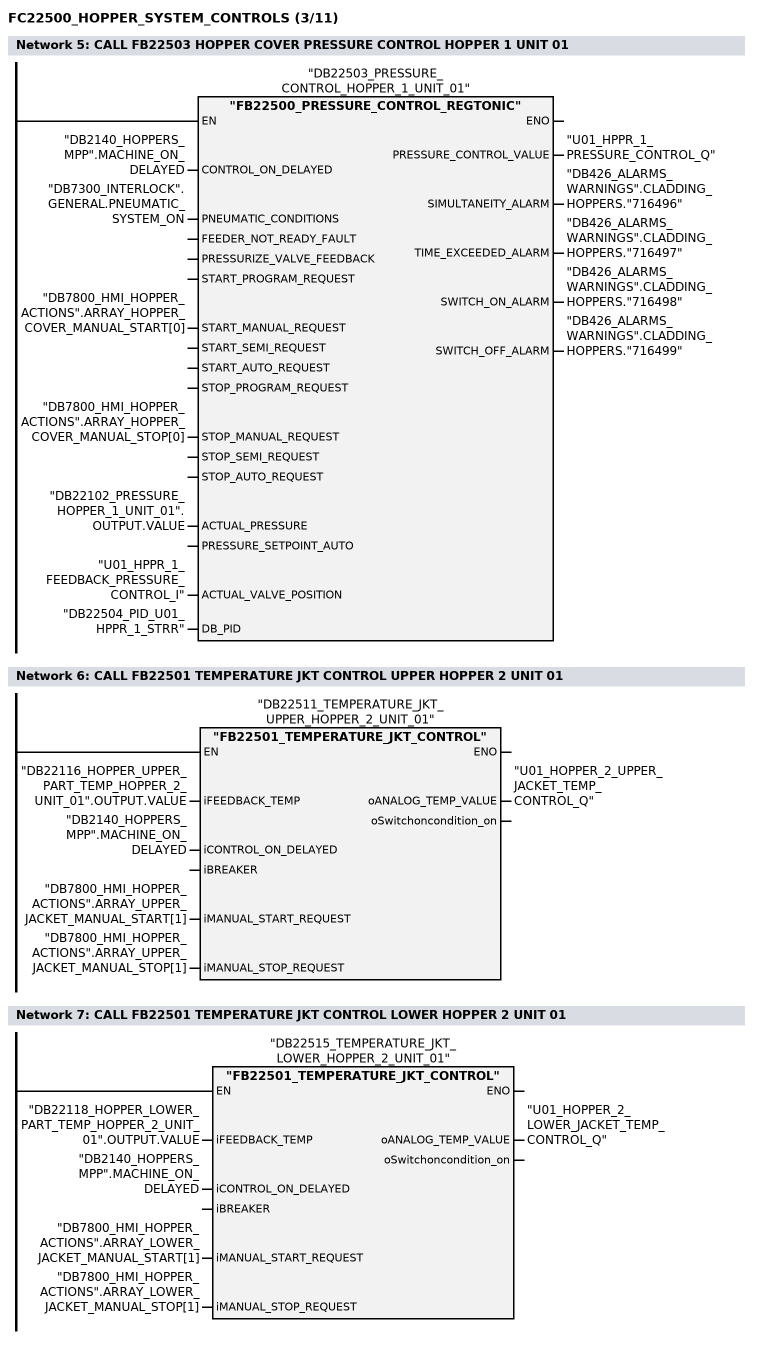
   RUNG wire#powerrail
      "DB22503_PRESSURE_CONTROL_HOPPER_1_UNIT_01"(CONTROL_ON_DELAYED := "DB2140_HOPPERS_MPP".MACHINE_ON_DELAYED, PNEUMATIC_CONDITIONS := "DB7300_INTERLOCK".GENERAL.PNEUMATIC_SYSTEM_ON, FEEDER_NOT_READY_FAULT :=, PRESSURIZE_VALVE_FEEDBACK :=, START_PROGRAM_REQUEST :=, START_MANUAL_REQUEST := "DB7800_HMI_HOPPER_ACTIONS".ARRAY_HOPPER_COVER_MANUAL_START[0], START_SEMI_REQUEST :=, START_AUTO_REQUEST :=, STOP_PROGRAM_REQUEST :=, STOP_MANUAL_REQUEST := "DB7800_HMI_HOPPER_ACTIONS".ARRAY_HOPPER_COVER_MANUAL_STOP[0], STOP_SEMI_REQUEST :=, STOP_AUTO_REQUEST :=, ACTUAL_PRESSURE := "DB22102_PRESSURE_HOPPER_1_UNIT_01".OUTPUT.VALUE, PRESSURE_SETPOINT_AUTO :=, ACTUAL_VALVE_POSITION := "U01_HPPR_1_FEEDBACK_PRESSURE_CONTROL_I", DB_PID := "DB22504_PID_U01_HPPR_1_STRR", PRESSURE_CONTROL_VALUE => "U01_HPPR_1_PRESSURE_CONTROL_Q", SIMULTANEITY_ALARM => "DB426_ALARMS_WARNINGS".CLADDING_HOPPERS."716496", TIME_EXCEEDED_ALARM => "DB426_ALARMS_WARNINGS".CLADDING_HOPPERS."716497", SWITCH_ON_ALARM => "DB426_ALARMS_WARNINGS".CLADDING_HOPPERS."716498", SWITCH_OFF_ALARM => "DB426_ALARMS_WARNINGS".CLADDING_HOPPERS."716499")
   END_RUNG
   // the same network as SCL:
   "DB22503_PRESSURE_CONTROL_HOPPER_1_UNIT_01"(CONTROL_ON_DELAYED := "DB2140_HOPPERS_MPP".MACHINE_ON_DELAYED,   // "FB22500_PRESSURE_CONTROL_REGTONIC"
                           PNEUMATIC_CONDITIONS := "DB7300_INTERLOCK".GENERAL.PNEUMATIC_SYSTEM_ON,
                           START_MANUAL_REQUEST := "DB7800_HMI_HOPPER_ACTIONS".ARRAY_HOPPER_COVER_MANUAL_START[0],
                           STOP_MANUAL_REQUEST := "DB7800_HMI_HOPPER_ACTIONS".ARRAY_HOPPER_COVER_MANUAL_STOP[0],
                           ACTUAL_PRESSURE := "DB22102_PRESSURE_HOPPER_1_UNIT_01".OUTPUT.VALUE,
                           ACTUAL_VALVE_POSITION := "U01_HPPR_1_FEEDBACK_PRESSURE_CONTROL_I",
                           DB_PID := "DB22504_PID_U01_HPPR_1_STRR",
                           PRESSURE_CONTROL_VALUE => "U01_HPPR_1_PRESSURE_CONTROL_Q",
                           SIMULTANEITY_ALARM => "DB426_ALARMS_WARNINGS".CLADDING_HOPPERS."716496",
                           TIME_EXCEEDED_ALARM => "DB426_ALARMS_WARNINGS".CLADDING_HOPPERS."716497",
                           SWITCH_ON_ALARM => "DB426_ALARMS_WARNINGS".CLADDING_HOPPERS."716498",
                           SWITCH_OFF_ALARM => "DB426_ALARMS_WARNINGS".CLADDING_HOPPERS."716499");
END_REGION

REGION Network 6: CALL FB22501 TEMPERATURE JKT CONTROL UPPER HOPPER 2 UNIT 01
   RUNG wire#powerrail
      "DB22511_TEMPERATURE_JKT_UPPER_HOPPER_2_UNIT_01"(iFEEDBACK_TEMP := "DB22116_HOPPER_UPPER_PART_TEMP_HOPPER_2_UNIT_01".OUTPUT.VALUE, iCONTROL_ON_DELAYED := "DB2140_HOPPERS_MPP".MACHINE_ON_DELAYED, iBREAKER :=, iMANUAL_START_REQUEST := "DB7800_HMI_HOPPER_ACTIONS".ARRAY_UPPER_JACKET_MANUAL_START[1], iMANUAL_STOP_REQUEST := "DB7800_HMI_HOPPER_ACTIONS".ARRAY_UPPER_JACKET_MANUAL_STOP[1], oANALOG_TEMP_VALUE => "U01_HOPPER_2_UPPER_JACKET_TEMP_CONTROL_Q", oSwitchoncondition_on =>)
   END_RUNG
   // the same network as SCL:
   "DB22511_TEMPERATURE_JKT_UPPER_HOPPER_2_UNIT_01"(iFEEDBACK_TEMP := "DB22116_HOPPER_UPPER_PART_TEMP_HOPPER_2_UNIT_01".OUTPUT.VALUE,   // "FB22501_TEMPERATURE_JKT_CONTROL"
                           iCONTROL_ON_DELAYED := "DB2140_HOPPERS_MPP".MACHINE_ON_DELAYED,
                           iMANUAL_START_REQUEST := "DB7800_HMI_HOPPER_ACTIONS".ARRAY_UPPER_JACKET_MANUAL_START[1],
                           iMANUAL_STOP_REQUEST := "DB7800_HMI_HOPPER_ACTIONS".ARRAY_UPPER_JACKET_MANUAL_STOP[1],
                           oANALOG_TEMP_VALUE => "U01_HOPPER_2_UPPER_JACKET_TEMP_CONTROL_Q");
END_REGION

REGION Network 7: CALL FB22501 TEMPERATURE JKT CONTROL LOWER HOPPER 2 UNIT 01
   RUNG wire#powerrail
      "DB22515_TEMPERATURE_JKT_LOWER_HOPPER_2_UNIT_01"(iFEEDBACK_TEMP := "DB22118_HOPPER_LOWER_PART_TEMP_HOPPER_2_UNIT_01".OUTPUT.VALUE, iCONTROL_ON_DELAYED := "DB2140_HOPPERS_MPP".MACHINE_ON_DELAYED, iBREAKER :=, iMANUAL_START_REQUEST := "DB7800_HMI_HOPPER_ACTIONS".ARRAY_LOWER_JACKET_MANUAL_START[1], iMANUAL_STOP_REQUEST := "DB7800_HMI_HOPPER_ACTIONS".ARRAY_LOWER_JACKET_MANUAL_STOP[1], oANALOG_TEMP_VALUE => "U01_HOPPER_2_LOWER_JACKET_TEMP_CONTROL_Q", oSwitchoncondition_on =>)
   END_RUNG
   // the same network as SCL:
   "DB22515_TEMPERATURE_JKT_LOWER_HOPPER_2_UNIT_01"(iFEEDBACK_TEMP := "DB22118_HOPPER_LOWER_PART_TEMP_HOPPER_2_UNIT_01".OUTPUT.VALUE,   // "FB22501_TEMPERATURE_JKT_CONTROL"
                           iCONTROL_ON_DELAYED := "DB2140_HOPPERS_MPP".MACHINE_ON_DELAYED,
                           iMANUAL_START_REQUEST := "DB7800_HMI_HOPPER_ACTIONS".ARRAY_LOWER_JACKET_MANUAL_START[1],
                           iMANUAL_STOP_REQUEST := "DB7800_HMI_HOPPER_ACTIONS".ARRAY_LOWER_JACKET_MANUAL_STOP[1],
                           oANALOG_TEMP_VALUE => "U01_HOPPER_2_LOWER_JACKET_TEMP_CONTROL_Q");
END_REGION

REGION Network 8: CALL FB22502 MOTOR STIRRER CONTROL HOPPER 2 UNIT 01
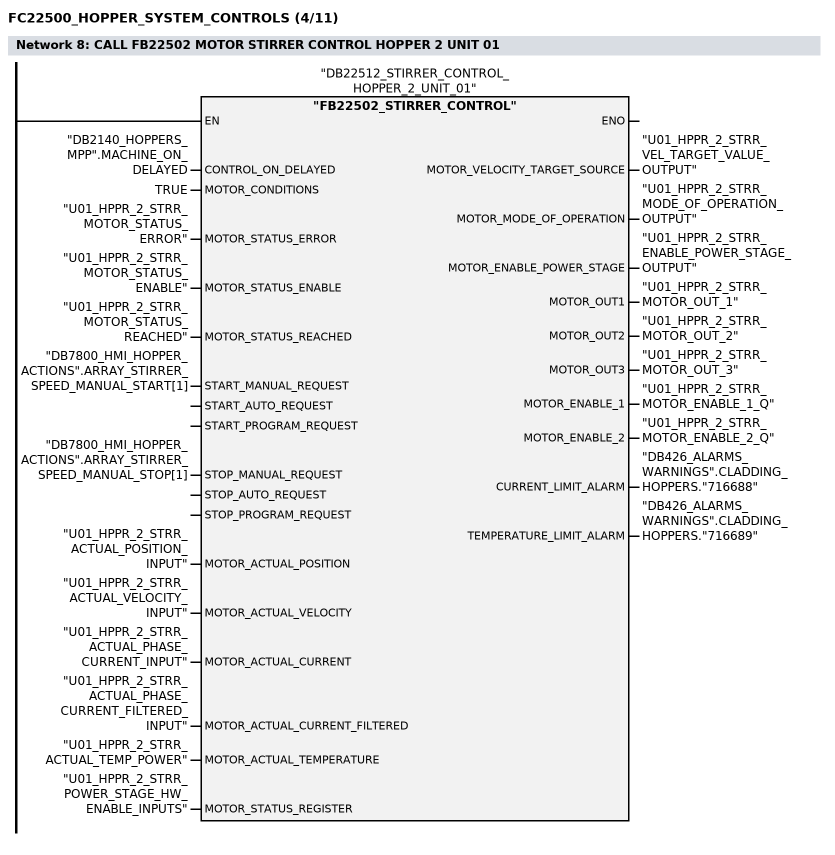
   RUNG wire#powerrail
      "DB22512_STIRRER_CONTROL_HOPPER_2_UNIT_01"(CONTROL_ON_DELAYED := "DB2140_HOPPERS_MPP".MACHINE_ON_DELAYED, MOTOR_CONDITIONS := TRUE, MOTOR_STATUS_ERROR := "U01_HPPR_2_STRR_MOTOR_STATUS_ERROR", MOTOR_STATUS_ENABLE := "U01_HPPR_2_STRR_MOTOR_STATUS_ENABLE", MOTOR_STATUS_REACHED := "U01_HPPR_2_STRR_MOTOR_STATUS_REACHED", START_MANUAL_REQUEST := "DB7800_HMI_HOPPER_ACTIONS".ARRAY_STIRRER_SPEED_MANUAL_START[1], START_AUTO_REQUEST :=, START_PROGRAM_REQUEST :=, STOP_MANUAL_REQUEST := "DB7800_HMI_HOPPER_ACTIONS".ARRAY_STIRRER_SPEED_MANUAL_STOP[1], STOP_AUTO_REQUEST :=, STOP_PROGRAM_REQUEST :=, MOTOR_ACTUAL_POSITION := "U01_HPPR_2_STRR_ACTUAL_POSITION_INPUT", MOTOR_ACTUAL_VELOCITY := "U01_HPPR_2_STRR_ACTUAL_VELOCITY_INPUT", MOTOR_ACTUAL_CURRENT := "U01_HPPR_2_STRR_ACTUAL_PHASE_CURRENT_INPUT", MOTOR_ACTUAL_CURRENT_FILTERED := "U01_HPPR_2_STRR_ACTUAL_PHASE_CURRENT_FILTERED_INPUT", MOTOR_ACTUAL_TEMPERATURE := "U01_HPPR_2_STRR_ACTUAL_TEMP_POWER", MOTOR_STATUS_REGISTER := "U01_HPPR_2_STRR_POWER_STAGE_HW_ENABLE_INPUTS", MOTOR_VELOCITY_TARGET_SOURCE => "U01_HPPR_2_STRR_VEL_TARGET_VALUE_OUTPUT", MOTOR_MODE_OF_OPERATION => "U01_HPPR_2_STRR_MODE_OF_OPERATION_OUTPUT", MOTOR_ENABLE_POWER_STAGE => "U01_HPPR_2_STRR_ENABLE_POWER_STAGE_OUTPUT", MOTOR_OUT1 => "U01_HPPR_2_STRR_MOTOR_OUT_1", MOTOR_OUT2 => "U01_HPPR_2_STRR_MOTOR_OUT_2", MOTOR_OUT3 => "U01_HPPR_2_STRR_MOTOR_OUT_3", MOTOR_ENABLE_1 => "U01_HPPR_2_STRR_MOTOR_ENABLE_1_Q", MOTOR_ENABLE_2 => "U01_HPPR_2_STRR_MOTOR_ENABLE_2_Q", CURRENT_LIMIT_ALARM => "DB426_ALARMS_WARNINGS".CLADDING_HOPPERS."716688", TEMPERATURE_LIMIT_ALARM => "DB426_ALARMS_WARNINGS".CLADDING_HOPPERS."716689")
   END_RUNG
   // the same network as SCL:
   "DB22512_STIRRER_CONTROL_HOPPER_2_UNIT_01"(CONTROL_ON_DELAYED := "DB2140_HOPPERS_MPP".MACHINE_ON_DELAYED,   // "FB22502_STIRRER_CONTROL"
                           MOTOR_CONDITIONS := TRUE,
                           MOTOR_STATUS_ERROR := "U01_HPPR_2_STRR_MOTOR_STATUS_ERROR",
                           MOTOR_STATUS_ENABLE := "U01_HPPR_2_STRR_MOTOR_STATUS_ENABLE",
                           MOTOR_STATUS_REACHED := "U01_HPPR_2_STRR_MOTOR_STATUS_REACHED",
                           START_MANUAL_REQUEST := "DB7800_HMI_HOPPER_ACTIONS".ARRAY_STIRRER_SPEED_MANUAL_START[1],
                           STOP_MANUAL_REQUEST := "DB7800_HMI_HOPPER_ACTIONS".ARRAY_STIRRER_SPEED_MANUAL_STOP[1],
                           MOTOR_ACTUAL_POSITION := "U01_HPPR_2_STRR_ACTUAL_POSITION_INPUT",
                           MOTOR_ACTUAL_VELOCITY := "U01_HPPR_2_STRR_ACTUAL_VELOCITY_INPUT",
                           MOTOR_ACTUAL_CURRENT := "U01_HPPR_2_STRR_ACTUAL_PHASE_CURRENT_INPUT",
                           MOTOR_ACTUAL_CURRENT_FILTERED := "U01_HPPR_2_STRR_ACTUAL_PHASE_CURRENT_FILTERED_INPUT",
                           MOTOR_ACTUAL_TEMPERATURE := "U01_HPPR_2_STRR_ACTUAL_TEMP_POWER",
                           MOTOR_STATUS_REGISTER := "U01_HPPR_2_STRR_POWER_STAGE_HW_ENABLE_INPUTS",
                           MOTOR_VELOCITY_TARGET_SOURCE => "U01_HPPR_2_STRR_VEL_TARGET_VALUE_OUTPUT",
                           MOTOR_MODE_OF_OPERATION => "U01_HPPR_2_STRR_MODE_OF_OPERATION_OUTPUT",
                           MOTOR_ENABLE_POWER_STAGE => "U01_HPPR_2_STRR_ENABLE_POWER_STAGE_OUTPUT",
                           MOTOR_OUT1 => "U01_HPPR_2_STRR_MOTOR_OUT_1",
                           MOTOR_OUT2 => "U01_HPPR_2_STRR_MOTOR_OUT_2",
                           MOTOR_OUT3 => "U01_HPPR_2_STRR_MOTOR_OUT_3",
                           MOTOR_ENABLE_1 => "U01_HPPR_2_STRR_MOTOR_ENABLE_1_Q",
                           MOTOR_ENABLE_2 => "U01_HPPR_2_STRR_MOTOR_ENABLE_2_Q",
                           CURRENT_LIMIT_ALARM => "DB426_ALARMS_WARNINGS".CLADDING_HOPPERS."716688",
                           TEMPERATURE_LIMIT_ALARM => "DB426_ALARMS_WARNINGS".CLADDING_HOPPERS."716689");
END_REGION

REGION Network 9: CALL FB22503 HOPPER PRESSURE CONTROL HOPPER 2 UNIT 01
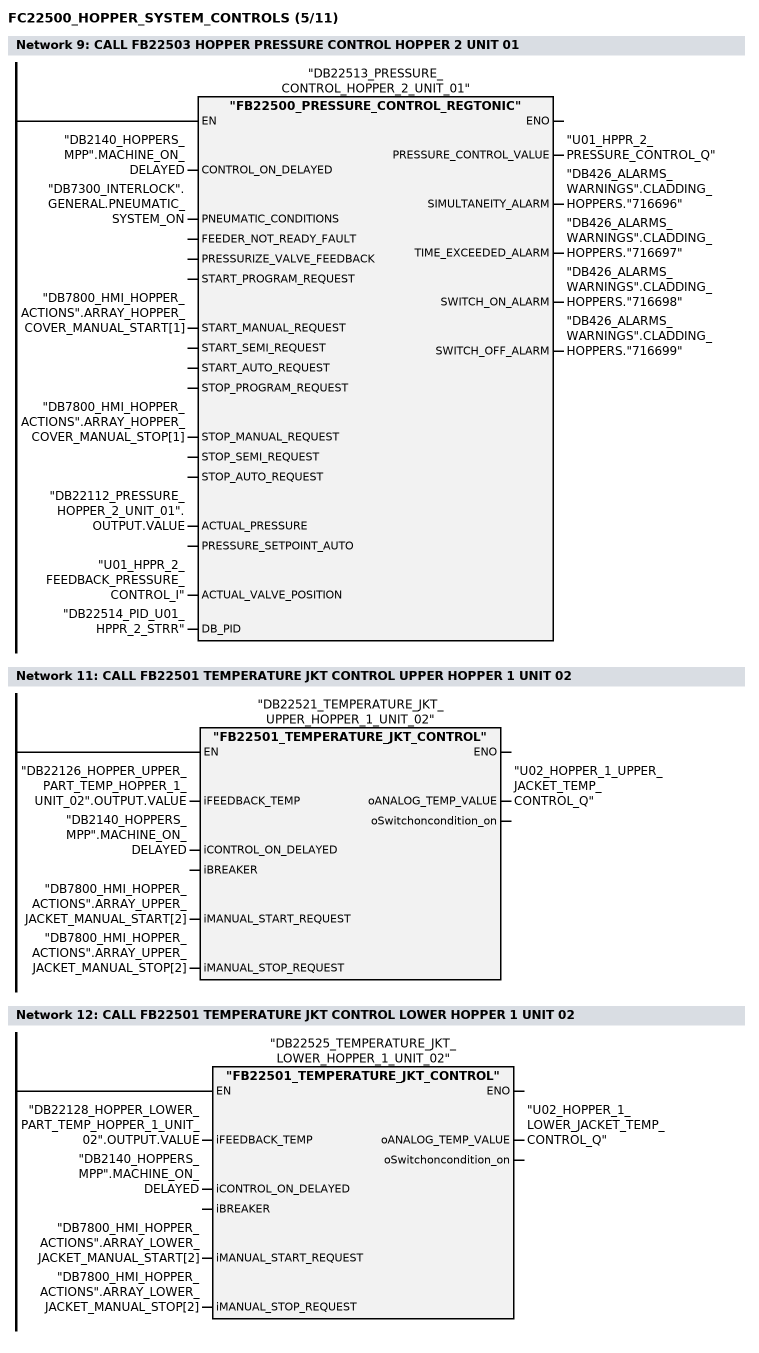
   RUNG wire#powerrail
      "DB22513_PRESSURE_CONTROL_HOPPER_2_UNIT_01"(CONTROL_ON_DELAYED := "DB2140_HOPPERS_MPP".MACHINE_ON_DELAYED, PNEUMATIC_CONDITIONS := "DB7300_INTERLOCK".GENERAL.PNEUMATIC_SYSTEM_ON, FEEDER_NOT_READY_FAULT :=, PRESSURIZE_VALVE_FEEDBACK :=, START_PROGRAM_REQUEST :=, START_MANUAL_REQUEST := "DB7800_HMI_HOPPER_ACTIONS".ARRAY_HOPPER_COVER_MANUAL_START[1], START_SEMI_REQUEST :=, START_AUTO_REQUEST :=, STOP_PROGRAM_REQUEST :=, STOP_MANUAL_REQUEST := "DB7800_HMI_HOPPER_ACTIONS".ARRAY_HOPPER_COVER_MANUAL_STOP[1], STOP_SEMI_REQUEST :=, STOP_AUTO_REQUEST :=, ACTUAL_PRESSURE := "DB22112_PRESSURE_HOPPER_2_UNIT_01".OUTPUT.VALUE, PRESSURE_SETPOINT_AUTO :=, ACTUAL_VALVE_POSITION := "U01_HPPR_2_FEEDBACK_PRESSURE_CONTROL_I", DB_PID := "DB22514_PID_U01_HPPR_2_STRR", PRESSURE_CONTROL_VALUE => "U01_HPPR_2_PRESSURE_CONTROL_Q", SIMULTANEITY_ALARM => "DB426_ALARMS_WARNINGS".CLADDING_HOPPERS."716696", TIME_EXCEEDED_ALARM => "DB426_ALARMS_WARNINGS".CLADDING_HOPPERS."716697", SWITCH_ON_ALARM => "DB426_ALARMS_WARNINGS".CLADDING_HOPPERS."716698", SWITCH_OFF_ALARM => "DB426_ALARMS_WARNINGS".CLADDING_HOPPERS."716699")
   END_RUNG
   // the same network as SCL:
   "DB22513_PRESSURE_CONTROL_HOPPER_2_UNIT_01"(CONTROL_ON_DELAYED := "DB2140_HOPPERS_MPP".MACHINE_ON_DELAYED,   // "FB22500_PRESSURE_CONTROL_REGTONIC"
                           PNEUMATIC_CONDITIONS := "DB7300_INTERLOCK".GENERAL.PNEUMATIC_SYSTEM_ON,
                           START_MANUAL_REQUEST := "DB7800_HMI_HOPPER_ACTIONS".ARRAY_HOPPER_COVER_MANUAL_START[1],
                           STOP_MANUAL_REQUEST := "DB7800_HMI_HOPPER_ACTIONS".ARRAY_HOPPER_COVER_MANUAL_STOP[1],
                           ACTUAL_PRESSURE := "DB22112_PRESSURE_HOPPER_2_UNIT_01".OUTPUT.VALUE,
                           ACTUAL_VALVE_POSITION := "U01_HPPR_2_FEEDBACK_PRESSURE_CONTROL_I",
                           DB_PID := "DB22514_PID_U01_HPPR_2_STRR",
                           PRESSURE_CONTROL_VALUE => "U01_HPPR_2_PRESSURE_CONTROL_Q",
                           SIMULTANEITY_ALARM => "DB426_ALARMS_WARNINGS".CLADDING_HOPPERS."716696",
                           TIME_EXCEEDED_ALARM => "DB426_ALARMS_WARNINGS".CLADDING_HOPPERS."716697",
                           SWITCH_ON_ALARM => "DB426_ALARMS_WARNINGS".CLADDING_HOPPERS."716698",
                           SWITCH_OFF_ALARM => "DB426_ALARMS_WARNINGS".CLADDING_HOPPERS."716699");
END_REGION

REGION Network 10: //////////UNIT 02 HOPERS CONTROLS//////////
END_REGION

REGION Network 11: CALL FB22501 TEMPERATURE JKT CONTROL UPPER HOPPER 1 UNIT 02
   RUNG wire#powerrail
      "DB22521_TEMPERATURE_JKT_UPPER_HOPPER_1_UNIT_02"(iFEEDBACK_TEMP := "DB22126_HOPPER_UPPER_PART_TEMP_HOPPER_1_UNIT_02".OUTPUT.VALUE, iCONTROL_ON_DELAYED := "DB2140_HOPPERS_MPP".MACHINE_ON_DELAYED, iBREAKER :=, iMANUAL_START_REQUEST := "DB7800_HMI_HOPPER_ACTIONS".ARRAY_UPPER_JACKET_MANUAL_START[2], iMANUAL_STOP_REQUEST := "DB7800_HMI_HOPPER_ACTIONS".ARRAY_UPPER_JACKET_MANUAL_STOP[2], oANALOG_TEMP_VALUE => "U02_HOPPER_1_UPPER_JACKET_TEMP_CONTROL_Q", oSwitchoncondition_on =>)
   END_RUNG
   // the same network as SCL:
   "DB22521_TEMPERATURE_JKT_UPPER_HOPPER_1_UNIT_02"(iFEEDBACK_TEMP := "DB22126_HOPPER_UPPER_PART_TEMP_HOPPER_1_UNIT_02".OUTPUT.VALUE,   // "FB22501_TEMPERATURE_JKT_CONTROL"
                           iCONTROL_ON_DELAYED := "DB2140_HOPPERS_MPP".MACHINE_ON_DELAYED,
                           iMANUAL_START_REQUEST := "DB7800_HMI_HOPPER_ACTIONS".ARRAY_UPPER_JACKET_MANUAL_START[2],
                           iMANUAL_STOP_REQUEST := "DB7800_HMI_HOPPER_ACTIONS".ARRAY_UPPER_JACKET_MANUAL_STOP[2],
                           oANALOG_TEMP_VALUE => "U02_HOPPER_1_UPPER_JACKET_TEMP_CONTROL_Q");
END_REGION

REGION Network 12: CALL FB22501 TEMPERATURE JKT CONTROL LOWER HOPPER 1 UNIT 02
   RUNG wire#powerrail
      "DB22525_TEMPERATURE_JKT_LOWER_HOPPER_1_UNIT_02"(iFEEDBACK_TEMP := "DB22128_HOPPER_LOWER_PART_TEMP_HOPPER_1_UNIT_02".OUTPUT.VALUE, iCONTROL_ON_DELAYED := "DB2140_HOPPERS_MPP".MACHINE_ON_DELAYED, iBREAKER :=, iMANUAL_START_REQUEST := "DB7800_HMI_HOPPER_ACTIONS".ARRAY_LOWER_JACKET_MANUAL_START[2], iMANUAL_STOP_REQUEST := "DB7800_HMI_HOPPER_ACTIONS".ARRAY_LOWER_JACKET_MANUAL_STOP[2], oANALOG_TEMP_VALUE => "U02_HOPPER_1_LOWER_JACKET_TEMP_CONTROL_Q", oSwitchoncondition_on =>)
   END_RUNG
   // the same network as SCL:
   "DB22525_TEMPERATURE_JKT_LOWER_HOPPER_1_UNIT_02"(iFEEDBACK_TEMP := "DB22128_HOPPER_LOWER_PART_TEMP_HOPPER_1_UNIT_02".OUTPUT.VALUE,   // "FB22501_TEMPERATURE_JKT_CONTROL"
                           iCONTROL_ON_DELAYED := "DB2140_HOPPERS_MPP".MACHINE_ON_DELAYED,
                           iMANUAL_START_REQUEST := "DB7800_HMI_HOPPER_ACTIONS".ARRAY_LOWER_JACKET_MANUAL_START[2],
                           iMANUAL_STOP_REQUEST := "DB7800_HMI_HOPPER_ACTIONS".ARRAY_LOWER_JACKET_MANUAL_STOP[2],
                           oANALOG_TEMP_VALUE => "U02_HOPPER_1_LOWER_JACKET_TEMP_CONTROL_Q");
END_REGION

REGION Network 13: CALL FB22502 MOTOR STIRRER CONTROL HOPPER 1 UNIT 02
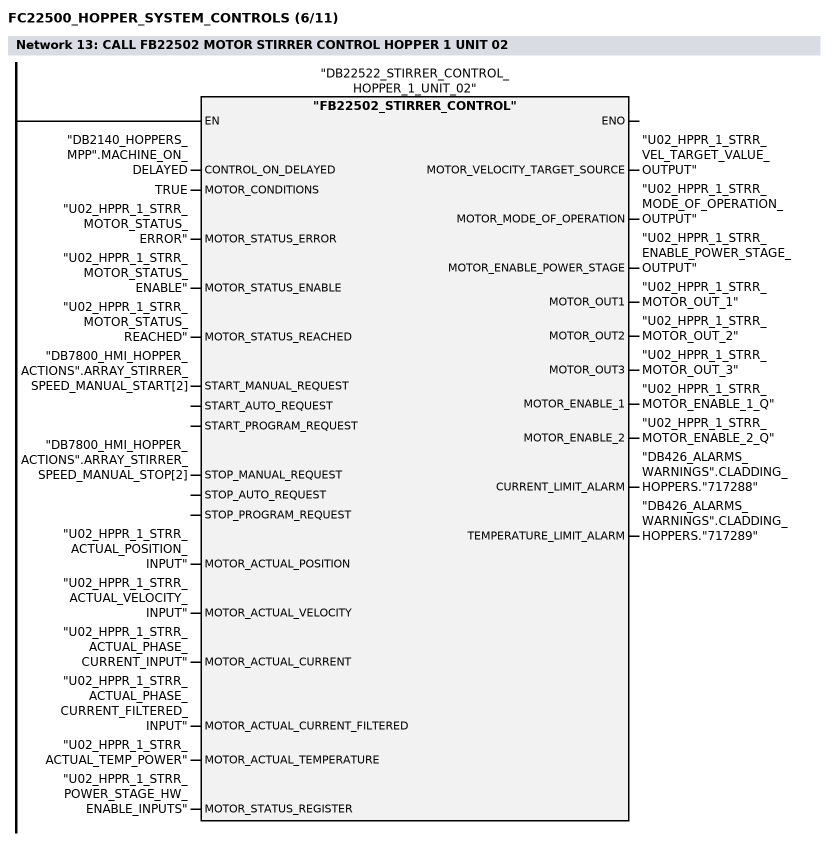
   RUNG wire#powerrail
      "DB22522_STIRRER_CONTROL_HOPPER_1_UNIT_02"(CONTROL_ON_DELAYED := "DB2140_HOPPERS_MPP".MACHINE_ON_DELAYED, MOTOR_CONDITIONS := TRUE, MOTOR_STATUS_ERROR := "U02_HPPR_1_STRR_MOTOR_STATUS_ERROR", MOTOR_STATUS_ENABLE := "U02_HPPR_1_STRR_MOTOR_STATUS_ENABLE", MOTOR_STATUS_REACHED := "U02_HPPR_1_STRR_MOTOR_STATUS_REACHED", START_MANUAL_REQUEST := "DB7800_HMI_HOPPER_ACTIONS".ARRAY_STIRRER_SPEED_MANUAL_START[2], START_AUTO_REQUEST :=, START_PROGRAM_REQUEST :=, STOP_MANUAL_REQUEST := "DB7800_HMI_HOPPER_ACTIONS".ARRAY_STIRRER_SPEED_MANUAL_STOP[2], STOP_AUTO_REQUEST :=, STOP_PROGRAM_REQUEST :=, MOTOR_ACTUAL_POSITION := "U02_HPPR_1_STRR_ACTUAL_POSITION_INPUT", MOTOR_ACTUAL_VELOCITY := "U02_HPPR_1_STRR_ACTUAL_VELOCITY_INPUT", MOTOR_ACTUAL_CURRENT := "U02_HPPR_1_STRR_ACTUAL_PHASE_CURRENT_INPUT", MOTOR_ACTUAL_CURRENT_FILTERED := "U02_HPPR_1_STRR_ACTUAL_PHASE_CURRENT_FILTERED_INPUT", MOTOR_ACTUAL_TEMPERATURE := "U02_HPPR_1_STRR_ACTUAL_TEMP_POWER", MOTOR_STATUS_REGISTER := "U02_HPPR_1_STRR_POWER_STAGE_HW_ENABLE_INPUTS", MOTOR_VELOCITY_TARGET_SOURCE => "U02_HPPR_1_STRR_VEL_TARGET_VALUE_OUTPUT", MOTOR_MODE_OF_OPERATION => "U02_HPPR_1_STRR_MODE_OF_OPERATION_OUTPUT", MOTOR_ENABLE_POWER_STAGE => "U02_HPPR_1_STRR_ENABLE_POWER_STAGE_OUTPUT", MOTOR_OUT1 => "U02_HPPR_1_STRR_MOTOR_OUT_1", MOTOR_OUT2 => "U02_HPPR_1_STRR_MOTOR_OUT_2", MOTOR_OUT3 => "U02_HPPR_1_STRR_MOTOR_OUT_3", MOTOR_ENABLE_1 => "U02_HPPR_1_STRR_MOTOR_ENABLE_1_Q", MOTOR_ENABLE_2 => "U02_HPPR_1_STRR_MOTOR_ENABLE_2_Q", CURRENT_LIMIT_ALARM => "DB426_ALARMS_WARNINGS".CLADDING_HOPPERS."717288", TEMPERATURE_LIMIT_ALARM => "DB426_ALARMS_WARNINGS".CLADDING_HOPPERS."717289")
   END_RUNG
   // the same network as SCL:
   "DB22522_STIRRER_CONTROL_HOPPER_1_UNIT_02"(CONTROL_ON_DELAYED := "DB2140_HOPPERS_MPP".MACHINE_ON_DELAYED,   // "FB22502_STIRRER_CONTROL"
                           MOTOR_CONDITIONS := TRUE,
                           MOTOR_STATUS_ERROR := "U02_HPPR_1_STRR_MOTOR_STATUS_ERROR",
                           MOTOR_STATUS_ENABLE := "U02_HPPR_1_STRR_MOTOR_STATUS_ENABLE",
                           MOTOR_STATUS_REACHED := "U02_HPPR_1_STRR_MOTOR_STATUS_REACHED",
                           START_MANUAL_REQUEST := "DB7800_HMI_HOPPER_ACTIONS".ARRAY_STIRRER_SPEED_MANUAL_START[2],
                           STOP_MANUAL_REQUEST := "DB7800_HMI_HOPPER_ACTIONS".ARRAY_STIRRER_SPEED_MANUAL_STOP[2],
                           MOTOR_ACTUAL_POSITION := "U02_HPPR_1_STRR_ACTUAL_POSITION_INPUT",
                           MOTOR_ACTUAL_VELOCITY := "U02_HPPR_1_STRR_ACTUAL_VELOCITY_INPUT",
                           MOTOR_ACTUAL_CURRENT := "U02_HPPR_1_STRR_ACTUAL_PHASE_CURRENT_INPUT",
                           MOTOR_ACTUAL_CURRENT_FILTERED := "U02_HPPR_1_STRR_ACTUAL_PHASE_CURRENT_FILTERED_INPUT",
                           MOTOR_ACTUAL_TEMPERATURE := "U02_HPPR_1_STRR_ACTUAL_TEMP_POWER",
                           MOTOR_STATUS_REGISTER := "U02_HPPR_1_STRR_POWER_STAGE_HW_ENABLE_INPUTS",
                           MOTOR_VELOCITY_TARGET_SOURCE => "U02_HPPR_1_STRR_VEL_TARGET_VALUE_OUTPUT",
                           MOTOR_MODE_OF_OPERATION => "U02_HPPR_1_STRR_MODE_OF_OPERATION_OUTPUT",
                           MOTOR_ENABLE_POWER_STAGE => "U02_HPPR_1_STRR_ENABLE_POWER_STAGE_OUTPUT",
                           MOTOR_OUT1 => "U02_HPPR_1_STRR_MOTOR_OUT_1",
                           MOTOR_OUT2 => "U02_HPPR_1_STRR_MOTOR_OUT_2",
                           MOTOR_OUT3 => "U02_HPPR_1_STRR_MOTOR_OUT_3",
                           MOTOR_ENABLE_1 => "U02_HPPR_1_STRR_MOTOR_ENABLE_1_Q",
                           MOTOR_ENABLE_2 => "U02_HPPR_1_STRR_MOTOR_ENABLE_2_Q",
                           CURRENT_LIMIT_ALARM => "DB426_ALARMS_WARNINGS".CLADDING_HOPPERS."717288",
                           TEMPERATURE_LIMIT_ALARM => "DB426_ALARMS_WARNINGS".CLADDING_HOPPERS."717289");
END_REGION

REGION Network 14: CALL FB22503 HOPPER PRESSURE CONTROL HOPPER 1 UNIT 02
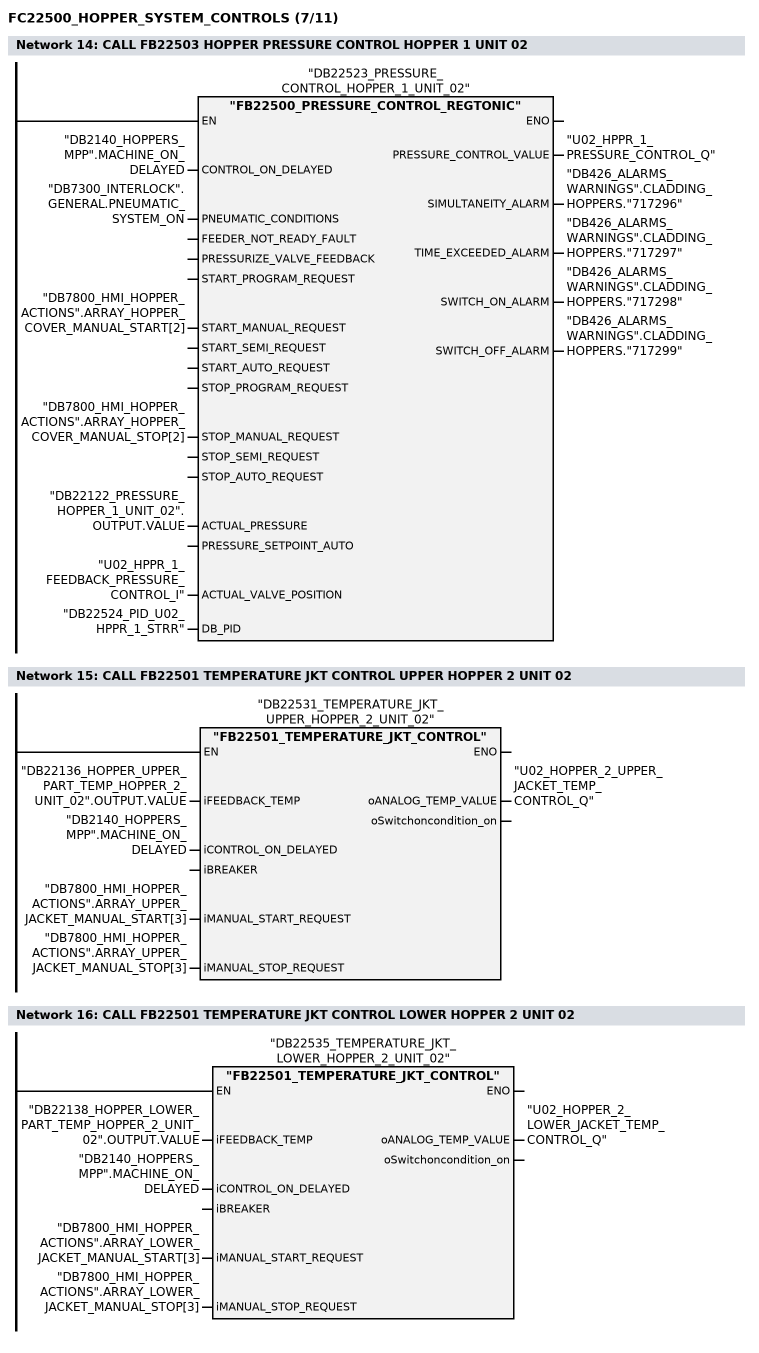
   RUNG wire#powerrail
      "DB22523_PRESSURE_CONTROL_HOPPER_1_UNIT_02"(CONTROL_ON_DELAYED := "DB2140_HOPPERS_MPP".MACHINE_ON_DELAYED, PNEUMATIC_CONDITIONS := "DB7300_INTERLOCK".GENERAL.PNEUMATIC_SYSTEM_ON, FEEDER_NOT_READY_FAULT :=, PRESSURIZE_VALVE_FEEDBACK :=, START_PROGRAM_REQUEST :=, START_MANUAL_REQUEST := "DB7800_HMI_HOPPER_ACTIONS".ARRAY_HOPPER_COVER_MANUAL_START[2], START_SEMI_REQUEST :=, START_AUTO_REQUEST :=, STOP_PROGRAM_REQUEST :=, STOP_MANUAL_REQUEST := "DB7800_HMI_HOPPER_ACTIONS".ARRAY_HOPPER_COVER_MANUAL_STOP[2], STOP_SEMI_REQUEST :=, STOP_AUTO_REQUEST :=, ACTUAL_PRESSURE := "DB22122_PRESSURE_HOPPER_1_UNIT_02".OUTPUT.VALUE, PRESSURE_SETPOINT_AUTO :=, ACTUAL_VALVE_POSITION := "U02_HPPR_1_FEEDBACK_PRESSURE_CONTROL_I", DB_PID := "DB22524_PID_U02_HPPR_1_STRR", PRESSURE_CONTROL_VALUE => "U02_HPPR_1_PRESSURE_CONTROL_Q", SIMULTANEITY_ALARM => "DB426_ALARMS_WARNINGS".CLADDING_HOPPERS."717296", TIME_EXCEEDED_ALARM => "DB426_ALARMS_WARNINGS".CLADDING_HOPPERS."717297", SWITCH_ON_ALARM => "DB426_ALARMS_WARNINGS".CLADDING_HOPPERS."717298", SWITCH_OFF_ALARM => "DB426_ALARMS_WARNINGS".CLADDING_HOPPERS."717299")
   END_RUNG
   // the same network as SCL:
   "DB22523_PRESSURE_CONTROL_HOPPER_1_UNIT_02"(CONTROL_ON_DELAYED := "DB2140_HOPPERS_MPP".MACHINE_ON_DELAYED,   // "FB22500_PRESSURE_CONTROL_REGTONIC"
                           PNEUMATIC_CONDITIONS := "DB7300_INTERLOCK".GENERAL.PNEUMATIC_SYSTEM_ON,
                           START_MANUAL_REQUEST := "DB7800_HMI_HOPPER_ACTIONS".ARRAY_HOPPER_COVER_MANUAL_START[2],
                           STOP_MANUAL_REQUEST := "DB7800_HMI_HOPPER_ACTIONS".ARRAY_HOPPER_COVER_MANUAL_STOP[2],
                           ACTUAL_PRESSURE := "DB22122_PRESSURE_HOPPER_1_UNIT_02".OUTPUT.VALUE,
                           ACTUAL_VALVE_POSITION := "U02_HPPR_1_FEEDBACK_PRESSURE_CONTROL_I",
                           DB_PID := "DB22524_PID_U02_HPPR_1_STRR",
                           PRESSURE_CONTROL_VALUE => "U02_HPPR_1_PRESSURE_CONTROL_Q",
                           SIMULTANEITY_ALARM => "DB426_ALARMS_WARNINGS".CLADDING_HOPPERS."717296",
                           TIME_EXCEEDED_ALARM => "DB426_ALARMS_WARNINGS".CLADDING_HOPPERS."717297",
                           SWITCH_ON_ALARM => "DB426_ALARMS_WARNINGS".CLADDING_HOPPERS."717298",
                           SWITCH_OFF_ALARM => "DB426_ALARMS_WARNINGS".CLADDING_HOPPERS."717299");
END_REGION

REGION Network 15: CALL FB22501 TEMPERATURE JKT CONTROL UPPER HOPPER 2 UNIT 02
   RUNG wire#powerrail
      "DB22531_TEMPERATURE_JKT_UPPER_HOPPER_2_UNIT_02"(iFEEDBACK_TEMP := "DB22136_HOPPER_UPPER_PART_TEMP_HOPPER_2_UNIT_02".OUTPUT.VALUE, iCONTROL_ON_DELAYED := "DB2140_HOPPERS_MPP".MACHINE_ON_DELAYED, iBREAKER :=, iMANUAL_START_REQUEST := "DB7800_HMI_HOPPER_ACTIONS".ARRAY_UPPER_JACKET_MANUAL_START[3], iMANUAL_STOP_REQUEST := "DB7800_HMI_HOPPER_ACTIONS".ARRAY_UPPER_JACKET_MANUAL_STOP[3], oANALOG_TEMP_VALUE => "U02_HOPPER_2_UPPER_JACKET_TEMP_CONTROL_Q", oSwitchoncondition_on =>)
   END_RUNG
   // the same network as SCL:
   "DB22531_TEMPERATURE_JKT_UPPER_HOPPER_2_UNIT_02"(iFEEDBACK_TEMP := "DB22136_HOPPER_UPPER_PART_TEMP_HOPPER_2_UNIT_02".OUTPUT.VALUE,   // "FB22501_TEMPERATURE_JKT_CONTROL"
                           iCONTROL_ON_DELAYED := "DB2140_HOPPERS_MPP".MACHINE_ON_DELAYED,
                           iMANUAL_START_REQUEST := "DB7800_HMI_HOPPER_ACTIONS".ARRAY_UPPER_JACKET_MANUAL_START[3],
                           iMANUAL_STOP_REQUEST := "DB7800_HMI_HOPPER_ACTIONS".ARRAY_UPPER_JACKET_MANUAL_STOP[3],
                           oANALOG_TEMP_VALUE => "U02_HOPPER_2_UPPER_JACKET_TEMP_CONTROL_Q");
END_REGION

REGION Network 16: CALL FB22501 TEMPERATURE JKT CONTROL LOWER HOPPER 2 UNIT 02
   RUNG wire#powerrail
      "DB22535_TEMPERATURE_JKT_LOWER_HOPPER_2_UNIT_02"(iFEEDBACK_TEMP := "DB22138_HOPPER_LOWER_PART_TEMP_HOPPER_2_UNIT_02".OUTPUT.VALUE, iCONTROL_ON_DELAYED := "DB2140_HOPPERS_MPP".MACHINE_ON_DELAYED, iBREAKER :=, iMANUAL_START_REQUEST := "DB7800_HMI_HOPPER_ACTIONS".ARRAY_LOWER_JACKET_MANUAL_START[3], iMANUAL_STOP_REQUEST := "DB7800_HMI_HOPPER_ACTIONS".ARRAY_LOWER_JACKET_MANUAL_STOP[3], oANALOG_TEMP_VALUE => "U02_HOPPER_2_LOWER_JACKET_TEMP_CONTROL_Q", oSwitchoncondition_on =>)
   END_RUNG
   // the same network as SCL:
   "DB22535_TEMPERATURE_JKT_LOWER_HOPPER_2_UNIT_02"(iFEEDBACK_TEMP := "DB22138_HOPPER_LOWER_PART_TEMP_HOPPER_2_UNIT_02".OUTPUT.VALUE,   // "FB22501_TEMPERATURE_JKT_CONTROL"
                           iCONTROL_ON_DELAYED := "DB2140_HOPPERS_MPP".MACHINE_ON_DELAYED,
                           iMANUAL_START_REQUEST := "DB7800_HMI_HOPPER_ACTIONS".ARRAY_LOWER_JACKET_MANUAL_START[3],
                           iMANUAL_STOP_REQUEST := "DB7800_HMI_HOPPER_ACTIONS".ARRAY_LOWER_JACKET_MANUAL_STOP[3],
                           oANALOG_TEMP_VALUE => "U02_HOPPER_2_LOWER_JACKET_TEMP_CONTROL_Q");
END_REGION

REGION Network 17: CALL FB22502 MOTOR STIRRER CONTROL HOPPER 2 UNIT 02
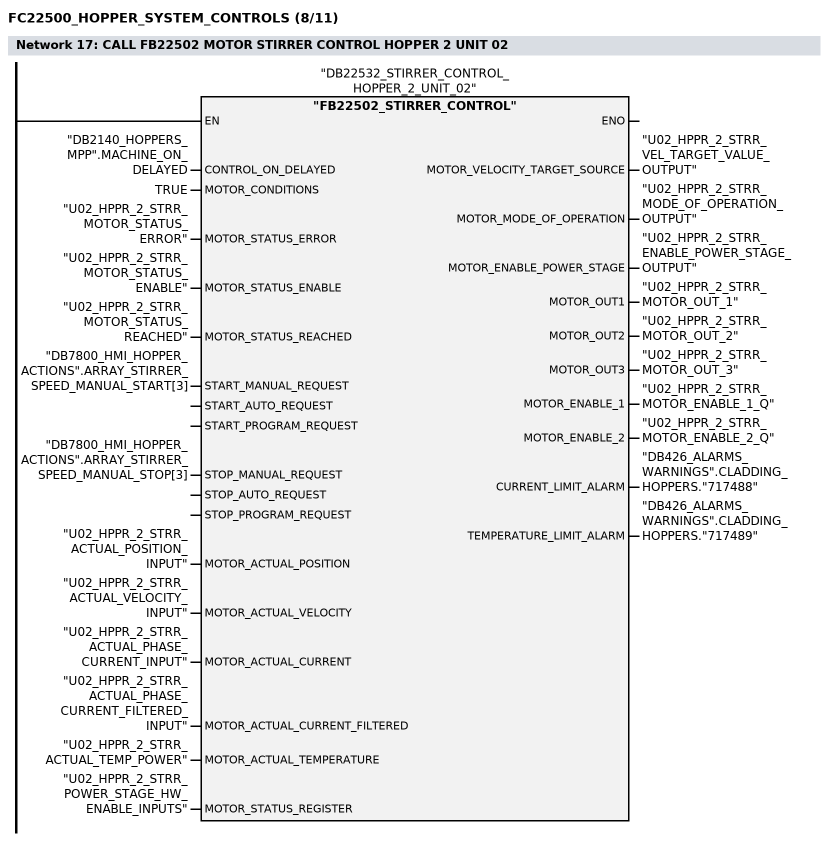
   RUNG wire#powerrail
      "DB22532_STIRRER_CONTROL_HOPPER_2_UNIT_02"(CONTROL_ON_DELAYED := "DB2140_HOPPERS_MPP".MACHINE_ON_DELAYED, MOTOR_CONDITIONS := TRUE, MOTOR_STATUS_ERROR := "U02_HPPR_2_STRR_MOTOR_STATUS_ERROR", MOTOR_STATUS_ENABLE := "U02_HPPR_2_STRR_MOTOR_STATUS_ENABLE", MOTOR_STATUS_REACHED := "U02_HPPR_2_STRR_MOTOR_STATUS_REACHED", START_MANUAL_REQUEST := "DB7800_HMI_HOPPER_ACTIONS".ARRAY_STIRRER_SPEED_MANUAL_START[3], START_AUTO_REQUEST :=, START_PROGRAM_REQUEST :=, STOP_MANUAL_REQUEST := "DB7800_HMI_HOPPER_ACTIONS".ARRAY_STIRRER_SPEED_MANUAL_STOP[3], STOP_AUTO_REQUEST :=, STOP_PROGRAM_REQUEST :=, MOTOR_ACTUAL_POSITION := "U02_HPPR_2_STRR_ACTUAL_POSITION_INPUT", MOTOR_ACTUAL_VELOCITY := "U02_HPPR_2_STRR_ACTUAL_VELOCITY_INPUT", MOTOR_ACTUAL_CURRENT := "U02_HPPR_2_STRR_ACTUAL_PHASE_CURRENT_INPUT", MOTOR_ACTUAL_CURRENT_FILTERED := "U02_HPPR_2_STRR_ACTUAL_PHASE_CURRENT_FILTERED_INPUT", MOTOR_ACTUAL_TEMPERATURE := "U02_HPPR_2_STRR_ACTUAL_TEMP_POWER", MOTOR_STATUS_REGISTER := "U02_HPPR_2_STRR_POWER_STAGE_HW_ENABLE_INPUTS", MOTOR_VELOCITY_TARGET_SOURCE => "U02_HPPR_2_STRR_VEL_TARGET_VALUE_OUTPUT", MOTOR_MODE_OF_OPERATION => "U02_HPPR_2_STRR_MODE_OF_OPERATION_OUTPUT", MOTOR_ENABLE_POWER_STAGE => "U02_HPPR_2_STRR_ENABLE_POWER_STAGE_OUTPUT", MOTOR_OUT1 => "U02_HPPR_2_STRR_MOTOR_OUT_1", MOTOR_OUT2 => "U02_HPPR_2_STRR_MOTOR_OUT_2", MOTOR_OUT3 => "U02_HPPR_2_STRR_MOTOR_OUT_3", MOTOR_ENABLE_1 => "U02_HPPR_2_STRR_MOTOR_ENABLE_1_Q", MOTOR_ENABLE_2 => "U02_HPPR_2_STRR_MOTOR_ENABLE_2_Q", CURRENT_LIMIT_ALARM => "DB426_ALARMS_WARNINGS".CLADDING_HOPPERS."717488", TEMPERATURE_LIMIT_ALARM => "DB426_ALARMS_WARNINGS".CLADDING_HOPPERS."717489")
   END_RUNG
   // the same network as SCL:
   "DB22532_STIRRER_CONTROL_HOPPER_2_UNIT_02"(CONTROL_ON_DELAYED := "DB2140_HOPPERS_MPP".MACHINE_ON_DELAYED,   // "FB22502_STIRRER_CONTROL"
                           MOTOR_CONDITIONS := TRUE,
                           MOTOR_STATUS_ERROR := "U02_HPPR_2_STRR_MOTOR_STATUS_ERROR",
                           MOTOR_STATUS_ENABLE := "U02_HPPR_2_STRR_MOTOR_STATUS_ENABLE",
                           MOTOR_STATUS_REACHED := "U02_HPPR_2_STRR_MOTOR_STATUS_REACHED",
                           START_MANUAL_REQUEST := "DB7800_HMI_HOPPER_ACTIONS".ARRAY_STIRRER_SPEED_MANUAL_START[3],
                           STOP_MANUAL_REQUEST := "DB7800_HMI_HOPPER_ACTIONS".ARRAY_STIRRER_SPEED_MANUAL_STOP[3],
                           MOTOR_ACTUAL_POSITION := "U02_HPPR_2_STRR_ACTUAL_POSITION_INPUT",
                           MOTOR_ACTUAL_VELOCITY := "U02_HPPR_2_STRR_ACTUAL_VELOCITY_INPUT",
                           MOTOR_ACTUAL_CURRENT := "U02_HPPR_2_STRR_ACTUAL_PHASE_CURRENT_INPUT",
                           MOTOR_ACTUAL_CURRENT_FILTERED := "U02_HPPR_2_STRR_ACTUAL_PHASE_CURRENT_FILTERED_INPUT",
                           MOTOR_ACTUAL_TEMPERATURE := "U02_HPPR_2_STRR_ACTUAL_TEMP_POWER",
                           MOTOR_STATUS_REGISTER := "U02_HPPR_2_STRR_POWER_STAGE_HW_ENABLE_INPUTS",
                           MOTOR_VELOCITY_TARGET_SOURCE => "U02_HPPR_2_STRR_VEL_TARGET_VALUE_OUTPUT",
                           MOTOR_MODE_OF_OPERATION => "U02_HPPR_2_STRR_MODE_OF_OPERATION_OUTPUT",
                           MOTOR_ENABLE_POWER_STAGE => "U02_HPPR_2_STRR_ENABLE_POWER_STAGE_OUTPUT",
                           MOTOR_OUT1 => "U02_HPPR_2_STRR_MOTOR_OUT_1",
                           MOTOR_OUT2 => "U02_HPPR_2_STRR_MOTOR_OUT_2",
                           MOTOR_OUT3 => "U02_HPPR_2_STRR_MOTOR_OUT_3",
                           MOTOR_ENABLE_1 => "U02_HPPR_2_STRR_MOTOR_ENABLE_1_Q",
                           MOTOR_ENABLE_2 => "U02_HPPR_2_STRR_MOTOR_ENABLE_2_Q",
                           CURRENT_LIMIT_ALARM => "DB426_ALARMS_WARNINGS".CLADDING_HOPPERS."717488",
                           TEMPERATURE_LIMIT_ALARM => "DB426_ALARMS_WARNINGS".CLADDING_HOPPERS."717489");
END_REGION

REGION Network 18: CALL FB22503 HOPPER PRESSURE CONTROL HOPPER 2 UNIT 02
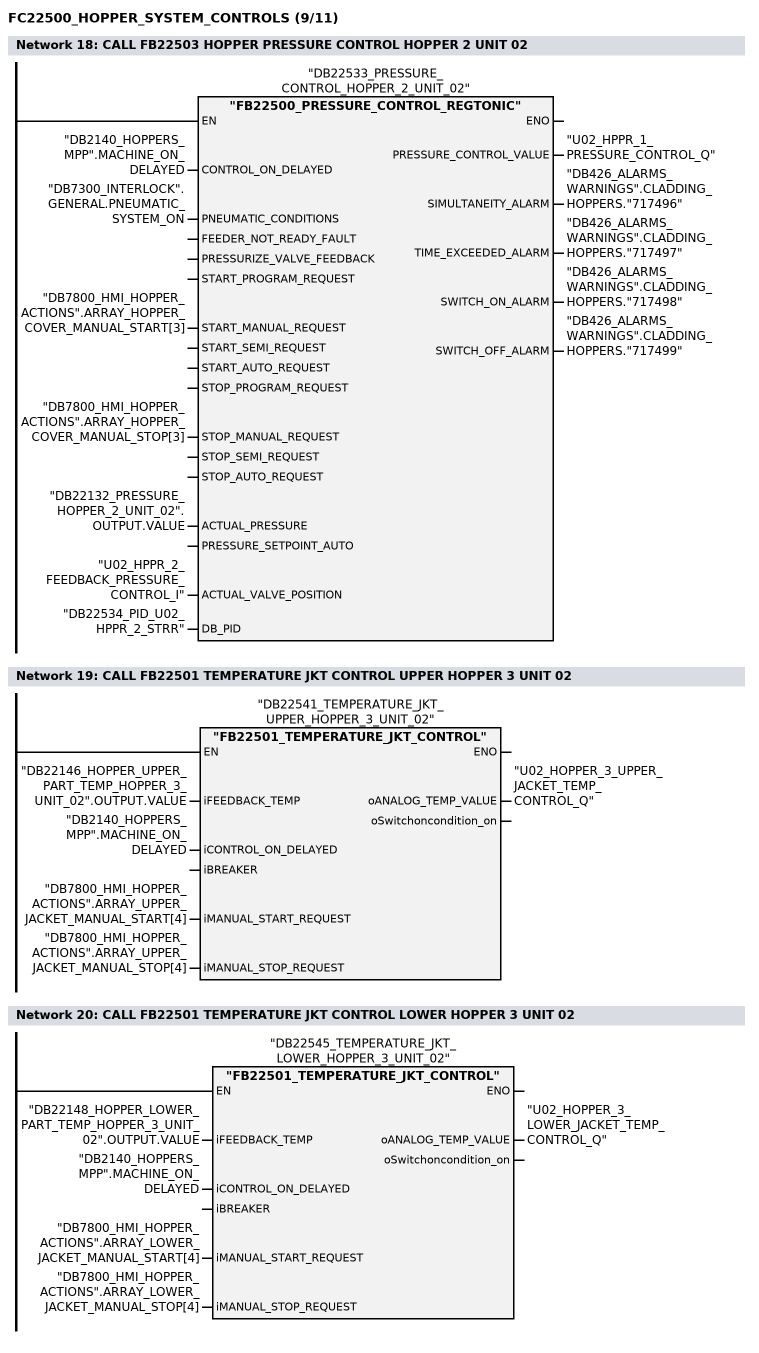
   RUNG wire#powerrail
      "DB22533_PRESSURE_CONTROL_HOPPER_2_UNIT_02"(CONTROL_ON_DELAYED := "DB2140_HOPPERS_MPP".MACHINE_ON_DELAYED, PNEUMATIC_CONDITIONS := "DB7300_INTERLOCK".GENERAL.PNEUMATIC_SYSTEM_ON, FEEDER_NOT_READY_FAULT :=, PRESSURIZE_VALVE_FEEDBACK :=, START_PROGRAM_REQUEST :=, START_MANUAL_REQUEST := "DB7800_HMI_HOPPER_ACTIONS".ARRAY_HOPPER_COVER_MANUAL_START[3], START_SEMI_REQUEST :=, START_AUTO_REQUEST :=, STOP_PROGRAM_REQUEST :=, STOP_MANUAL_REQUEST := "DB7800_HMI_HOPPER_ACTIONS".ARRAY_HOPPER_COVER_MANUAL_STOP[3], STOP_SEMI_REQUEST :=, STOP_AUTO_REQUEST :=, ACTUAL_PRESSURE := "DB22132_PRESSURE_HOPPER_2_UNIT_02".OUTPUT.VALUE, PRESSURE_SETPOINT_AUTO :=, ACTUAL_VALVE_POSITION := "U02_HPPR_2_FEEDBACK_PRESSURE_CONTROL_I", DB_PID := "DB22534_PID_U02_HPPR_2_STRR", PRESSURE_CONTROL_VALUE => "U02_HPPR_1_PRESSURE_CONTROL_Q", SIMULTANEITY_ALARM => "DB426_ALARMS_WARNINGS".CLADDING_HOPPERS."717496", TIME_EXCEEDED_ALARM => "DB426_ALARMS_WARNINGS".CLADDING_HOPPERS."717497", SWITCH_ON_ALARM => "DB426_ALARMS_WARNINGS".CLADDING_HOPPERS."717498", SWITCH_OFF_ALARM => "DB426_ALARMS_WARNINGS".CLADDING_HOPPERS."717499")
   END_RUNG
   // the same network as SCL:
   "DB22533_PRESSURE_CONTROL_HOPPER_2_UNIT_02"(CONTROL_ON_DELAYED := "DB2140_HOPPERS_MPP".MACHINE_ON_DELAYED,   // "FB22500_PRESSURE_CONTROL_REGTONIC"
                           PNEUMATIC_CONDITIONS := "DB7300_INTERLOCK".GENERAL.PNEUMATIC_SYSTEM_ON,
                           START_MANUAL_REQUEST := "DB7800_HMI_HOPPER_ACTIONS".ARRAY_HOPPER_COVER_MANUAL_START[3],
                           STOP_MANUAL_REQUEST := "DB7800_HMI_HOPPER_ACTIONS".ARRAY_HOPPER_COVER_MANUAL_STOP[3],
                           ACTUAL_PRESSURE := "DB22132_PRESSURE_HOPPER_2_UNIT_02".OUTPUT.VALUE,
                           ACTUAL_VALVE_POSITION := "U02_HPPR_2_FEEDBACK_PRESSURE_CONTROL_I",
                           DB_PID := "DB22534_PID_U02_HPPR_2_STRR",
                           PRESSURE_CONTROL_VALUE => "U02_HPPR_1_PRESSURE_CONTROL_Q",
                           SIMULTANEITY_ALARM => "DB426_ALARMS_WARNINGS".CLADDING_HOPPERS."717496",
                           TIME_EXCEEDED_ALARM => "DB426_ALARMS_WARNINGS".CLADDING_HOPPERS."717497",
                           SWITCH_ON_ALARM => "DB426_ALARMS_WARNINGS".CLADDING_HOPPERS."717498",
                           SWITCH_OFF_ALARM => "DB426_ALARMS_WARNINGS".CLADDING_HOPPERS."717499");
END_REGION

REGION Network 19: CALL FB22501 TEMPERATURE JKT CONTROL UPPER HOPPER 3 UNIT 02
   RUNG wire#powerrail
      "DB22541_TEMPERATURE_JKT_UPPER_HOPPER_3_UNIT_02"(iFEEDBACK_TEMP := "DB22146_HOPPER_UPPER_PART_TEMP_HOPPER_3_UNIT_02".OUTPUT.VALUE, iCONTROL_ON_DELAYED := "DB2140_HOPPERS_MPP".MACHINE_ON_DELAYED, iBREAKER :=, iMANUAL_START_REQUEST := "DB7800_HMI_HOPPER_ACTIONS".ARRAY_UPPER_JACKET_MANUAL_START[4], iMANUAL_STOP_REQUEST := "DB7800_HMI_HOPPER_ACTIONS".ARRAY_UPPER_JACKET_MANUAL_STOP[4], oANALOG_TEMP_VALUE => "U02_HOPPER_3_UPPER_JACKET_TEMP_CONTROL_Q", oSwitchoncondition_on =>)
   END_RUNG
   // the same network as SCL:
   "DB22541_TEMPERATURE_JKT_UPPER_HOPPER_3_UNIT_02"(iFEEDBACK_TEMP := "DB22146_HOPPER_UPPER_PART_TEMP_HOPPER_3_UNIT_02".OUTPUT.VALUE,   // "FB22501_TEMPERATURE_JKT_CONTROL"
                           iCONTROL_ON_DELAYED := "DB2140_HOPPERS_MPP".MACHINE_ON_DELAYED,
                           iMANUAL_START_REQUEST := "DB7800_HMI_HOPPER_ACTIONS".ARRAY_UPPER_JACKET_MANUAL_START[4],
                           iMANUAL_STOP_REQUEST := "DB7800_HMI_HOPPER_ACTIONS".ARRAY_UPPER_JACKET_MANUAL_STOP[4],
                           oANALOG_TEMP_VALUE => "U02_HOPPER_3_UPPER_JACKET_TEMP_CONTROL_Q");
END_REGION

REGION Network 20: CALL FB22501 TEMPERATURE JKT CONTROL LOWER HOPPER 3 UNIT 02
   RUNG wire#powerrail
      "DB22545_TEMPERATURE_JKT_LOWER_HOPPER_3_UNIT_02"(iFEEDBACK_TEMP := "DB22148_HOPPER_LOWER_PART_TEMP_HOPPER_3_UNIT_02".OUTPUT.VALUE, iCONTROL_ON_DELAYED := "DB2140_HOPPERS_MPP".MACHINE_ON_DELAYED, iBREAKER :=, iMANUAL_START_REQUEST := "DB7800_HMI_HOPPER_ACTIONS".ARRAY_LOWER_JACKET_MANUAL_START[4], iMANUAL_STOP_REQUEST := "DB7800_HMI_HOPPER_ACTIONS".ARRAY_LOWER_JACKET_MANUAL_STOP[4], oANALOG_TEMP_VALUE => "U02_HOPPER_3_LOWER_JACKET_TEMP_CONTROL_Q", oSwitchoncondition_on =>)
   END_RUNG
   // the same network as SCL:
   "DB22545_TEMPERATURE_JKT_LOWER_HOPPER_3_UNIT_02"(iFEEDBACK_TEMP := "DB22148_HOPPER_LOWER_PART_TEMP_HOPPER_3_UNIT_02".OUTPUT.VALUE,   // "FB22501_TEMPERATURE_JKT_CONTROL"
                           iCONTROL_ON_DELAYED := "DB2140_HOPPERS_MPP".MACHINE_ON_DELAYED,
                           iMANUAL_START_REQUEST := "DB7800_HMI_HOPPER_ACTIONS".ARRAY_LOWER_JACKET_MANUAL_START[4],
                           iMANUAL_STOP_REQUEST := "DB7800_HMI_HOPPER_ACTIONS".ARRAY_LOWER_JACKET_MANUAL_STOP[4],
                           oANALOG_TEMP_VALUE => "U02_HOPPER_3_LOWER_JACKET_TEMP_CONTROL_Q");
END_REGION

REGION Network 21: CALL FB22502 MOTOR STIRRER CONTROL HOPPER 3 UNIT 02
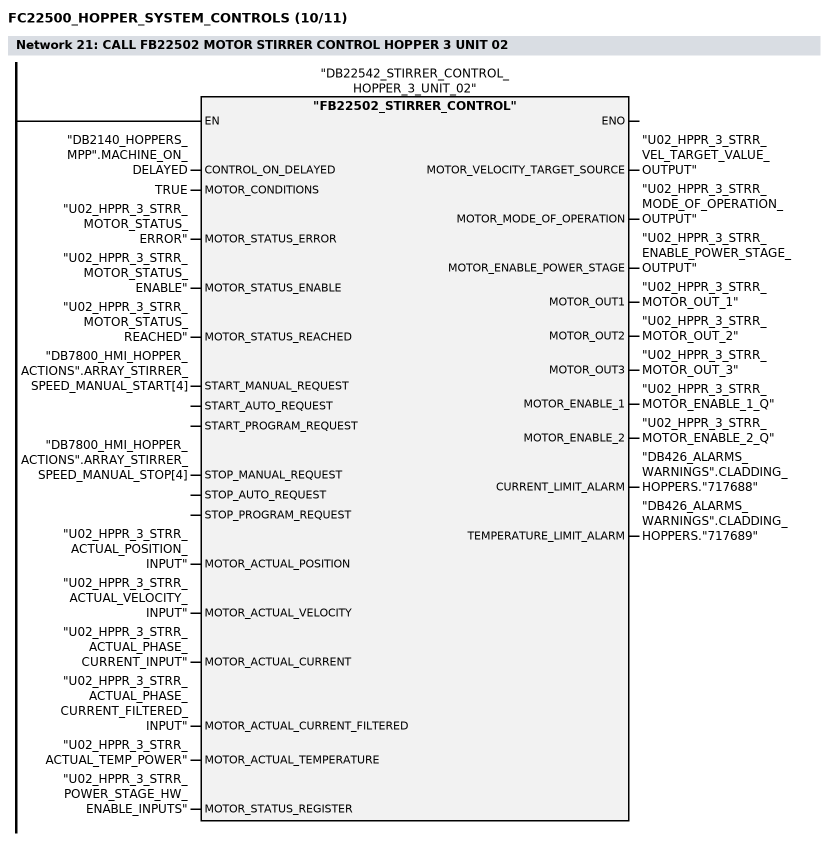
   RUNG wire#powerrail
      "DB22542_STIRRER_CONTROL_HOPPER_3_UNIT_02"(CONTROL_ON_DELAYED := "DB2140_HOPPERS_MPP".MACHINE_ON_DELAYED, MOTOR_CONDITIONS := TRUE, MOTOR_STATUS_ERROR := "U02_HPPR_3_STRR_MOTOR_STATUS_ERROR", MOTOR_STATUS_ENABLE := "U02_HPPR_3_STRR_MOTOR_STATUS_ENABLE", MOTOR_STATUS_REACHED := "U02_HPPR_3_STRR_MOTOR_STATUS_REACHED", START_MANUAL_REQUEST := "DB7800_HMI_HOPPER_ACTIONS".ARRAY_STIRRER_SPEED_MANUAL_START[4], START_AUTO_REQUEST :=, START_PROGRAM_REQUEST :=, STOP_MANUAL_REQUEST := "DB7800_HMI_HOPPER_ACTIONS".ARRAY_STIRRER_SPEED_MANUAL_STOP[4], STOP_AUTO_REQUEST :=, STOP_PROGRAM_REQUEST :=, MOTOR_ACTUAL_POSITION := "U02_HPPR_3_STRR_ACTUAL_POSITION_INPUT", MOTOR_ACTUAL_VELOCITY := "U02_HPPR_3_STRR_ACTUAL_VELOCITY_INPUT", MOTOR_ACTUAL_CURRENT := "U02_HPPR_3_STRR_ACTUAL_PHASE_CURRENT_INPUT", MOTOR_ACTUAL_CURRENT_FILTERED := "U02_HPPR_3_STRR_ACTUAL_PHASE_CURRENT_FILTERED_INPUT", MOTOR_ACTUAL_TEMPERATURE := "U02_HPPR_3_STRR_ACTUAL_TEMP_POWER", MOTOR_STATUS_REGISTER := "U02_HPPR_3_STRR_POWER_STAGE_HW_ENABLE_INPUTS", MOTOR_VELOCITY_TARGET_SOURCE => "U02_HPPR_3_STRR_VEL_TARGET_VALUE_OUTPUT", MOTOR_MODE_OF_OPERATION => "U02_HPPR_3_STRR_MODE_OF_OPERATION_OUTPUT", MOTOR_ENABLE_POWER_STAGE => "U02_HPPR_3_STRR_ENABLE_POWER_STAGE_OUTPUT", MOTOR_OUT1 => "U02_HPPR_3_STRR_MOTOR_OUT_1", MOTOR_OUT2 => "U02_HPPR_3_STRR_MOTOR_OUT_2", MOTOR_OUT3 => "U02_HPPR_3_STRR_MOTOR_OUT_3", MOTOR_ENABLE_1 => "U02_HPPR_3_STRR_MOTOR_ENABLE_1_Q", MOTOR_ENABLE_2 => "U02_HPPR_3_STRR_MOTOR_ENABLE_2_Q", CURRENT_LIMIT_ALARM => "DB426_ALARMS_WARNINGS".CLADDING_HOPPERS."717688", TEMPERATURE_LIMIT_ALARM => "DB426_ALARMS_WARNINGS".CLADDING_HOPPERS."717689")
   END_RUNG
   // the same network as SCL:
   "DB22542_STIRRER_CONTROL_HOPPER_3_UNIT_02"(CONTROL_ON_DELAYED := "DB2140_HOPPERS_MPP".MACHINE_ON_DELAYED,   // "FB22502_STIRRER_CONTROL"
                           MOTOR_CONDITIONS := TRUE,
                           MOTOR_STATUS_ERROR := "U02_HPPR_3_STRR_MOTOR_STATUS_ERROR",
                           MOTOR_STATUS_ENABLE := "U02_HPPR_3_STRR_MOTOR_STATUS_ENABLE",
                           MOTOR_STATUS_REACHED := "U02_HPPR_3_STRR_MOTOR_STATUS_REACHED",
                           START_MANUAL_REQUEST := "DB7800_HMI_HOPPER_ACTIONS".ARRAY_STIRRER_SPEED_MANUAL_START[4],
                           STOP_MANUAL_REQUEST := "DB7800_HMI_HOPPER_ACTIONS".ARRAY_STIRRER_SPEED_MANUAL_STOP[4],
                           MOTOR_ACTUAL_POSITION := "U02_HPPR_3_STRR_ACTUAL_POSITION_INPUT",
                           MOTOR_ACTUAL_VELOCITY := "U02_HPPR_3_STRR_ACTUAL_VELOCITY_INPUT",
                           MOTOR_ACTUAL_CURRENT := "U02_HPPR_3_STRR_ACTUAL_PHASE_CURRENT_INPUT",
                           MOTOR_ACTUAL_CURRENT_FILTERED := "U02_HPPR_3_STRR_ACTUAL_PHASE_CURRENT_FILTERED_INPUT",
                           MOTOR_ACTUAL_TEMPERATURE := "U02_HPPR_3_STRR_ACTUAL_TEMP_POWER",
                           MOTOR_STATUS_REGISTER := "U02_HPPR_3_STRR_POWER_STAGE_HW_ENABLE_INPUTS",
                           MOTOR_VELOCITY_TARGET_SOURCE => "U02_HPPR_3_STRR_VEL_TARGET_VALUE_OUTPUT",
                           MOTOR_MODE_OF_OPERATION => "U02_HPPR_3_STRR_MODE_OF_OPERATION_OUTPUT",
                           MOTOR_ENABLE_POWER_STAGE => "U02_HPPR_3_STRR_ENABLE_POWER_STAGE_OUTPUT",
                           MOTOR_OUT1 => "U02_HPPR_3_STRR_MOTOR_OUT_1",
                           MOTOR_OUT2 => "U02_HPPR_3_STRR_MOTOR_OUT_2",
                           MOTOR_OUT3 => "U02_HPPR_3_STRR_MOTOR_OUT_3",
                           MOTOR_ENABLE_1 => "U02_HPPR_3_STRR_MOTOR_ENABLE_1_Q",
                           MOTOR_ENABLE_2 => "U02_HPPR_3_STRR_MOTOR_ENABLE_2_Q",
                           CURRENT_LIMIT_ALARM => "DB426_ALARMS_WARNINGS".CLADDING_HOPPERS."717688",
                           TEMPERATURE_LIMIT_ALARM => "DB426_ALARMS_WARNINGS".CLADDING_HOPPERS."717689");
END_REGION

REGION Network 22: CALL FB22503 HOPPER PRESSURE CONTROL HOPPER 3 UNIT 02
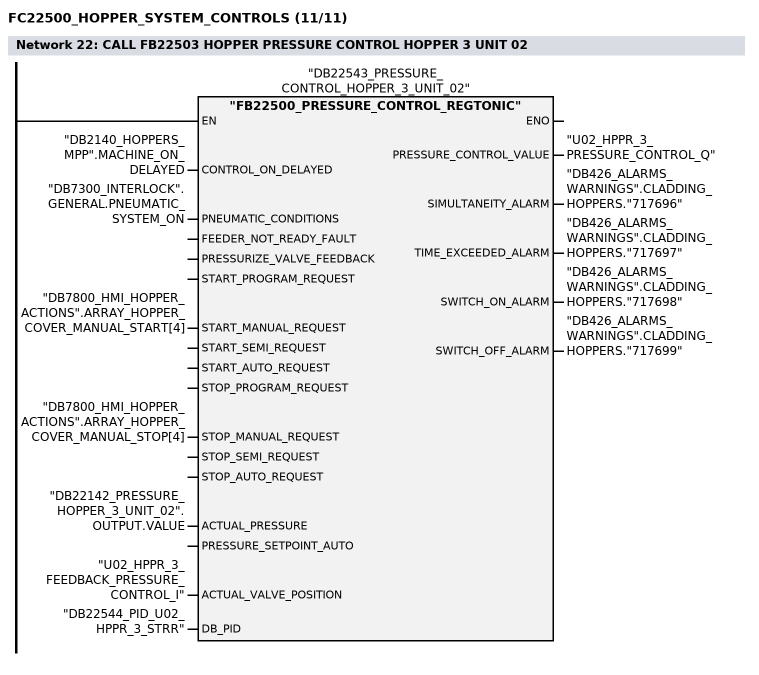
   RUNG wire#powerrail
      "DB22543_PRESSURE_CONTROL_HOPPER_3_UNIT_02"(CONTROL_ON_DELAYED := "DB2140_HOPPERS_MPP".MACHINE_ON_DELAYED, PNEUMATIC_CONDITIONS := "DB7300_INTERLOCK".GENERAL.PNEUMATIC_SYSTEM_ON, FEEDER_NOT_READY_FAULT :=, PRESSURIZE_VALVE_FEEDBACK :=, START_PROGRAM_REQUEST :=, START_MANUAL_REQUEST := "DB7800_HMI_HOPPER_ACTIONS".ARRAY_HOPPER_COVER_MANUAL_START[4], START_SEMI_REQUEST :=, START_AUTO_REQUEST :=, STOP_PROGRAM_REQUEST :=, STOP_MANUAL_REQUEST := "DB7800_HMI_HOPPER_ACTIONS".ARRAY_HOPPER_COVER_MANUAL_STOP[4], STOP_SEMI_REQUEST :=, STOP_AUTO_REQUEST :=, ACTUAL_PRESSURE := "DB22142_PRESSURE_HOPPER_3_UNIT_02".OUTPUT.VALUE, PRESSURE_SETPOINT_AUTO :=, ACTUAL_VALVE_POSITION := "U02_HPPR_3_FEEDBACK_PRESSURE_CONTROL_I", DB_PID := "DB22544_PID_U02_HPPR_3_STRR", PRESSURE_CONTROL_VALUE => "U02_HPPR_3_PRESSURE_CONTROL_Q", SIMULTANEITY_ALARM => "DB426_ALARMS_WARNINGS".CLADDING_HOPPERS."717696", TIME_EXCEEDED_ALARM => "DB426_ALARMS_WARNINGS".CLADDING_HOPPERS."717697", SWITCH_ON_ALARM => "DB426_ALARMS_WARNINGS".CLADDING_HOPPERS."717698", SWITCH_OFF_ALARM => "DB426_ALARMS_WARNINGS".CLADDING_HOPPERS."717699")
   END_RUNG
   // the same network as SCL:
   "DB22543_PRESSURE_CONTROL_HOPPER_3_UNIT_02"(CONTROL_ON_DELAYED := "DB2140_HOPPERS_MPP".MACHINE_ON_DELAYED,   // "FB22500_PRESSURE_CONTROL_REGTONIC"
                           PNEUMATIC_CONDITIONS := "DB7300_INTERLOCK".GENERAL.PNEUMATIC_SYSTEM_ON,
                           START_MANUAL_REQUEST := "DB7800_HMI_HOPPER_ACTIONS".ARRAY_HOPPER_COVER_MANUAL_START[4],
                           STOP_MANUAL_REQUEST := "DB7800_HMI_HOPPER_ACTIONS".ARRAY_HOPPER_COVER_MANUAL_STOP[4],
                           ACTUAL_PRESSURE := "DB22142_PRESSURE_HOPPER_3_UNIT_02".OUTPUT.VALUE,
                           ACTUAL_VALVE_POSITION := "U02_HPPR_3_FEEDBACK_PRESSURE_CONTROL_I",
                           DB_PID := "DB22544_PID_U02_HPPR_3_STRR",
                           PRESSURE_CONTROL_VALUE => "U02_HPPR_3_PRESSURE_CONTROL_Q",
                           SIMULTANEITY_ALARM => "DB426_ALARMS_WARNINGS".CLADDING_HOPPERS."717696",
                           TIME_EXCEEDED_ALARM => "DB426_ALARMS_WARNINGS".CLADDING_HOPPERS."717697",
                           SWITCH_ON_ALARM => "DB426_ALARMS_WARNINGS".CLADDING_HOPPERS."717698",
                           SWITCH_OFF_ALARM => "DB426_ALARMS_WARNINGS".CLADDING_HOPPERS."717699");
END_REGION
END_FUNCTION

FUNCTION "FC22700_HOPPER_SEQUENCE_COORDINATOR" : Void   // FC22700, LAD
TITLE = FC22700 HOPPER SEQUENCE COORDINATOR
{ S7_Optimized_Access := 'TRUE' }
VERSION : 0.1
// stored: AutoNumber false, IsIECCheckEnabled false, SetENOAutomatically false, UDAEnableTagReadback false
BEGIN

REGION Network 1: CALL FC22701 LOAD FEEDER SEQUENCES
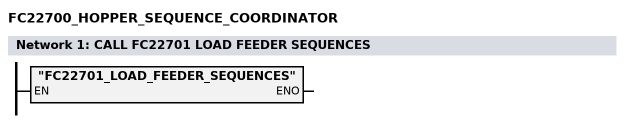
   RUNG wire#powerrail
      "FC22701_LOAD_FEEDER_SEQUENCES"()
   END_RUNG
   // the same network as SCL:
   "FC22701_LOAD_FEEDER_SEQUENCES"();
END_REGION
END_FUNCTION

FUNCTION "FC22701_LOAD_FEEDER_SEQUENCES" : Void   // FC22701, LAD
TITLE = FC22701 LOAD FEEDER SEQUENCES
{ S7_Optimized_Access := 'TRUE' }
VERSION : 0.1
// stored: AutoNumber false, IsIECCheckEnabled false, SetENOAutomatically false, UDAEnableTagReadback false
BEGIN

REGION Network 1: //////////_UNIT_01_//////////
END_REGION

REGION Network 2: /////_HOPPER_1_SEQUENCES_/////
END_REGION

REGION Network 3: CALL FB22701 LOAD FEEDER SEQUENCE TIME UNIT 01 HOPPER 1
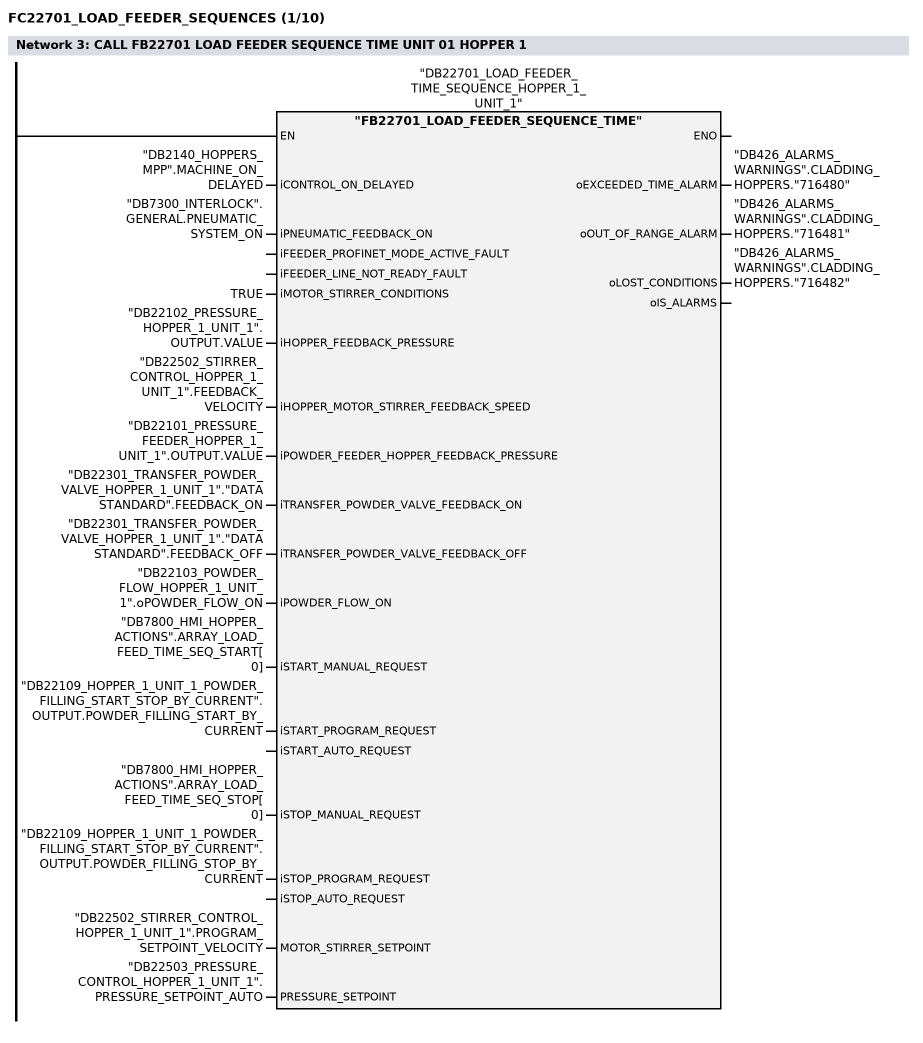
   RUNG wire#powerrail
      "DB22701_LOAD_FEEDER_TIME_SEQUENCE_HOPPER_1_UNIT_1"(iCONTROL_ON_DELAYED := "DB2140_HOPPERS_MPP".MACHINE_ON_DELAYED, iPNEUMATIC_FEEDBACK_ON := "DB7300_INTERLOCK".GENERAL.PNEUMATIC_SYSTEM_ON, iFEEDER_PROFINET_MODE_ACTIVE_FAULT :=, iFEEDER_LINE_NOT_READY_FAULT :=, iMOTOR_STIRRER_CONDITIONS := TRUE, iHOPPER_FEEDBACK_PRESSURE := "DB22102_PRESSURE_HOPPER_1_UNIT_1".OUTPUT.VALUE, iHOPPER_MOTOR_STIRRER_FEEDBACK_SPEED := "DB22502_STIRRER_CONTROL_HOPPER_1_UNIT_1".FEEDBACK_VELOCITY, iPOWDER_FEEDER_HOPPER_FEEDBACK_PRESSURE := "DB22101_PRESSURE_FEEDER_HOPPER_1_UNIT_1".OUTPUT.VALUE, iTRANSFER_POWDER_VALVE_FEEDBACK_ON := "DB22301_TRANSFER_POWDER_VALVE_HOPPER_1_UNIT_1"."DATA STANDARD".FEEDBACK_ON, iTRANSFER_POWDER_VALVE_FEEDBACK_OFF := "DB22301_TRANSFER_POWDER_VALVE_HOPPER_1_UNIT_1"."DATA STANDARD".FEEDBACK_OFF, iPOWDER_FLOW_ON := "DB22103_POWDER_FLOW_HOPPER_1_UNIT_1".oPOWDER_FLOW_ON, iSTART_MANUAL_REQUEST := "DB7800_HMI_HOPPER_ACTIONS".ARRAY_LOAD_FEED_TIME_SEQ_START[0], iSTART_PROGRAM_REQUEST := "DB22109_HOPPER_1_UNIT_1_POWDER_FILLING_START_STOP_BY_CURRENT".OUTPUT.POWDER_FILLING_START_BY_CURRENT, iSTART_AUTO_REQUEST :=, iSTOP_MANUAL_REQUEST := "DB7800_HMI_HOPPER_ACTIONS".ARRAY_LOAD_FEED_TIME_SEQ_STOP[0], iSTOP_PROGRAM_REQUEST := "DB22109_HOPPER_1_UNIT_1_POWDER_FILLING_START_STOP_BY_CURRENT".OUTPUT.POWDER_FILLING_STOP_BY_CURRENT, iSTOP_AUTO_REQUEST :=, MOTOR_STIRRER_SETPOINT := "DB22502_STIRRER_CONTROL_HOPPER_1_UNIT_1".PROGRAM_SETPOINT_VELOCITY, PRESSURE_SETPOINT := "DB22503_PRESSURE_CONTROL_HOPPER_1_UNIT_1".PRESSURE_SETPOINT_AUTO, oEXCEEDED_TIME_ALARM => "DB426_ALARMS_WARNINGS".CLADDING_HOPPERS."716480", oOUT_OF_RANGE_ALARM => "DB426_ALARMS_WARNINGS".CLADDING_HOPPERS."716481", oLOST_CONDITIONS => "DB426_ALARMS_WARNINGS".CLADDING_HOPPERS."716482", oIS_ALARMS =>)
   END_RUNG
   // the same network as SCL:
   "DB22701_LOAD_FEEDER_TIME_SEQUENCE_HOPPER_1_UNIT_1"(iCONTROL_ON_DELAYED := "DB2140_HOPPERS_MPP".MACHINE_ON_DELAYED,   // "FB22701_LOAD_FEEDER_SEQUENCE_TIME"
                           iPNEUMATIC_FEEDBACK_ON := "DB7300_INTERLOCK".GENERAL.PNEUMATIC_SYSTEM_ON,
                           iMOTOR_STIRRER_CONDITIONS := TRUE,
                           iHOPPER_FEEDBACK_PRESSURE := "DB22102_PRESSURE_HOPPER_1_UNIT_1".OUTPUT.VALUE,
                           iHOPPER_MOTOR_STIRRER_FEEDBACK_SPEED := "DB22502_STIRRER_CONTROL_HOPPER_1_UNIT_1".FEEDBACK_VELOCITY,
                           iPOWDER_FEEDER_HOPPER_FEEDBACK_PRESSURE := "DB22101_PRESSURE_FEEDER_HOPPER_1_UNIT_1".OUTPUT.VALUE,
                           iTRANSFER_POWDER_VALVE_FEEDBACK_ON := "DB22301_TRANSFER_POWDER_VALVE_HOPPER_1_UNIT_1"."DATA STANDARD".FEEDBACK_ON,
                           iTRANSFER_POWDER_VALVE_FEEDBACK_OFF := "DB22301_TRANSFER_POWDER_VALVE_HOPPER_1_UNIT_1"."DATA STANDARD".FEEDBACK_OFF,
                           iPOWDER_FLOW_ON := "DB22103_POWDER_FLOW_HOPPER_1_UNIT_1".oPOWDER_FLOW_ON,
                           iSTART_MANUAL_REQUEST := "DB7800_HMI_HOPPER_ACTIONS".ARRAY_LOAD_FEED_TIME_SEQ_START[0],
                           iSTART_PROGRAM_REQUEST := "DB22109_HOPPER_1_UNIT_1_POWDER_FILLING_START_STOP_BY_CURRENT".OUTPUT.POWDER_FILLING_START_BY_CURRENT,
                           iSTOP_MANUAL_REQUEST := "DB7800_HMI_HOPPER_ACTIONS".ARRAY_LOAD_FEED_TIME_SEQ_STOP[0],
                           iSTOP_PROGRAM_REQUEST := "DB22109_HOPPER_1_UNIT_1_POWDER_FILLING_START_STOP_BY_CURRENT".OUTPUT.POWDER_FILLING_STOP_BY_CURRENT,
                           MOTOR_STIRRER_SETPOINT := "DB22502_STIRRER_CONTROL_HOPPER_1_UNIT_1".PROGRAM_SETPOINT_VELOCITY,
                           PRESSURE_SETPOINT := "DB22503_PRESSURE_CONTROL_HOPPER_1_UNIT_1".PRESSURE_SETPOINT_AUTO,
                           oEXCEEDED_TIME_ALARM => "DB426_ALARMS_WARNINGS".CLADDING_HOPPERS."716480",
                           oOUT_OF_RANGE_ALARM => "DB426_ALARMS_WARNINGS".CLADDING_HOPPERS."716481",
                           oLOST_CONDITIONS => "DB426_ALARMS_WARNINGS".CLADDING_HOPPERS."716482");
END_REGION

REGION Network 4: CALL FB22702 LOAD FEEDER SEQUENCE WEIGHT UNIT 01 HOPPER 1
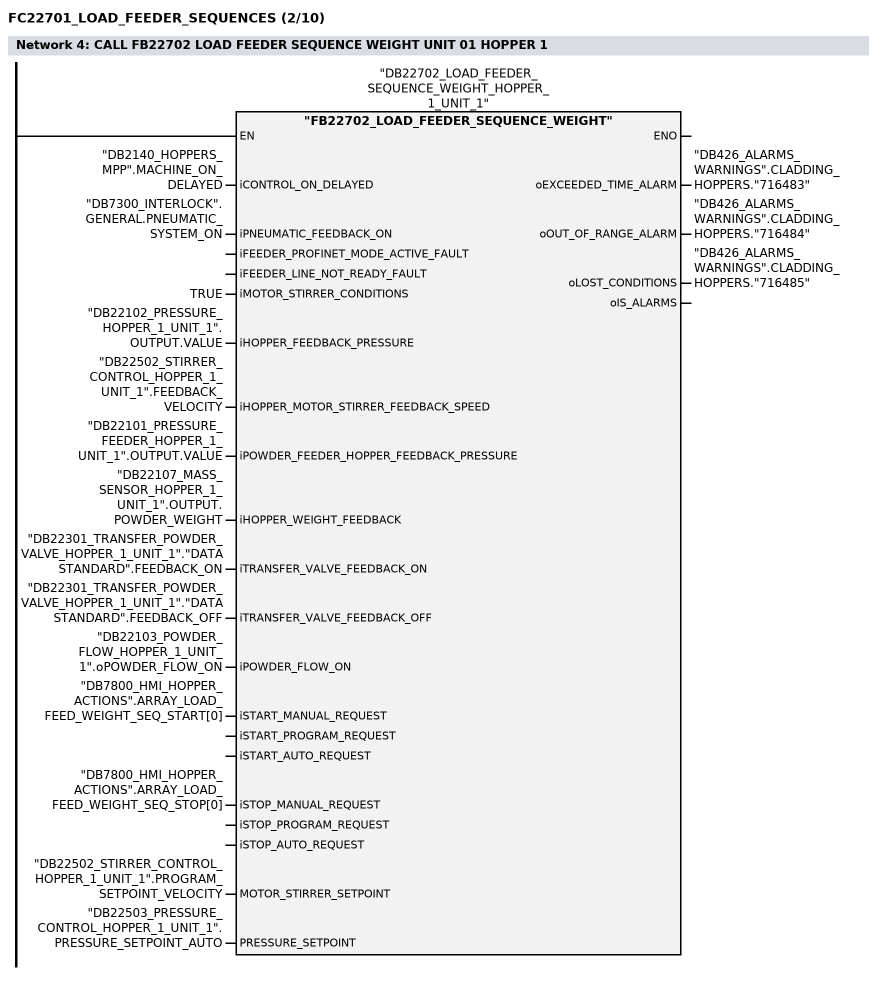
   RUNG wire#powerrail
      "DB22702_LOAD_FEEDER_SEQUENCE_WEIGHT_HOPPER_1_UNIT_1"(iCONTROL_ON_DELAYED := "DB2140_HOPPERS_MPP".MACHINE_ON_DELAYED, iPNEUMATIC_FEEDBACK_ON := "DB7300_INTERLOCK".GENERAL.PNEUMATIC_SYSTEM_ON, iFEEDER_PROFINET_MODE_ACTIVE_FAULT :=, iFEEDER_LINE_NOT_READY_FAULT :=, iMOTOR_STIRRER_CONDITIONS := TRUE, iHOPPER_FEEDBACK_PRESSURE := "DB22102_PRESSURE_HOPPER_1_UNIT_1".OUTPUT.VALUE, iHOPPER_MOTOR_STIRRER_FEEDBACK_SPEED := "DB22502_STIRRER_CONTROL_HOPPER_1_UNIT_1".FEEDBACK_VELOCITY, iPOWDER_FEEDER_HOPPER_FEEDBACK_PRESSURE := "DB22101_PRESSURE_FEEDER_HOPPER_1_UNIT_1".OUTPUT.VALUE, iHOPPER_WEIGHT_FEEDBACK := "DB22107_MASS_SENSOR_HOPPER_1_UNIT_1".OUTPUT.POWDER_WEIGHT, iTRANSFER_VALVE_FEEDBACK_ON := "DB22301_TRANSFER_POWDER_VALVE_HOPPER_1_UNIT_1"."DATA STANDARD".FEEDBACK_ON, iTRANSFER_VALVE_FEEDBACK_OFF := "DB22301_TRANSFER_POWDER_VALVE_HOPPER_1_UNIT_1"."DATA STANDARD".FEEDBACK_OFF, iPOWDER_FLOW_ON := "DB22103_POWDER_FLOW_HOPPER_1_UNIT_1".oPOWDER_FLOW_ON, iSTART_MANUAL_REQUEST := "DB7800_HMI_HOPPER_ACTIONS".ARRAY_LOAD_FEED_WEIGHT_SEQ_START[0], iSTART_PROGRAM_REQUEST :=, iSTART_AUTO_REQUEST :=, iSTOP_MANUAL_REQUEST := "DB7800_HMI_HOPPER_ACTIONS".ARRAY_LOAD_FEED_WEIGHT_SEQ_STOP[0], iSTOP_PROGRAM_REQUEST :=, iSTOP_AUTO_REQUEST :=, MOTOR_STIRRER_SETPOINT := "DB22502_STIRRER_CONTROL_HOPPER_1_UNIT_1".PROGRAM_SETPOINT_VELOCITY, PRESSURE_SETPOINT := "DB22503_PRESSURE_CONTROL_HOPPER_1_UNIT_1".PRESSURE_SETPOINT_AUTO, oEXCEEDED_TIME_ALARM => "DB426_ALARMS_WARNINGS".CLADDING_HOPPERS."716483", oOUT_OF_RANGE_ALARM => "DB426_ALARMS_WARNINGS".CLADDING_HOPPERS."716484", oLOST_CONDITIONS => "DB426_ALARMS_WARNINGS".CLADDING_HOPPERS."716485", oIS_ALARMS =>)
   END_RUNG
   // the same network as SCL:
   "DB22702_LOAD_FEEDER_SEQUENCE_WEIGHT_HOPPER_1_UNIT_1"(iCONTROL_ON_DELAYED := "DB2140_HOPPERS_MPP".MACHINE_ON_DELAYED,   // "FB22702_LOAD_FEEDER_SEQUENCE_WEIGHT"
                           iPNEUMATIC_FEEDBACK_ON := "DB7300_INTERLOCK".GENERAL.PNEUMATIC_SYSTEM_ON,
                           iMOTOR_STIRRER_CONDITIONS := TRUE,
                           iHOPPER_FEEDBACK_PRESSURE := "DB22102_PRESSURE_HOPPER_1_UNIT_1".OUTPUT.VALUE,
                           iHOPPER_MOTOR_STIRRER_FEEDBACK_SPEED := "DB22502_STIRRER_CONTROL_HOPPER_1_UNIT_1".FEEDBACK_VELOCITY,
                           iPOWDER_FEEDER_HOPPER_FEEDBACK_PRESSURE := "DB22101_PRESSURE_FEEDER_HOPPER_1_UNIT_1".OUTPUT.VALUE,
                           iHOPPER_WEIGHT_FEEDBACK := "DB22107_MASS_SENSOR_HOPPER_1_UNIT_1".OUTPUT.POWDER_WEIGHT,
                           iTRANSFER_VALVE_FEEDBACK_ON := "DB22301_TRANSFER_POWDER_VALVE_HOPPER_1_UNIT_1"."DATA STANDARD".FEEDBACK_ON,
                           iTRANSFER_VALVE_FEEDBACK_OFF := "DB22301_TRANSFER_POWDER_VALVE_HOPPER_1_UNIT_1"."DATA STANDARD".FEEDBACK_OFF,
                           iPOWDER_FLOW_ON := "DB22103_POWDER_FLOW_HOPPER_1_UNIT_1".oPOWDER_FLOW_ON,
                           iSTART_MANUAL_REQUEST := "DB7800_HMI_HOPPER_ACTIONS".ARRAY_LOAD_FEED_WEIGHT_SEQ_START[0],
                           iSTOP_MANUAL_REQUEST := "DB7800_HMI_HOPPER_ACTIONS".ARRAY_LOAD_FEED_WEIGHT_SEQ_STOP[0],
                           MOTOR_STIRRER_SETPOINT := "DB22502_STIRRER_CONTROL_HOPPER_1_UNIT_1".PROGRAM_SETPOINT_VELOCITY,
                           PRESSURE_SETPOINT := "DB22503_PRESSURE_CONTROL_HOPPER_1_UNIT_1".PRESSURE_SETPOINT_AUTO,
                           oEXCEEDED_TIME_ALARM => "DB426_ALARMS_WARNINGS".CLADDING_HOPPERS."716483",
                           oOUT_OF_RANGE_ALARM => "DB426_ALARMS_WARNINGS".CLADDING_HOPPERS."716484",
                           oLOST_CONDITIONS => "DB426_ALARMS_WARNINGS".CLADDING_HOPPERS."716485");
END_REGION

REGION Network 5: /////_HOPPER_2_SEQUENCES_/////
END_REGION

REGION Network 6: CALL FB22701 LOAD FEEDER SEQUENCE TIME UNIT 01 HOPPER 2
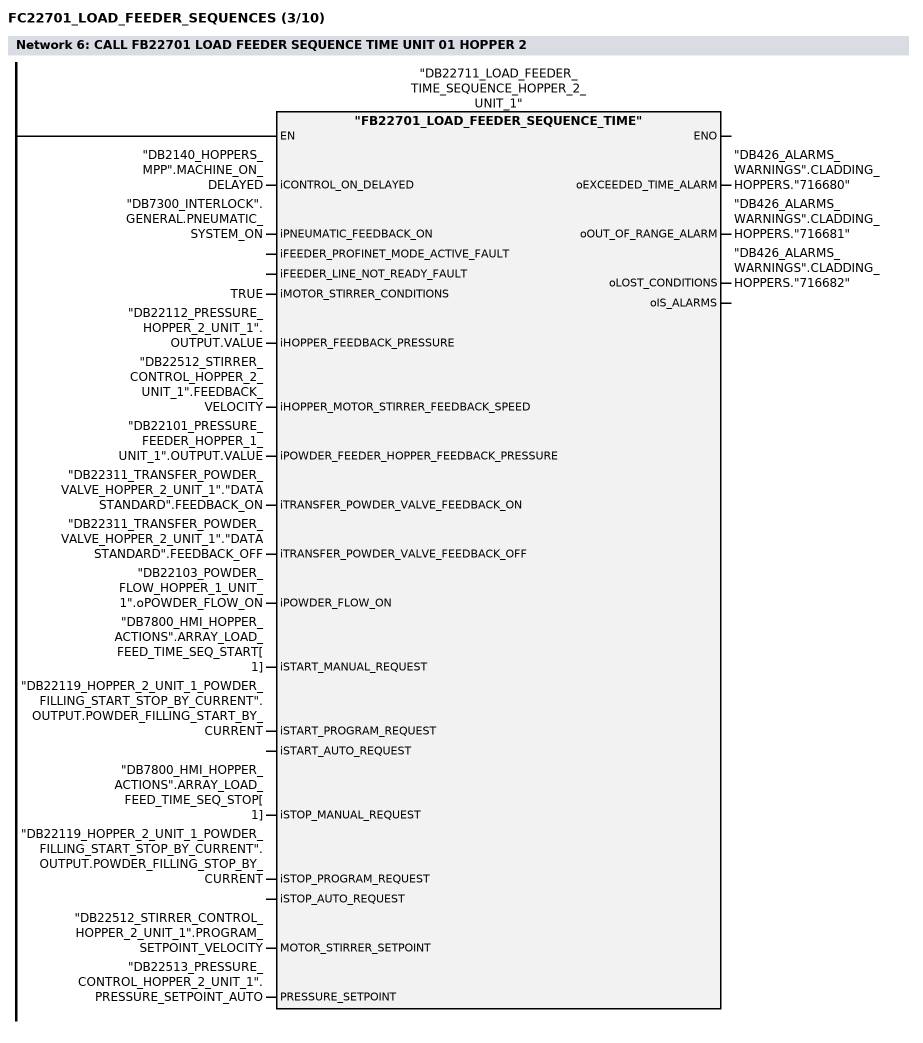
   RUNG wire#powerrail
      "DB22711_LOAD_FEEDER_TIME_SEQUENCE_HOPPER_2_UNIT_1"(iCONTROL_ON_DELAYED := "DB2140_HOPPERS_MPP".MACHINE_ON_DELAYED, iPNEUMATIC_FEEDBACK_ON := "DB7300_INTERLOCK".GENERAL.PNEUMATIC_SYSTEM_ON, iFEEDER_PROFINET_MODE_ACTIVE_FAULT :=, iFEEDER_LINE_NOT_READY_FAULT :=, iMOTOR_STIRRER_CONDITIONS := TRUE, iHOPPER_FEEDBACK_PRESSURE := "DB22112_PRESSURE_HOPPER_2_UNIT_1".OUTPUT.VALUE, iHOPPER_MOTOR_STIRRER_FEEDBACK_SPEED := "DB22512_STIRRER_CONTROL_HOPPER_2_UNIT_1".FEEDBACK_VELOCITY, iPOWDER_FEEDER_HOPPER_FEEDBACK_PRESSURE := "DB22101_PRESSURE_FEEDER_HOPPER_1_UNIT_1".OUTPUT.VALUE, iTRANSFER_POWDER_VALVE_FEEDBACK_ON := "DB22311_TRANSFER_POWDER_VALVE_HOPPER_2_UNIT_1"."DATA STANDARD".FEEDBACK_ON, iTRANSFER_POWDER_VALVE_FEEDBACK_OFF := "DB22311_TRANSFER_POWDER_VALVE_HOPPER_2_UNIT_1"."DATA STANDARD".FEEDBACK_OFF, iPOWDER_FLOW_ON := "DB22103_POWDER_FLOW_HOPPER_1_UNIT_1".oPOWDER_FLOW_ON, iSTART_MANUAL_REQUEST := "DB7800_HMI_HOPPER_ACTIONS".ARRAY_LOAD_FEED_TIME_SEQ_START[1], iSTART_PROGRAM_REQUEST := "DB22119_HOPPER_2_UNIT_1_POWDER_FILLING_START_STOP_BY_CURRENT".OUTPUT.POWDER_FILLING_START_BY_CURRENT, iSTART_AUTO_REQUEST :=, iSTOP_MANUAL_REQUEST := "DB7800_HMI_HOPPER_ACTIONS".ARRAY_LOAD_FEED_TIME_SEQ_STOP[1], iSTOP_PROGRAM_REQUEST := "DB22119_HOPPER_2_UNIT_1_POWDER_FILLING_START_STOP_BY_CURRENT".OUTPUT.POWDER_FILLING_STOP_BY_CURRENT, iSTOP_AUTO_REQUEST :=, MOTOR_STIRRER_SETPOINT := "DB22512_STIRRER_CONTROL_HOPPER_2_UNIT_1".PROGRAM_SETPOINT_VELOCITY, PRESSURE_SETPOINT := "DB22513_PRESSURE_CONTROL_HOPPER_2_UNIT_1".PRESSURE_SETPOINT_AUTO, oEXCEEDED_TIME_ALARM => "DB426_ALARMS_WARNINGS".CLADDING_HOPPERS."716680", oOUT_OF_RANGE_ALARM => "DB426_ALARMS_WARNINGS".CLADDING_HOPPERS."716681", oLOST_CONDITIONS => "DB426_ALARMS_WARNINGS".CLADDING_HOPPERS."716682", oIS_ALARMS =>)
   END_RUNG
   // the same network as SCL:
   "DB22711_LOAD_FEEDER_TIME_SEQUENCE_HOPPER_2_UNIT_1"(iCONTROL_ON_DELAYED := "DB2140_HOPPERS_MPP".MACHINE_ON_DELAYED,   // "FB22701_LOAD_FEEDER_SEQUENCE_TIME"
                           iPNEUMATIC_FEEDBACK_ON := "DB7300_INTERLOCK".GENERAL.PNEUMATIC_SYSTEM_ON,
                           iMOTOR_STIRRER_CONDITIONS := TRUE,
                           iHOPPER_FEEDBACK_PRESSURE := "DB22112_PRESSURE_HOPPER_2_UNIT_1".OUTPUT.VALUE,
                           iHOPPER_MOTOR_STIRRER_FEEDBACK_SPEED := "DB22512_STIRRER_CONTROL_HOPPER_2_UNIT_1".FEEDBACK_VELOCITY,
                           iPOWDER_FEEDER_HOPPER_FEEDBACK_PRESSURE := "DB22101_PRESSURE_FEEDER_HOPPER_1_UNIT_1".OUTPUT.VALUE,
                           iTRANSFER_POWDER_VALVE_FEEDBACK_ON := "DB22311_TRANSFER_POWDER_VALVE_HOPPER_2_UNIT_1"."DATA STANDARD".FEEDBACK_ON,
                           iTRANSFER_POWDER_VALVE_FEEDBACK_OFF := "DB22311_TRANSFER_POWDER_VALVE_HOPPER_2_UNIT_1"."DATA STANDARD".FEEDBACK_OFF,
                           iPOWDER_FLOW_ON := "DB22103_POWDER_FLOW_HOPPER_1_UNIT_1".oPOWDER_FLOW_ON,
                           iSTART_MANUAL_REQUEST := "DB7800_HMI_HOPPER_ACTIONS".ARRAY_LOAD_FEED_TIME_SEQ_START[1],
                           iSTART_PROGRAM_REQUEST := "DB22119_HOPPER_2_UNIT_1_POWDER_FILLING_START_STOP_BY_CURRENT".OUTPUT.POWDER_FILLING_START_BY_CURRENT,
                           iSTOP_MANUAL_REQUEST := "DB7800_HMI_HOPPER_ACTIONS".ARRAY_LOAD_FEED_TIME_SEQ_STOP[1],
                           iSTOP_PROGRAM_REQUEST := "DB22119_HOPPER_2_UNIT_1_POWDER_FILLING_START_STOP_BY_CURRENT".OUTPUT.POWDER_FILLING_STOP_BY_CURRENT,
                           MOTOR_STIRRER_SETPOINT := "DB22512_STIRRER_CONTROL_HOPPER_2_UNIT_1".PROGRAM_SETPOINT_VELOCITY,
                           PRESSURE_SETPOINT := "DB22513_PRESSURE_CONTROL_HOPPER_2_UNIT_1".PRESSURE_SETPOINT_AUTO,
                           oEXCEEDED_TIME_ALARM => "DB426_ALARMS_WARNINGS".CLADDING_HOPPERS."716680",
                           oOUT_OF_RANGE_ALARM => "DB426_ALARMS_WARNINGS".CLADDING_HOPPERS."716681",
                           oLOST_CONDITIONS => "DB426_ALARMS_WARNINGS".CLADDING_HOPPERS."716682");
END_REGION

REGION Network 7: CALL FB22702 LOAD FEEDER SEQUENCE WEIGHT UNIT 01 HOPPER 2
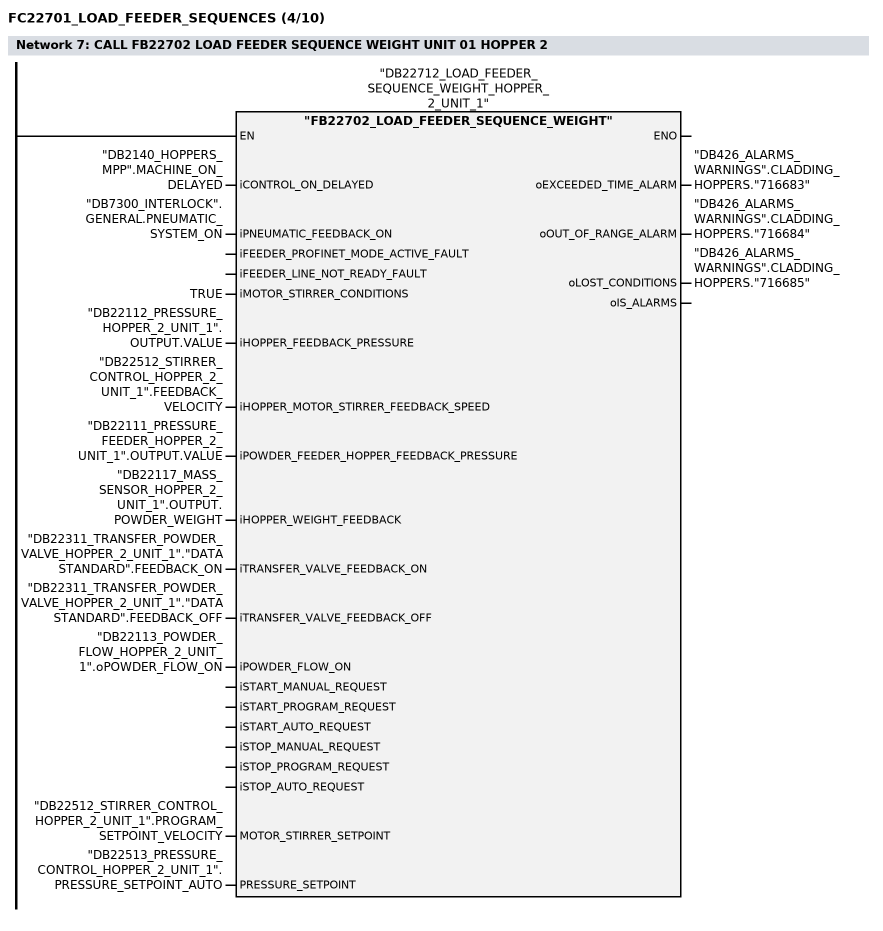
   RUNG wire#powerrail
      "DB22712_LOAD_FEEDER_SEQUENCE_WEIGHT_HOPPER_2_UNIT_1"(iCONTROL_ON_DELAYED := "DB2140_HOPPERS_MPP".MACHINE_ON_DELAYED, iPNEUMATIC_FEEDBACK_ON := "DB7300_INTERLOCK".GENERAL.PNEUMATIC_SYSTEM_ON, iFEEDER_PROFINET_MODE_ACTIVE_FAULT :=, iFEEDER_LINE_NOT_READY_FAULT :=, iMOTOR_STIRRER_CONDITIONS := TRUE, iHOPPER_FEEDBACK_PRESSURE := "DB22112_PRESSURE_HOPPER_2_UNIT_1".OUTPUT.VALUE, iHOPPER_MOTOR_STIRRER_FEEDBACK_SPEED := "DB22512_STIRRER_CONTROL_HOPPER_2_UNIT_1".FEEDBACK_VELOCITY, iPOWDER_FEEDER_HOPPER_FEEDBACK_PRESSURE := "DB22111_PRESSURE_FEEDER_HOPPER_2_UNIT_1".OUTPUT.VALUE, iHOPPER_WEIGHT_FEEDBACK := "DB22117_MASS_SENSOR_HOPPER_2_UNIT_1".OUTPUT.POWDER_WEIGHT, iTRANSFER_VALVE_FEEDBACK_ON := "DB22311_TRANSFER_POWDER_VALVE_HOPPER_2_UNIT_1"."DATA STANDARD".FEEDBACK_ON, iTRANSFER_VALVE_FEEDBACK_OFF := "DB22311_TRANSFER_POWDER_VALVE_HOPPER_2_UNIT_1"."DATA STANDARD".FEEDBACK_OFF, iPOWDER_FLOW_ON := "DB22113_POWDER_FLOW_HOPPER_2_UNIT_1".oPOWDER_FLOW_ON, iSTART_MANUAL_REQUEST :=, iSTART_AUTO_REQUEST :=, iSTOP_MANUAL_REQUEST :=, iSTOP_AUTO_REQUEST :=, MOTOR_STIRRER_SETPOINT := "DB22512_STIRRER_CONTROL_HOPPER_2_UNIT_1".PROGRAM_SETPOINT_VELOCITY, PRESSURE_SETPOINT := "DB22513_PRESSURE_CONTROL_HOPPER_2_UNIT_1".PRESSURE_SETPOINT_AUTO, oEXCEEDED_TIME_ALARM => "DB426_ALARMS_WARNINGS".CLADDING_HOPPERS."716683", oOUT_OF_RANGE_ALARM => "DB426_ALARMS_WARNINGS".CLADDING_HOPPERS."716684", oLOST_CONDITIONS => "DB426_ALARMS_WARNINGS".CLADDING_HOPPERS."716685", oIS_ALARMS =>, iSTART_PROGRAM_REQUEST :=, iSTOP_PROGRAM_REQUEST :=)
   END_RUNG
   // the same network as SCL:
   "DB22712_LOAD_FEEDER_SEQUENCE_WEIGHT_HOPPER_2_UNIT_1"(iCONTROL_ON_DELAYED := "DB2140_HOPPERS_MPP".MACHINE_ON_DELAYED,   // "FB22702_LOAD_FEEDER_SEQUENCE_WEIGHT"
                           iPNEUMATIC_FEEDBACK_ON := "DB7300_INTERLOCK".GENERAL.PNEUMATIC_SYSTEM_ON,
                           iMOTOR_STIRRER_CONDITIONS := TRUE,
                           iHOPPER_FEEDBACK_PRESSURE := "DB22112_PRESSURE_HOPPER_2_UNIT_1".OUTPUT.VALUE,
                           iHOPPER_MOTOR_STIRRER_FEEDBACK_SPEED := "DB22512_STIRRER_CONTROL_HOPPER_2_UNIT_1".FEEDBACK_VELOCITY,
                           iPOWDER_FEEDER_HOPPER_FEEDBACK_PRESSURE := "DB22111_PRESSURE_FEEDER_HOPPER_2_UNIT_1".OUTPUT.VALUE,
                           iHOPPER_WEIGHT_FEEDBACK := "DB22117_MASS_SENSOR_HOPPER_2_UNIT_1".OUTPUT.POWDER_WEIGHT,
                           iTRANSFER_VALVE_FEEDBACK_ON := "DB22311_TRANSFER_POWDER_VALVE_HOPPER_2_UNIT_1"."DATA STANDARD".FEEDBACK_ON,
                           iTRANSFER_VALVE_FEEDBACK_OFF := "DB22311_TRANSFER_POWDER_VALVE_HOPPER_2_UNIT_1"."DATA STANDARD".FEEDBACK_OFF,
                           iPOWDER_FLOW_ON := "DB22113_POWDER_FLOW_HOPPER_2_UNIT_1".oPOWDER_FLOW_ON,
                           MOTOR_STIRRER_SETPOINT := "DB22512_STIRRER_CONTROL_HOPPER_2_UNIT_1".PROGRAM_SETPOINT_VELOCITY,
                           PRESSURE_SETPOINT := "DB22513_PRESSURE_CONTROL_HOPPER_2_UNIT_1".PRESSURE_SETPOINT_AUTO,
                           oEXCEEDED_TIME_ALARM => "DB426_ALARMS_WARNINGS".CLADDING_HOPPERS."716683",
                           oOUT_OF_RANGE_ALARM => "DB426_ALARMS_WARNINGS".CLADDING_HOPPERS."716684",
                           oLOST_CONDITIONS => "DB426_ALARMS_WARNINGS".CLADDING_HOPPERS."716685");
END_REGION

REGION Network 8: //////////_UNIT_02_//////////
END_REGION

REGION Network 9: /////_HOPPER_1_SEQUENCES_/////
END_REGION

REGION Network 10: CALL FB22701 LOAD FEEDER SEQUENCE TIME UNIT 02 HOPPER 1
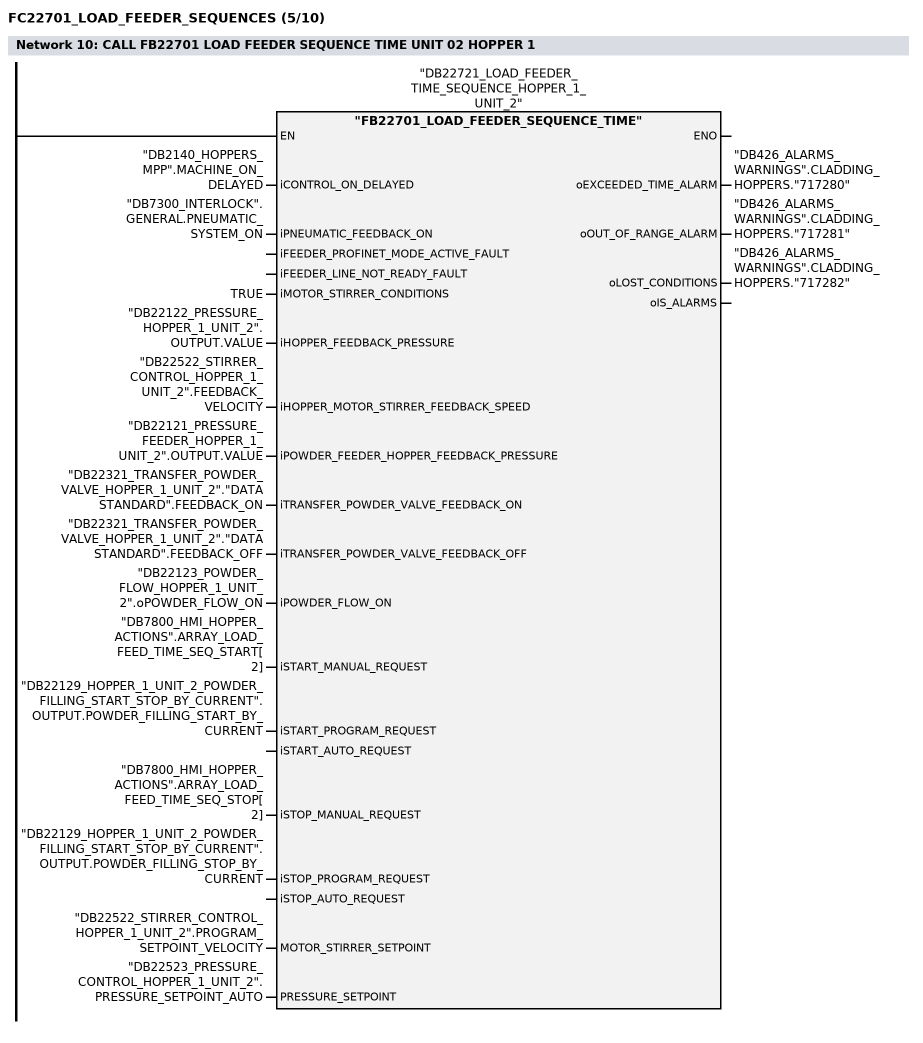
   RUNG wire#powerrail
      "DB22721_LOAD_FEEDER_TIME_SEQUENCE_HOPPER_1_UNIT_2"(iCONTROL_ON_DELAYED := "DB2140_HOPPERS_MPP".MACHINE_ON_DELAYED, iPNEUMATIC_FEEDBACK_ON := "DB7300_INTERLOCK".GENERAL.PNEUMATIC_SYSTEM_ON, iFEEDER_PROFINET_MODE_ACTIVE_FAULT :=, iFEEDER_LINE_NOT_READY_FAULT :=, iMOTOR_STIRRER_CONDITIONS := TRUE, iHOPPER_FEEDBACK_PRESSURE := "DB22122_PRESSURE_HOPPER_1_UNIT_2".OUTPUT.VALUE, iHOPPER_MOTOR_STIRRER_FEEDBACK_SPEED := "DB22522_STIRRER_CONTROL_HOPPER_1_UNIT_2".FEEDBACK_VELOCITY, iPOWDER_FEEDER_HOPPER_FEEDBACK_PRESSURE := "DB22121_PRESSURE_FEEDER_HOPPER_1_UNIT_2".OUTPUT.VALUE, iTRANSFER_POWDER_VALVE_FEEDBACK_ON := "DB22321_TRANSFER_POWDER_VALVE_HOPPER_1_UNIT_2"."DATA STANDARD".FEEDBACK_ON, iTRANSFER_POWDER_VALVE_FEEDBACK_OFF := "DB22321_TRANSFER_POWDER_VALVE_HOPPER_1_UNIT_2"."DATA STANDARD".FEEDBACK_OFF, iPOWDER_FLOW_ON := "DB22123_POWDER_FLOW_HOPPER_1_UNIT_2".oPOWDER_FLOW_ON, iSTART_MANUAL_REQUEST := "DB7800_HMI_HOPPER_ACTIONS".ARRAY_LOAD_FEED_TIME_SEQ_START[2], iSTART_PROGRAM_REQUEST := "DB22129_HOPPER_1_UNIT_2_POWDER_FILLING_START_STOP_BY_CURRENT".OUTPUT.POWDER_FILLING_START_BY_CURRENT, iSTART_AUTO_REQUEST :=, iSTOP_MANUAL_REQUEST := "DB7800_HMI_HOPPER_ACTIONS".ARRAY_LOAD_FEED_TIME_SEQ_STOP[2], iSTOP_PROGRAM_REQUEST := "DB22129_HOPPER_1_UNIT_2_POWDER_FILLING_START_STOP_BY_CURRENT".OUTPUT.POWDER_FILLING_STOP_BY_CURRENT, iSTOP_AUTO_REQUEST :=, MOTOR_STIRRER_SETPOINT := "DB22522_STIRRER_CONTROL_HOPPER_1_UNIT_2".PROGRAM_SETPOINT_VELOCITY, PRESSURE_SETPOINT := "DB22523_PRESSURE_CONTROL_HOPPER_1_UNIT_2".PRESSURE_SETPOINT_AUTO, oEXCEEDED_TIME_ALARM => "DB426_ALARMS_WARNINGS".CLADDING_HOPPERS."717280", oOUT_OF_RANGE_ALARM => "DB426_ALARMS_WARNINGS".CLADDING_HOPPERS."717281", oLOST_CONDITIONS => "DB426_ALARMS_WARNINGS".CLADDING_HOPPERS."717282", oIS_ALARMS =>)
   END_RUNG
   // the same network as SCL:
   "DB22721_LOAD_FEEDER_TIME_SEQUENCE_HOPPER_1_UNIT_2"(iCONTROL_ON_DELAYED := "DB2140_HOPPERS_MPP".MACHINE_ON_DELAYED,   // "FB22701_LOAD_FEEDER_SEQUENCE_TIME"
                           iPNEUMATIC_FEEDBACK_ON := "DB7300_INTERLOCK".GENERAL.PNEUMATIC_SYSTEM_ON,
                           iMOTOR_STIRRER_CONDITIONS := TRUE,
                           iHOPPER_FEEDBACK_PRESSURE := "DB22122_PRESSURE_HOPPER_1_UNIT_2".OUTPUT.VALUE,
                           iHOPPER_MOTOR_STIRRER_FEEDBACK_SPEED := "DB22522_STIRRER_CONTROL_HOPPER_1_UNIT_2".FEEDBACK_VELOCITY,
                           iPOWDER_FEEDER_HOPPER_FEEDBACK_PRESSURE := "DB22121_PRESSURE_FEEDER_HOPPER_1_UNIT_2".OUTPUT.VALUE,
                           iTRANSFER_POWDER_VALVE_FEEDBACK_ON := "DB22321_TRANSFER_POWDER_VALVE_HOPPER_1_UNIT_2"."DATA STANDARD".FEEDBACK_ON,
                           iTRANSFER_POWDER_VALVE_FEEDBACK_OFF := "DB22321_TRANSFER_POWDER_VALVE_HOPPER_1_UNIT_2"."DATA STANDARD".FEEDBACK_OFF,
                           iPOWDER_FLOW_ON := "DB22123_POWDER_FLOW_HOPPER_1_UNIT_2".oPOWDER_FLOW_ON,
                           iSTART_MANUAL_REQUEST := "DB7800_HMI_HOPPER_ACTIONS".ARRAY_LOAD_FEED_TIME_SEQ_START[2],
                           iSTART_PROGRAM_REQUEST := "DB22129_HOPPER_1_UNIT_2_POWDER_FILLING_START_STOP_BY_CURRENT".OUTPUT.POWDER_FILLING_START_BY_CURRENT,
                           iSTOP_MANUAL_REQUEST := "DB7800_HMI_HOPPER_ACTIONS".ARRAY_LOAD_FEED_TIME_SEQ_STOP[2],
                           iSTOP_PROGRAM_REQUEST := "DB22129_HOPPER_1_UNIT_2_POWDER_FILLING_START_STOP_BY_CURRENT".OUTPUT.POWDER_FILLING_STOP_BY_CURRENT,
                           MOTOR_STIRRER_SETPOINT := "DB22522_STIRRER_CONTROL_HOPPER_1_UNIT_2".PROGRAM_SETPOINT_VELOCITY,
                           PRESSURE_SETPOINT := "DB22523_PRESSURE_CONTROL_HOPPER_1_UNIT_2".PRESSURE_SETPOINT_AUTO,
                           oEXCEEDED_TIME_ALARM => "DB426_ALARMS_WARNINGS".CLADDING_HOPPERS."717280",
                           oOUT_OF_RANGE_ALARM => "DB426_ALARMS_WARNINGS".CLADDING_HOPPERS."717281",
                           oLOST_CONDITIONS => "DB426_ALARMS_WARNINGS".CLADDING_HOPPERS."717282");
END_REGION

REGION Network 11: CALL FB22702 LOAD FEEDER SEQUENCE WEIGHT UNIT 02 HOPPER 1
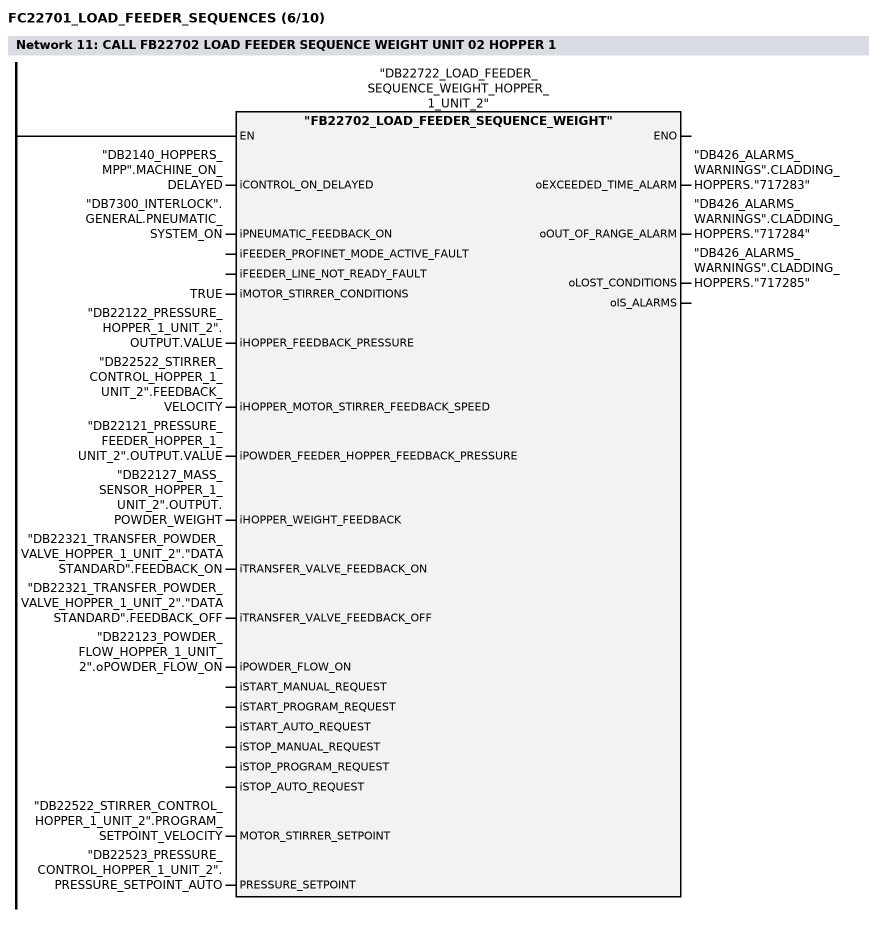
   RUNG wire#powerrail
      "DB22722_LOAD_FEEDER_SEQUENCE_WEIGHT_HOPPER_1_UNIT_2"(iCONTROL_ON_DELAYED := "DB2140_HOPPERS_MPP".MACHINE_ON_DELAYED, iPNEUMATIC_FEEDBACK_ON := "DB7300_INTERLOCK".GENERAL.PNEUMATIC_SYSTEM_ON, iFEEDER_PROFINET_MODE_ACTIVE_FAULT :=, iFEEDER_LINE_NOT_READY_FAULT :=, iMOTOR_STIRRER_CONDITIONS := TRUE, iHOPPER_FEEDBACK_PRESSURE := "DB22122_PRESSURE_HOPPER_1_UNIT_2".OUTPUT.VALUE, iHOPPER_MOTOR_STIRRER_FEEDBACK_SPEED := "DB22522_STIRRER_CONTROL_HOPPER_1_UNIT_2".FEEDBACK_VELOCITY, iPOWDER_FEEDER_HOPPER_FEEDBACK_PRESSURE := "DB22121_PRESSURE_FEEDER_HOPPER_1_UNIT_2".OUTPUT.VALUE, iHOPPER_WEIGHT_FEEDBACK := "DB22127_MASS_SENSOR_HOPPER_1_UNIT_2".OUTPUT.POWDER_WEIGHT, iTRANSFER_VALVE_FEEDBACK_ON := "DB22321_TRANSFER_POWDER_VALVE_HOPPER_1_UNIT_2"."DATA STANDARD".FEEDBACK_ON, iTRANSFER_VALVE_FEEDBACK_OFF := "DB22321_TRANSFER_POWDER_VALVE_HOPPER_1_UNIT_2"."DATA STANDARD".FEEDBACK_OFF, iPOWDER_FLOW_ON := "DB22123_POWDER_FLOW_HOPPER_1_UNIT_2".oPOWDER_FLOW_ON, iSTART_MANUAL_REQUEST :=, iSTART_AUTO_REQUEST :=, iSTOP_MANUAL_REQUEST :=, iSTOP_AUTO_REQUEST :=, MOTOR_STIRRER_SETPOINT := "DB22522_STIRRER_CONTROL_HOPPER_1_UNIT_2".PROGRAM_SETPOINT_VELOCITY, PRESSURE_SETPOINT := "DB22523_PRESSURE_CONTROL_HOPPER_1_UNIT_2".PRESSURE_SETPOINT_AUTO, oEXCEEDED_TIME_ALARM => "DB426_ALARMS_WARNINGS".CLADDING_HOPPERS."717283", oOUT_OF_RANGE_ALARM => "DB426_ALARMS_WARNINGS".CLADDING_HOPPERS."717284", oLOST_CONDITIONS => "DB426_ALARMS_WARNINGS".CLADDING_HOPPERS."717285", oIS_ALARMS =>, iSTART_PROGRAM_REQUEST :=, iSTOP_PROGRAM_REQUEST :=)
   END_RUNG
   // the same network as SCL:
   "DB22722_LOAD_FEEDER_SEQUENCE_WEIGHT_HOPPER_1_UNIT_2"(iCONTROL_ON_DELAYED := "DB2140_HOPPERS_MPP".MACHINE_ON_DELAYED,   // "FB22702_LOAD_FEEDER_SEQUENCE_WEIGHT"
                           iPNEUMATIC_FEEDBACK_ON := "DB7300_INTERLOCK".GENERAL.PNEUMATIC_SYSTEM_ON,
                           iMOTOR_STIRRER_CONDITIONS := TRUE,
                           iHOPPER_FEEDBACK_PRESSURE := "DB22122_PRESSURE_HOPPER_1_UNIT_2".OUTPUT.VALUE,
                           iHOPPER_MOTOR_STIRRER_FEEDBACK_SPEED := "DB22522_STIRRER_CONTROL_HOPPER_1_UNIT_2".FEEDBACK_VELOCITY,
                           iPOWDER_FEEDER_HOPPER_FEEDBACK_PRESSURE := "DB22121_PRESSURE_FEEDER_HOPPER_1_UNIT_2".OUTPUT.VALUE,
                           iHOPPER_WEIGHT_FEEDBACK := "DB22127_MASS_SENSOR_HOPPER_1_UNIT_2".OUTPUT.POWDER_WEIGHT,
                           iTRANSFER_VALVE_FEEDBACK_ON := "DB22321_TRANSFER_POWDER_VALVE_HOPPER_1_UNIT_2"."DATA STANDARD".FEEDBACK_ON,
                           iTRANSFER_VALVE_FEEDBACK_OFF := "DB22321_TRANSFER_POWDER_VALVE_HOPPER_1_UNIT_2"."DATA STANDARD".FEEDBACK_OFF,
                           iPOWDER_FLOW_ON := "DB22123_POWDER_FLOW_HOPPER_1_UNIT_2".oPOWDER_FLOW_ON,
                           MOTOR_STIRRER_SETPOINT := "DB22522_STIRRER_CONTROL_HOPPER_1_UNIT_2".PROGRAM_SETPOINT_VELOCITY,
                           PRESSURE_SETPOINT := "DB22523_PRESSURE_CONTROL_HOPPER_1_UNIT_2".PRESSURE_SETPOINT_AUTO,
                           oEXCEEDED_TIME_ALARM => "DB426_ALARMS_WARNINGS".CLADDING_HOPPERS."717283",
                           oOUT_OF_RANGE_ALARM => "DB426_ALARMS_WARNINGS".CLADDING_HOPPERS."717284",
                           oLOST_CONDITIONS => "DB426_ALARMS_WARNINGS".CLADDING_HOPPERS."717285");
END_REGION

REGION Network 12: /////_HOPPER_2_SEQUENCES_/////
END_REGION

REGION Network 13: CALL FB22701 LOAD FEEDER SEQUENCE TIME UNIT 02 HOPPER 2
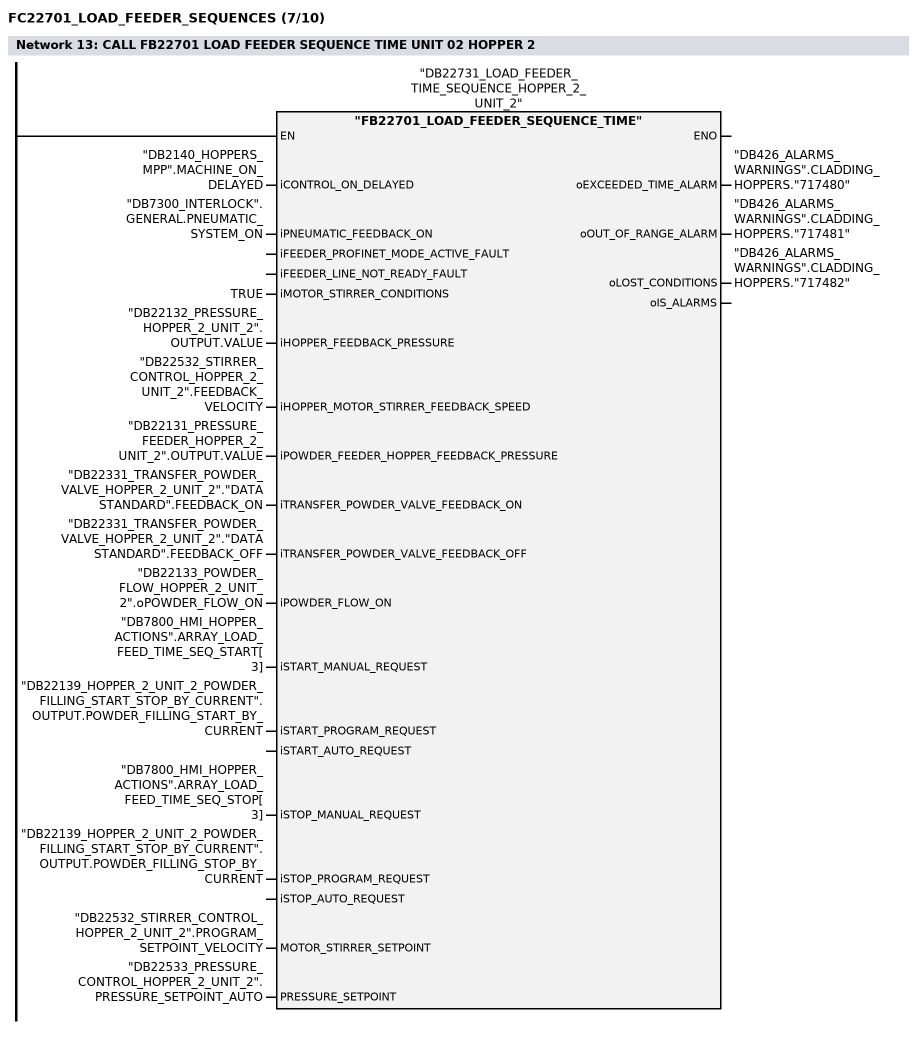
   RUNG wire#powerrail
      "DB22731_LOAD_FEEDER_TIME_SEQUENCE_HOPPER_2_UNIT_2"(iCONTROL_ON_DELAYED := "DB2140_HOPPERS_MPP".MACHINE_ON_DELAYED, iPNEUMATIC_FEEDBACK_ON := "DB7300_INTERLOCK".GENERAL.PNEUMATIC_SYSTEM_ON, iFEEDER_PROFINET_MODE_ACTIVE_FAULT :=, iFEEDER_LINE_NOT_READY_FAULT :=, iMOTOR_STIRRER_CONDITIONS := TRUE, iHOPPER_FEEDBACK_PRESSURE := "DB22132_PRESSURE_HOPPER_2_UNIT_2".OUTPUT.VALUE, iHOPPER_MOTOR_STIRRER_FEEDBACK_SPEED := "DB22532_STIRRER_CONTROL_HOPPER_2_UNIT_2".FEEDBACK_VELOCITY, iPOWDER_FEEDER_HOPPER_FEEDBACK_PRESSURE := "DB22131_PRESSURE_FEEDER_HOPPER_2_UNIT_2".OUTPUT.VALUE, iTRANSFER_POWDER_VALVE_FEEDBACK_ON := "DB22331_TRANSFER_POWDER_VALVE_HOPPER_2_UNIT_2"."DATA STANDARD".FEEDBACK_ON, iTRANSFER_POWDER_VALVE_FEEDBACK_OFF := "DB22331_TRANSFER_POWDER_VALVE_HOPPER_2_UNIT_2"."DATA STANDARD".FEEDBACK_OFF, iPOWDER_FLOW_ON := "DB22133_POWDER_FLOW_HOPPER_2_UNIT_2".oPOWDER_FLOW_ON, iSTART_MANUAL_REQUEST := "DB7800_HMI_HOPPER_ACTIONS".ARRAY_LOAD_FEED_TIME_SEQ_START[3], iSTART_PROGRAM_REQUEST := "DB22139_HOPPER_2_UNIT_2_POWDER_FILLING_START_STOP_BY_CURRENT".OUTPUT.POWDER_FILLING_START_BY_CURRENT, iSTART_AUTO_REQUEST :=, iSTOP_MANUAL_REQUEST := "DB7800_HMI_HOPPER_ACTIONS".ARRAY_LOAD_FEED_TIME_SEQ_STOP[3], iSTOP_PROGRAM_REQUEST := "DB22139_HOPPER_2_UNIT_2_POWDER_FILLING_START_STOP_BY_CURRENT".OUTPUT.POWDER_FILLING_STOP_BY_CURRENT, iSTOP_AUTO_REQUEST :=, MOTOR_STIRRER_SETPOINT := "DB22532_STIRRER_CONTROL_HOPPER_2_UNIT_2".PROGRAM_SETPOINT_VELOCITY, PRESSURE_SETPOINT := "DB22533_PRESSURE_CONTROL_HOPPER_2_UNIT_2".PRESSURE_SETPOINT_AUTO, oEXCEEDED_TIME_ALARM => "DB426_ALARMS_WARNINGS".CLADDING_HOPPERS."717480", oOUT_OF_RANGE_ALARM => "DB426_ALARMS_WARNINGS".CLADDING_HOPPERS."717481", oLOST_CONDITIONS => "DB426_ALARMS_WARNINGS".CLADDING_HOPPERS."717482", oIS_ALARMS =>)
   END_RUNG
   // the same network as SCL:
   "DB22731_LOAD_FEEDER_TIME_SEQUENCE_HOPPER_2_UNIT_2"(iCONTROL_ON_DELAYED := "DB2140_HOPPERS_MPP".MACHINE_ON_DELAYED,   // "FB22701_LOAD_FEEDER_SEQUENCE_TIME"
                           iPNEUMATIC_FEEDBACK_ON := "DB7300_INTERLOCK".GENERAL.PNEUMATIC_SYSTEM_ON,
                           iMOTOR_STIRRER_CONDITIONS := TRUE,
                           iHOPPER_FEEDBACK_PRESSURE := "DB22132_PRESSURE_HOPPER_2_UNIT_2".OUTPUT.VALUE,
                           iHOPPER_MOTOR_STIRRER_FEEDBACK_SPEED := "DB22532_STIRRER_CONTROL_HOPPER_2_UNIT_2".FEEDBACK_VELOCITY,
                           iPOWDER_FEEDER_HOPPER_FEEDBACK_PRESSURE := "DB22131_PRESSURE_FEEDER_HOPPER_2_UNIT_2".OUTPUT.VALUE,
                           iTRANSFER_POWDER_VALVE_FEEDBACK_ON := "DB22331_TRANSFER_POWDER_VALVE_HOPPER_2_UNIT_2"."DATA STANDARD".FEEDBACK_ON,
                           iTRANSFER_POWDER_VALVE_FEEDBACK_OFF := "DB22331_TRANSFER_POWDER_VALVE_HOPPER_2_UNIT_2"."DATA STANDARD".FEEDBACK_OFF,
                           iPOWDER_FLOW_ON := "DB22133_POWDER_FLOW_HOPPER_2_UNIT_2".oPOWDER_FLOW_ON,
                           iSTART_MANUAL_REQUEST := "DB7800_HMI_HOPPER_ACTIONS".ARRAY_LOAD_FEED_TIME_SEQ_START[3],
                           iSTART_PROGRAM_REQUEST := "DB22139_HOPPER_2_UNIT_2_POWDER_FILLING_START_STOP_BY_CURRENT".OUTPUT.POWDER_FILLING_START_BY_CURRENT,
                           iSTOP_MANUAL_REQUEST := "DB7800_HMI_HOPPER_ACTIONS".ARRAY_LOAD_FEED_TIME_SEQ_STOP[3],
                           iSTOP_PROGRAM_REQUEST := "DB22139_HOPPER_2_UNIT_2_POWDER_FILLING_START_STOP_BY_CURRENT".OUTPUT.POWDER_FILLING_STOP_BY_CURRENT,
                           MOTOR_STIRRER_SETPOINT := "DB22532_STIRRER_CONTROL_HOPPER_2_UNIT_2".PROGRAM_SETPOINT_VELOCITY,
                           PRESSURE_SETPOINT := "DB22533_PRESSURE_CONTROL_HOPPER_2_UNIT_2".PRESSURE_SETPOINT_AUTO,
                           oEXCEEDED_TIME_ALARM => "DB426_ALARMS_WARNINGS".CLADDING_HOPPERS."717480",
                           oOUT_OF_RANGE_ALARM => "DB426_ALARMS_WARNINGS".CLADDING_HOPPERS."717481",
                           oLOST_CONDITIONS => "DB426_ALARMS_WARNINGS".CLADDING_HOPPERS."717482");
END_REGION

REGION Network 14: CALL FB22702 LOAD FEEDER SEQUENCE WEIGHT UNIT 02 HOPPER 2
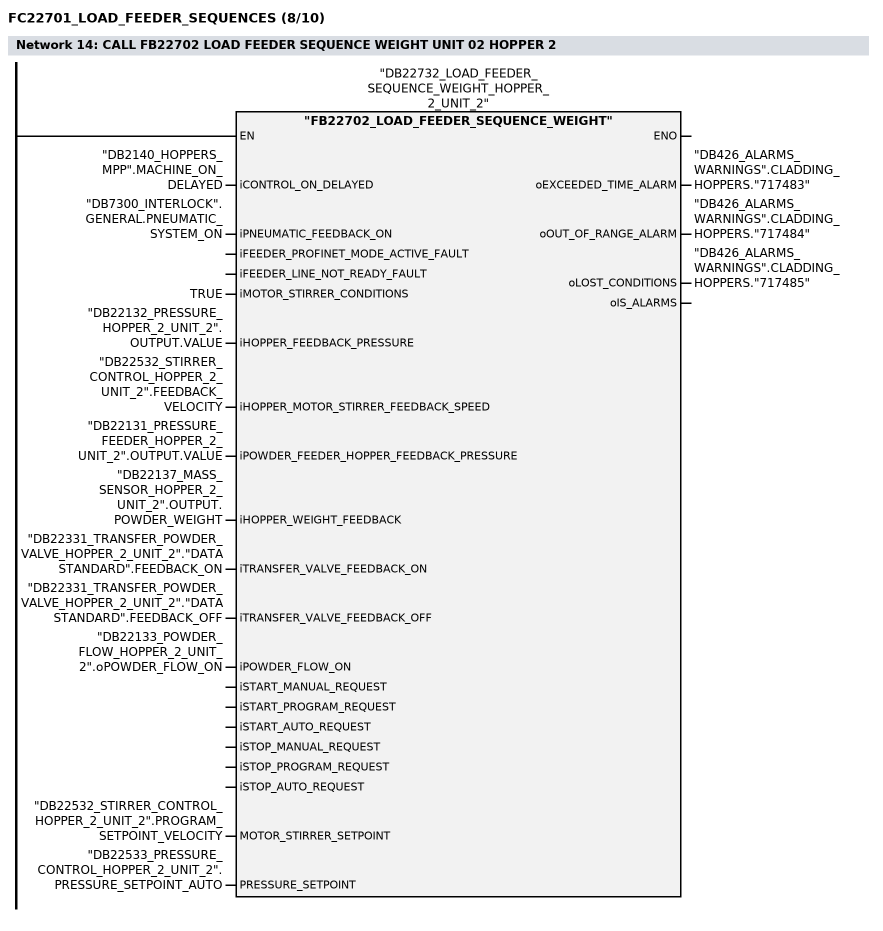
   RUNG wire#powerrail
      "DB22732_LOAD_FEEDER_SEQUENCE_WEIGHT_HOPPER_2_UNIT_2"(iCONTROL_ON_DELAYED := "DB2140_HOPPERS_MPP".MACHINE_ON_DELAYED, iPNEUMATIC_FEEDBACK_ON := "DB7300_INTERLOCK".GENERAL.PNEUMATIC_SYSTEM_ON, iFEEDER_PROFINET_MODE_ACTIVE_FAULT :=, iFEEDER_LINE_NOT_READY_FAULT :=, iMOTOR_STIRRER_CONDITIONS := TRUE, iHOPPER_FEEDBACK_PRESSURE := "DB22132_PRESSURE_HOPPER_2_UNIT_2".OUTPUT.VALUE, iHOPPER_MOTOR_STIRRER_FEEDBACK_SPEED := "DB22532_STIRRER_CONTROL_HOPPER_2_UNIT_2".FEEDBACK_VELOCITY, iPOWDER_FEEDER_HOPPER_FEEDBACK_PRESSURE := "DB22131_PRESSURE_FEEDER_HOPPER_2_UNIT_2".OUTPUT.VALUE, iHOPPER_WEIGHT_FEEDBACK := "DB22137_MASS_SENSOR_HOPPER_2_UNIT_2".OUTPUT.POWDER_WEIGHT, iTRANSFER_VALVE_FEEDBACK_ON := "DB22331_TRANSFER_POWDER_VALVE_HOPPER_2_UNIT_2"."DATA STANDARD".FEEDBACK_ON, iTRANSFER_VALVE_FEEDBACK_OFF := "DB22331_TRANSFER_POWDER_VALVE_HOPPER_2_UNIT_2"."DATA STANDARD".FEEDBACK_OFF, iPOWDER_FLOW_ON := "DB22133_POWDER_FLOW_HOPPER_2_UNIT_2".oPOWDER_FLOW_ON, iSTART_MANUAL_REQUEST :=, iSTART_AUTO_REQUEST :=, iSTOP_MANUAL_REQUEST :=, iSTOP_AUTO_REQUEST :=, MOTOR_STIRRER_SETPOINT := "DB22532_STIRRER_CONTROL_HOPPER_2_UNIT_2".PROGRAM_SETPOINT_VELOCITY, PRESSURE_SETPOINT := "DB22533_PRESSURE_CONTROL_HOPPER_2_UNIT_2".PRESSURE_SETPOINT_AUTO, oEXCEEDED_TIME_ALARM => "DB426_ALARMS_WARNINGS".CLADDING_HOPPERS."717483", oOUT_OF_RANGE_ALARM => "DB426_ALARMS_WARNINGS".CLADDING_HOPPERS."717484", oLOST_CONDITIONS => "DB426_ALARMS_WARNINGS".CLADDING_HOPPERS."717485", oIS_ALARMS =>, iSTART_PROGRAM_REQUEST :=, iSTOP_PROGRAM_REQUEST :=)
   END_RUNG
   // the same network as SCL:
   "DB22732_LOAD_FEEDER_SEQUENCE_WEIGHT_HOPPER_2_UNIT_2"(iCONTROL_ON_DELAYED := "DB2140_HOPPERS_MPP".MACHINE_ON_DELAYED,   // "FB22702_LOAD_FEEDER_SEQUENCE_WEIGHT"
                           iPNEUMATIC_FEEDBACK_ON := "DB7300_INTERLOCK".GENERAL.PNEUMATIC_SYSTEM_ON,
                           iMOTOR_STIRRER_CONDITIONS := TRUE,
                           iHOPPER_FEEDBACK_PRESSURE := "DB22132_PRESSURE_HOPPER_2_UNIT_2".OUTPUT.VALUE,
                           iHOPPER_MOTOR_STIRRER_FEEDBACK_SPEED := "DB22532_STIRRER_CONTROL_HOPPER_2_UNIT_2".FEEDBACK_VELOCITY,
                           iPOWDER_FEEDER_HOPPER_FEEDBACK_PRESSURE := "DB22131_PRESSURE_FEEDER_HOPPER_2_UNIT_2".OUTPUT.VALUE,
                           iHOPPER_WEIGHT_FEEDBACK := "DB22137_MASS_SENSOR_HOPPER_2_UNIT_2".OUTPUT.POWDER_WEIGHT,
                           iTRANSFER_VALVE_FEEDBACK_ON := "DB22331_TRANSFER_POWDER_VALVE_HOPPER_2_UNIT_2"."DATA STANDARD".FEEDBACK_ON,
                           iTRANSFER_VALVE_FEEDBACK_OFF := "DB22331_TRANSFER_POWDER_VALVE_HOPPER_2_UNIT_2"."DATA STANDARD".FEEDBACK_OFF,
                           iPOWDER_FLOW_ON := "DB22133_POWDER_FLOW_HOPPER_2_UNIT_2".oPOWDER_FLOW_ON,
                           MOTOR_STIRRER_SETPOINT := "DB22532_STIRRER_CONTROL_HOPPER_2_UNIT_2".PROGRAM_SETPOINT_VELOCITY,
                           PRESSURE_SETPOINT := "DB22533_PRESSURE_CONTROL_HOPPER_2_UNIT_2".PRESSURE_SETPOINT_AUTO,
                           oEXCEEDED_TIME_ALARM => "DB426_ALARMS_WARNINGS".CLADDING_HOPPERS."717483",
                           oOUT_OF_RANGE_ALARM => "DB426_ALARMS_WARNINGS".CLADDING_HOPPERS."717484",
                           oLOST_CONDITIONS => "DB426_ALARMS_WARNINGS".CLADDING_HOPPERS."717485");
END_REGION

REGION Network 15: /////_HOPPER_3_SEQUENCES_/////
END_REGION

REGION Network 16: CALL FB22701 LOAD FEEDER SEQUENCE TIME UNIT 02 HOPPER 3
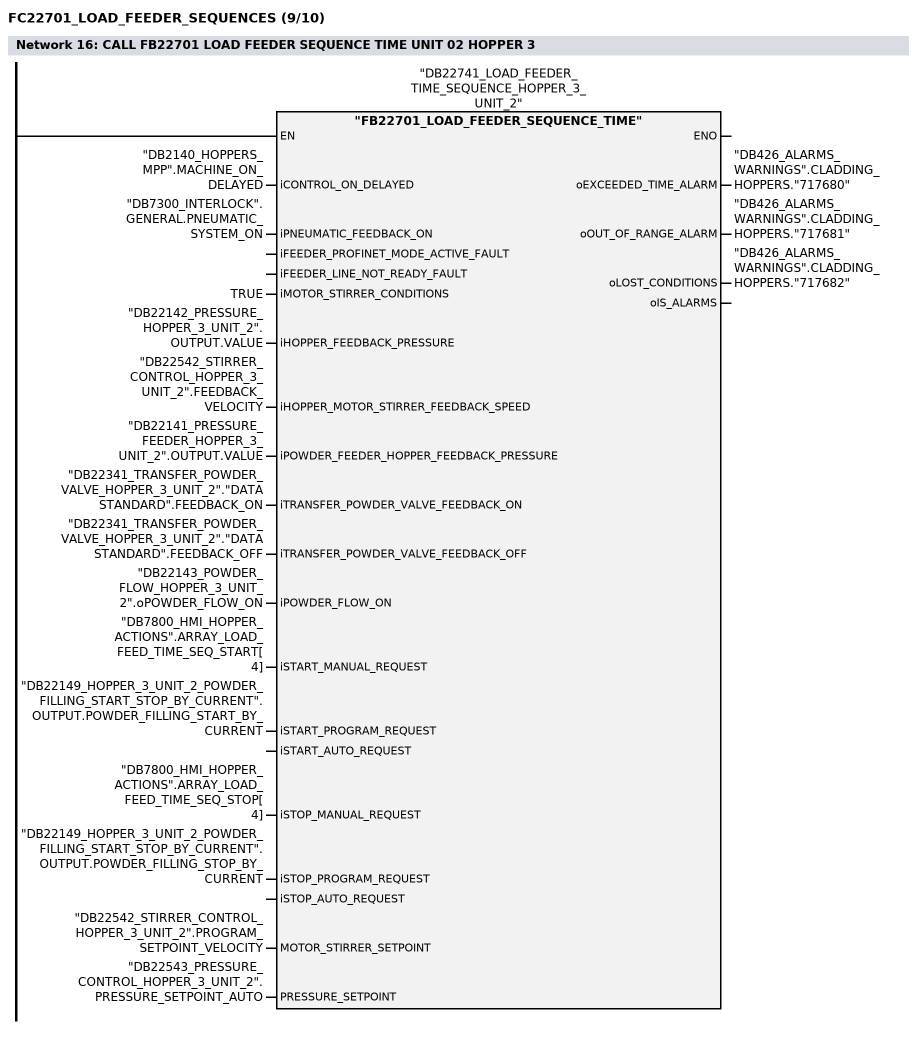
   RUNG wire#powerrail
      "DB22741_LOAD_FEEDER_TIME_SEQUENCE_HOPPER_3_UNIT_2"(iCONTROL_ON_DELAYED := "DB2140_HOPPERS_MPP".MACHINE_ON_DELAYED, iPNEUMATIC_FEEDBACK_ON := "DB7300_INTERLOCK".GENERAL.PNEUMATIC_SYSTEM_ON, iFEEDER_PROFINET_MODE_ACTIVE_FAULT :=, iFEEDER_LINE_NOT_READY_FAULT :=, iMOTOR_STIRRER_CONDITIONS := TRUE, iHOPPER_FEEDBACK_PRESSURE := "DB22142_PRESSURE_HOPPER_3_UNIT_2".OUTPUT.VALUE, iHOPPER_MOTOR_STIRRER_FEEDBACK_SPEED := "DB22542_STIRRER_CONTROL_HOPPER_3_UNIT_2".FEEDBACK_VELOCITY, iPOWDER_FEEDER_HOPPER_FEEDBACK_PRESSURE := "DB22141_PRESSURE_FEEDER_HOPPER_3_UNIT_2".OUTPUT.VALUE, iTRANSFER_POWDER_VALVE_FEEDBACK_ON := "DB22341_TRANSFER_POWDER_VALVE_HOPPER_3_UNIT_2"."DATA STANDARD".FEEDBACK_ON, iTRANSFER_POWDER_VALVE_FEEDBACK_OFF := "DB22341_TRANSFER_POWDER_VALVE_HOPPER_3_UNIT_2"."DATA STANDARD".FEEDBACK_OFF, iPOWDER_FLOW_ON := "DB22143_POWDER_FLOW_HOPPER_3_UNIT_2".oPOWDER_FLOW_ON, iSTART_MANUAL_REQUEST := "DB7800_HMI_HOPPER_ACTIONS".ARRAY_LOAD_FEED_TIME_SEQ_START[4], iSTART_PROGRAM_REQUEST := "DB22149_HOPPER_3_UNIT_2_POWDER_FILLING_START_STOP_BY_CURRENT".OUTPUT.POWDER_FILLING_START_BY_CURRENT, iSTART_AUTO_REQUEST :=, iSTOP_MANUAL_REQUEST := "DB7800_HMI_HOPPER_ACTIONS".ARRAY_LOAD_FEED_TIME_SEQ_STOP[4], iSTOP_PROGRAM_REQUEST := "DB22149_HOPPER_3_UNIT_2_POWDER_FILLING_START_STOP_BY_CURRENT".OUTPUT.POWDER_FILLING_STOP_BY_CURRENT, iSTOP_AUTO_REQUEST :=, MOTOR_STIRRER_SETPOINT := "DB22542_STIRRER_CONTROL_HOPPER_3_UNIT_2".PROGRAM_SETPOINT_VELOCITY, PRESSURE_SETPOINT := "DB22543_PRESSURE_CONTROL_HOPPER_3_UNIT_2".PRESSURE_SETPOINT_AUTO, oEXCEEDED_TIME_ALARM => "DB426_ALARMS_WARNINGS".CLADDING_HOPPERS."717680", oOUT_OF_RANGE_ALARM => "DB426_ALARMS_WARNINGS".CLADDING_HOPPERS."717681", oLOST_CONDITIONS => "DB426_ALARMS_WARNINGS".CLADDING_HOPPERS."717682", oIS_ALARMS =>)
   END_RUNG
   // the same network as SCL:
   "DB22741_LOAD_FEEDER_TIME_SEQUENCE_HOPPER_3_UNIT_2"(iCONTROL_ON_DELAYED := "DB2140_HOPPERS_MPP".MACHINE_ON_DELAYED,   // "FB22701_LOAD_FEEDER_SEQUENCE_TIME"
                           iPNEUMATIC_FEEDBACK_ON := "DB7300_INTERLOCK".GENERAL.PNEUMATIC_SYSTEM_ON,
                           iMOTOR_STIRRER_CONDITIONS := TRUE,
                           iHOPPER_FEEDBACK_PRESSURE := "DB22142_PRESSURE_HOPPER_3_UNIT_2".OUTPUT.VALUE,
                           iHOPPER_MOTOR_STIRRER_FEEDBACK_SPEED := "DB22542_STIRRER_CONTROL_HOPPER_3_UNIT_2".FEEDBACK_VELOCITY,
                           iPOWDER_FEEDER_HOPPER_FEEDBACK_PRESSURE := "DB22141_PRESSURE_FEEDER_HOPPER_3_UNIT_2".OUTPUT.VALUE,
                           iTRANSFER_POWDER_VALVE_FEEDBACK_ON := "DB22341_TRANSFER_POWDER_VALVE_HOPPER_3_UNIT_2"."DATA STANDARD".FEEDBACK_ON,
                           iTRANSFER_POWDER_VALVE_FEEDBACK_OFF := "DB22341_TRANSFER_POWDER_VALVE_HOPPER_3_UNIT_2"."DATA STANDARD".FEEDBACK_OFF,
                           iPOWDER_FLOW_ON := "DB22143_POWDER_FLOW_HOPPER_3_UNIT_2".oPOWDER_FLOW_ON,
                           iSTART_MANUAL_REQUEST := "DB7800_HMI_HOPPER_ACTIONS".ARRAY_LOAD_FEED_TIME_SEQ_START[4],
                           iSTART_PROGRAM_REQUEST := "DB22149_HOPPER_3_UNIT_2_POWDER_FILLING_START_STOP_BY_CURRENT".OUTPUT.POWDER_FILLING_START_BY_CURRENT,
                           iSTOP_MANUAL_REQUEST := "DB7800_HMI_HOPPER_ACTIONS".ARRAY_LOAD_FEED_TIME_SEQ_STOP[4],
                           iSTOP_PROGRAM_REQUEST := "DB22149_HOPPER_3_UNIT_2_POWDER_FILLING_START_STOP_BY_CURRENT".OUTPUT.POWDER_FILLING_STOP_BY_CURRENT,
                           MOTOR_STIRRER_SETPOINT := "DB22542_STIRRER_CONTROL_HOPPER_3_UNIT_2".PROGRAM_SETPOINT_VELOCITY,
                           PRESSURE_SETPOINT := "DB22543_PRESSURE_CONTROL_HOPPER_3_UNIT_2".PRESSURE_SETPOINT_AUTO,
                           oEXCEEDED_TIME_ALARM => "DB426_ALARMS_WARNINGS".CLADDING_HOPPERS."717680",
                           oOUT_OF_RANGE_ALARM => "DB426_ALARMS_WARNINGS".CLADDING_HOPPERS."717681",
                           oLOST_CONDITIONS => "DB426_ALARMS_WARNINGS".CLADDING_HOPPERS."717682");
END_REGION

REGION Network 17: CALL FB22702 LOAD FEEDER SEQUENCE WEIGHT UNIT 02 HOPPER 3
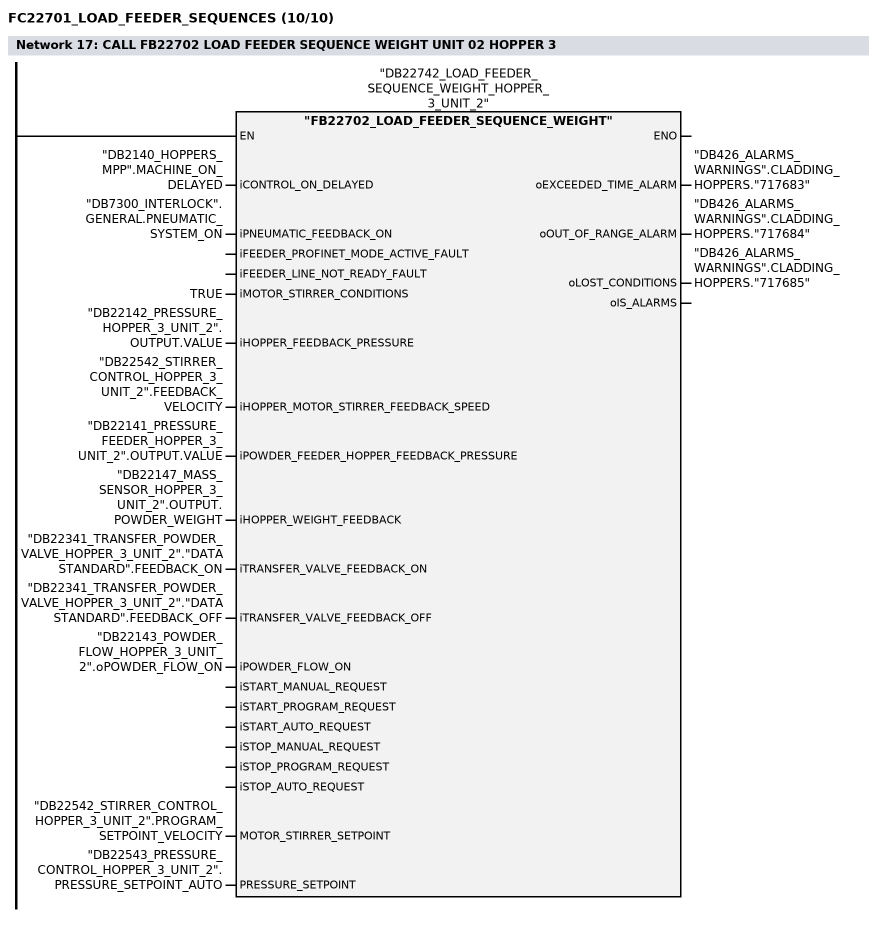
   RUNG wire#powerrail
      "DB22742_LOAD_FEEDER_SEQUENCE_WEIGHT_HOPPER_3_UNIT_2"(iCONTROL_ON_DELAYED := "DB2140_HOPPERS_MPP".MACHINE_ON_DELAYED, iPNEUMATIC_FEEDBACK_ON := "DB7300_INTERLOCK".GENERAL.PNEUMATIC_SYSTEM_ON, iFEEDER_PROFINET_MODE_ACTIVE_FAULT :=, iFEEDER_LINE_NOT_READY_FAULT :=, iMOTOR_STIRRER_CONDITIONS := TRUE, iHOPPER_FEEDBACK_PRESSURE := "DB22142_PRESSURE_HOPPER_3_UNIT_2".OUTPUT.VALUE, iHOPPER_MOTOR_STIRRER_FEEDBACK_SPEED := "DB22542_STIRRER_CONTROL_HOPPER_3_UNIT_2".FEEDBACK_VELOCITY, iPOWDER_FEEDER_HOPPER_FEEDBACK_PRESSURE := "DB22141_PRESSURE_FEEDER_HOPPER_3_UNIT_2".OUTPUT.VALUE, iHOPPER_WEIGHT_FEEDBACK := "DB22147_MASS_SENSOR_HOPPER_3_UNIT_2".OUTPUT.POWDER_WEIGHT, iTRANSFER_VALVE_FEEDBACK_ON := "DB22341_TRANSFER_POWDER_VALVE_HOPPER_3_UNIT_2"."DATA STANDARD".FEEDBACK_ON, iTRANSFER_VALVE_FEEDBACK_OFF := "DB22341_TRANSFER_POWDER_VALVE_HOPPER_3_UNIT_2"."DATA STANDARD".FEEDBACK_OFF, iPOWDER_FLOW_ON := "DB22143_POWDER_FLOW_HOPPER_3_UNIT_2".oPOWDER_FLOW_ON, iSTART_MANUAL_REQUEST :=, iSTART_AUTO_REQUEST :=, iSTOP_MANUAL_REQUEST :=, iSTOP_AUTO_REQUEST :=, MOTOR_STIRRER_SETPOINT := "DB22542_STIRRER_CONTROL_HOPPER_3_UNIT_2".PROGRAM_SETPOINT_VELOCITY, PRESSURE_SETPOINT := "DB22543_PRESSURE_CONTROL_HOPPER_3_UNIT_2".PRESSURE_SETPOINT_AUTO, oEXCEEDED_TIME_ALARM => "DB426_ALARMS_WARNINGS".CLADDING_HOPPERS."717683", oOUT_OF_RANGE_ALARM => "DB426_ALARMS_WARNINGS".CLADDING_HOPPERS."717684", oLOST_CONDITIONS => "DB426_ALARMS_WARNINGS".CLADDING_HOPPERS."717685", oIS_ALARMS =>, iSTART_PROGRAM_REQUEST :=, iSTOP_PROGRAM_REQUEST :=)
   END_RUNG
   // the same network as SCL:
   "DB22742_LOAD_FEEDER_SEQUENCE_WEIGHT_HOPPER_3_UNIT_2"(iCONTROL_ON_DELAYED := "DB2140_HOPPERS_MPP".MACHINE_ON_DELAYED,   // "FB22702_LOAD_FEEDER_SEQUENCE_WEIGHT"
                           iPNEUMATIC_FEEDBACK_ON := "DB7300_INTERLOCK".GENERAL.PNEUMATIC_SYSTEM_ON,
                           iMOTOR_STIRRER_CONDITIONS := TRUE,
                           iHOPPER_FEEDBACK_PRESSURE := "DB22142_PRESSURE_HOPPER_3_UNIT_2".OUTPUT.VALUE,
                           iHOPPER_MOTOR_STIRRER_FEEDBACK_SPEED := "DB22542_STIRRER_CONTROL_HOPPER_3_UNIT_2".FEEDBACK_VELOCITY,
                           iPOWDER_FEEDER_HOPPER_FEEDBACK_PRESSURE := "DB22141_PRESSURE_FEEDER_HOPPER_3_UNIT_2".OUTPUT.VALUE,
                           iHOPPER_WEIGHT_FEEDBACK := "DB22147_MASS_SENSOR_HOPPER_3_UNIT_2".OUTPUT.POWDER_WEIGHT,
                           iTRANSFER_VALVE_FEEDBACK_ON := "DB22341_TRANSFER_POWDER_VALVE_HOPPER_3_UNIT_2"."DATA STANDARD".FEEDBACK_ON,
                           iTRANSFER_VALVE_FEEDBACK_OFF := "DB22341_TRANSFER_POWDER_VALVE_HOPPER_3_UNIT_2"."DATA STANDARD".FEEDBACK_OFF,
                           iPOWDER_FLOW_ON := "DB22143_POWDER_FLOW_HOPPER_3_UNIT_2".oPOWDER_FLOW_ON,
                           MOTOR_STIRRER_SETPOINT := "DB22542_STIRRER_CONTROL_HOPPER_3_UNIT_2".PROGRAM_SETPOINT_VELOCITY,
                           PRESSURE_SETPOINT := "DB22543_PRESSURE_CONTROL_HOPPER_3_UNIT_2".PRESSURE_SETPOINT_AUTO,
                           oEXCEEDED_TIME_ALARM => "DB426_ALARMS_WARNINGS".CLADDING_HOPPERS."717683",
                           oOUT_OF_RANGE_ALARM => "DB426_ALARMS_WARNINGS".CLADDING_HOPPERS."717684",
                           oLOST_CONDITIONS => "DB426_ALARMS_WARNINGS".CLADDING_HOPPERS."717685");
END_REGION
END_FUNCTION

FUNCTION_BLOCK "FB31_SPINDLE"   // FB31, LAD
{ S7_Optimized_Access := 'FALSE' }
AUTHOR : ETXETAR
VERSION : 1.0
// stored: AutoNumber false, IsIECCheckEnabled false, SetENOAutomatically false, UDAEnableTagReadback false
   VAR_INPUT
      OPTIONS_0 : Byte := 2#0000_0000;   // OPTIONS 0
      OPTIONS_1 : Byte := 2#0000_0000;   // OPTIONS 1
      SAFETY_BYPASS : Bool;   // MUST BE ALWAYS OFF, ACTIVATE ONLY FOR TEST
      OPTIMIZATION_BYPASS : Bool;   // MUST BE ALWAYS OFF, ACTIVATE ONLY FOR OPTIMIZATION TEST
      RPMS_REACHED : Bool;   // RPMS REACHED / N.O
      BELT_BROKEN : Bool;   // BELT BROKEN / N.C
      COOLING_SYS_IN_SERVICE : Bool;   // COOLING SYSTEM IN SERVICE
      MQL_HP_IN_SERVICE : Bool;   // MQL OR HP IN SERVICE
      TEMPERATURE_SENSOR : Word;   // TEMPERATURE SENSOR
      TEMPERATURE_SENSOR_PTC : Bool;   // TEMPERATURE SENSOR PTC
      VPM_READY : Bool;   // VOLTAGE PROTECTION MODULE READY
      ENABLE : Bool;   // ENABLE
      FEED_HOLD_COND : Bool;   // FEED HOLD CONDITION
      UNIT_SEQ_RUNNING : Bool;   // UNIT SEQUENCE RUNNING
      SAFE_ENABLED : Bool;   // SAFETY ENABLED
      TEST_STOP_INTERNAL_PULSES : Bool;   // TEST STOP INTERNAL PULSES
      FEED_OVERRIDE : Byte;   // FEED OVERRIDE
      SPINDLE_OVERRIDE : Byte;   // SPINDLE OVERRIDE
      HMI_SP_SELECTED : Bool;   // HMI SPINDLE SELECTED
      HMI_REQ_LINE : Bool;   // HMI REQUEST LINE
      CHANNEL_M3 : Bool;   // CHANNEL M3
      CHANNEL_M300 : Bool;   // CHANNEL M300
      M_VERIFY_CLAMP_F1 : Bool;   // M VERIFY CLAMPED FIXTURE 1
      M_VERIFY_CLAMP_F2 : Bool;   // M VERIFY CLAMPED FIXTURE 2
      SP_CLAMP : Bool;   // SPINDLE CLAMPING UNIT CLAMP
      SP_CLAMPED : Bool;   // SPINDLE CLAMPING UNIT CLAMPED
      SP_CLAMPED_WITH_TOOL : Bool;   // SPINDLE CLAMPING UNIT CLAMPED WITH TOOL
      HARDWARE_ENABLE : Bool;   // HARDWARE ENABLE
      TOOL_CHANGE_POS : Bool;   // TOOL CHANGE POSITION
      FIXTURE_1_PART_OK : Bool;   // FIXTURE 1 PART OK
      FIXTURE_2_PART_OK : Bool;   // FIXTURE 2 PART OK
      READ_POS : DWord;   // READ POSITION
      UNIT_ALARM : UInt;   // UNIT NUMBER MAX. NUMBER=10
      STATION_ALARM : UInt;   // STATION NUMBER MIN. NUMBER=0 MAX. NUMBER=4
      DESELECT_SPINDLE_STO : Bool;   // DESELECT SPINDLE STO
   END_VAR
   VAR_OUTPUT
      DELAYED_ENABLE : Bool;   // DELAYED ENABLE
      FEED_HOLD_CONDITIONS : Bool;   // FEED HOLD CONDITIONS
      FEED_HOLD_CONDITIONS_HMI : Bool;   // HMI FEED HOLD CONDITIONS
      SP_DESELECTED : Bool;   // SPINDLE DESELECTED
      SPEED_NOT_REACHED_ALARM : Bool;   // SPEED NOT REACHED ALARM
      BELT_BROKEN_ALARM : Bool;   // BELT BROKEN ALARM
      COOLING_ALARM : Bool;   // COOLING ALARM
      MQL_HP_ALARM : Bool;   // MQL HP ALARM
      HIGH_TEMP_ALARM : Bool;   // HIGH TEMPERATURE ALARM
      HIGH_TEMP_PTC_ALARM : Bool;   // HIGH TEMPERATURE PTC ALARM
      VPM_READY_ALARM : Bool;   // VPM READY ALARM
      HIGH_TEMP_PREALM : Bool;   // HIGH TEMPERATURE PREALARM
      SPINDLE_POS : Real;   // SPINDLE POSITION
      HMI_MOTION_EXECUTABILITY_LEFT : Bool;   // HMI MOTION EXECUTABILITY LEFT
      HMI_MOTION_EXECUTABILITY_RIGHT : Bool;   // HMI MOTION EXECUTABILITY RIGHT
      HMI_MOTION_END_POS_LEFT : Bool;   // HMI MOTION END POSITION LEFT
      HMI_MOTION_END_POS_RIGHT : Bool;   // HMI MOTION END POSITION RIGHT
   END_VAR
   VAR_IN_OUT
      SpindleDB : "LBP_typeAxisX";
   END_VAR
   VAR DB_SPECIFIC
      SP : "SPINDLE";
      SP_TEMPERATURE : Real;   // SPINDLE TEMPERATURE
      TEMP_MUL_VAL { S7_SetPoint := 'True'} : Real := 800.0;   // CONVERSION VALUE TO MUL THE INPUT
      TEMP_DIV_VAL { S7_SetPoint := 'True'} : Real := 16383.0;   // CONVERSION VALUE TO DIV THE MUL VALUE
      TEMP_SUB_VAL { S7_SetPoint := 'True'} : Real := 200.0;   // CONVERSION VALUE TO SUB TO THE SUB VALUE
      TEMP_PREALARM_VAL { S7_SetPoint := 'True'} : Real := 40.0;   // TEMPERATURE PREALARM VALUE
      TEMP_ALARM_VAL { S7_SetPoint := 'True'} : Real := 45.0;   // TEMPERATURE ALARM VALUE
      WARNING_GONE { S7_SetPoint := 'True'} : Bool;   // WARNING GONE
      TIMER_ENABLE_PULSE { S7_SetPoint := 'True'} : TOF_TIME;   // ENABLE PULSE TIMER
      TIMER_DELETE_DIST_TO_GO { S7_SetPoint := 'True'} : TON_TIME;   // DELETE DISTANCE TO GO TIMER
      TIMER_SPEED_NOT_REACHED { S7_SetPoint := 'True'} : TOF_TIME;   // SPEED NOT REACHED TIMER
      TIMER_BELT_BROKEN_ALARM { S7_SetPoint := 'True'} : TON_TIME;   // BELT BROKEN TIMER
      TIMER_MQL_HP_FAULT { S7_SetPoint := 'True'} : TON_TIME;   // MQL OR HP FAULT TIMER
      TIMER_COMMAND_JOG_PLUS { S7_SetPoint := 'True'} : TON_TIME;   // COMMAND JOG PLUS TIMER
   END_VAR
   VAR
      SAFETY_POSITIONS { S7_SetPoint := 'True'} : "FB33_SAFETY_POSITIONS";
   END_VAR
   VAR_TEMP
      INPUTS_MASK : Byte;   // INPUT MASK
      O_BYTE_0 : Struct   // OPTION BYTE 0
         MEASURING_SYSTEM_2 : Bool;   // MEASURING SYSTEM 2 OPTION / ALWAYS ON OR ALWAYS OFF
         BELT_BROKEN : Bool;   // BELT BROKEN OPTION
         COOLING : Bool;   // COOLING OPTION / ALWAYS ON OR ALWAYS OFF
         MQL_OR_HP : Bool;   // MQL OR HP OPTION / ALWAYS ON OR ALWAYS OFF
         ANALOG_TEMPERATURE_SENSOR : Bool;   // ANALOG TEMPERATURE SENSOR OPTION
         PTC_TEMP_SENSOR : Bool;   // PTC TEMPERATURE SENSOR OPTION
         TWIN_KESSLER_VPM_READY : Bool;   // TWIN KESSLER VPM READY OPTION
         MPP_SP_OVERRIDE : Bool;   // MPP SPINDLE OVERRIDE OPTION
      END_STRUCT;
      O_BYTE_1 : Struct   // OPTION BYTE 1
         SPARE_0 : Bool;   // SPARE OPTION / ALWAYS ON OR ALWAYS OFF
         SPARE_1 : Bool;   // SPARE OPTION
         SPARE_2 : Bool;   // SPARE OPTION / ALWAYS ON OR ALWAYS OFF
         SPARE_3 : Bool;   // SPARE OPTION / ALWAYS ON OR ALWAYS OFF
         SPARE_4 : Bool;   // SPARE OPTION
         SPARE_5 : Bool;   // SPARE OPTION
         SPARE_6 : Bool;   // SPARE OPTION
         SPARE_7 : Bool;   // SPARE OPTION
      END_STRUCT;
      TEMP_INPUT : DInt;   // TEMPERATURE INPUR SHIFTED
      TEMP_REAL : Real;   // TEMPERATURE IN REAL
      DB_NUMBER : DInt;   // DB NUMBER FOR ALARMS AND HELP DECODING
   END_VAR
   // TIMER_ENABLE_PULSE.PT := T#1s;
   // TIMER_DELETE_DIST_TO_GO.PT := T#20ms;
   // TIMER_SPEED_NOT_REACHED.PT := T#100ms;
   // TIMER_BELT_BROKEN_ALARM.PT := T#150ms;
   // TIMER_MQL_HP_FAULT.PT := T#50ms;
   // TIMER_COMMAND_JOG_PLUS.PT := T#100ms;
   VAR_TEMP   // added for the SCL form of the ladder/FBD networks
      _w1 : Bool;
      _w2 : Bool;
      _w3 : Bool;
      _w4 : Bool;
      _w5 : Bool;
      _w6 : Bool;
      _w7 : Bool;
      _w8 : Bool;
      _w9 : Bool;
      _w10 : Bool;
      _w11 : Bool;
   END_VAR
BEGIN

NETWORK
TITLE = READ INSTANCE DB
      L     DINO;
      +     10#800000;
      T     #DB_NUMBER;


REGION Network 2: OPTIONS
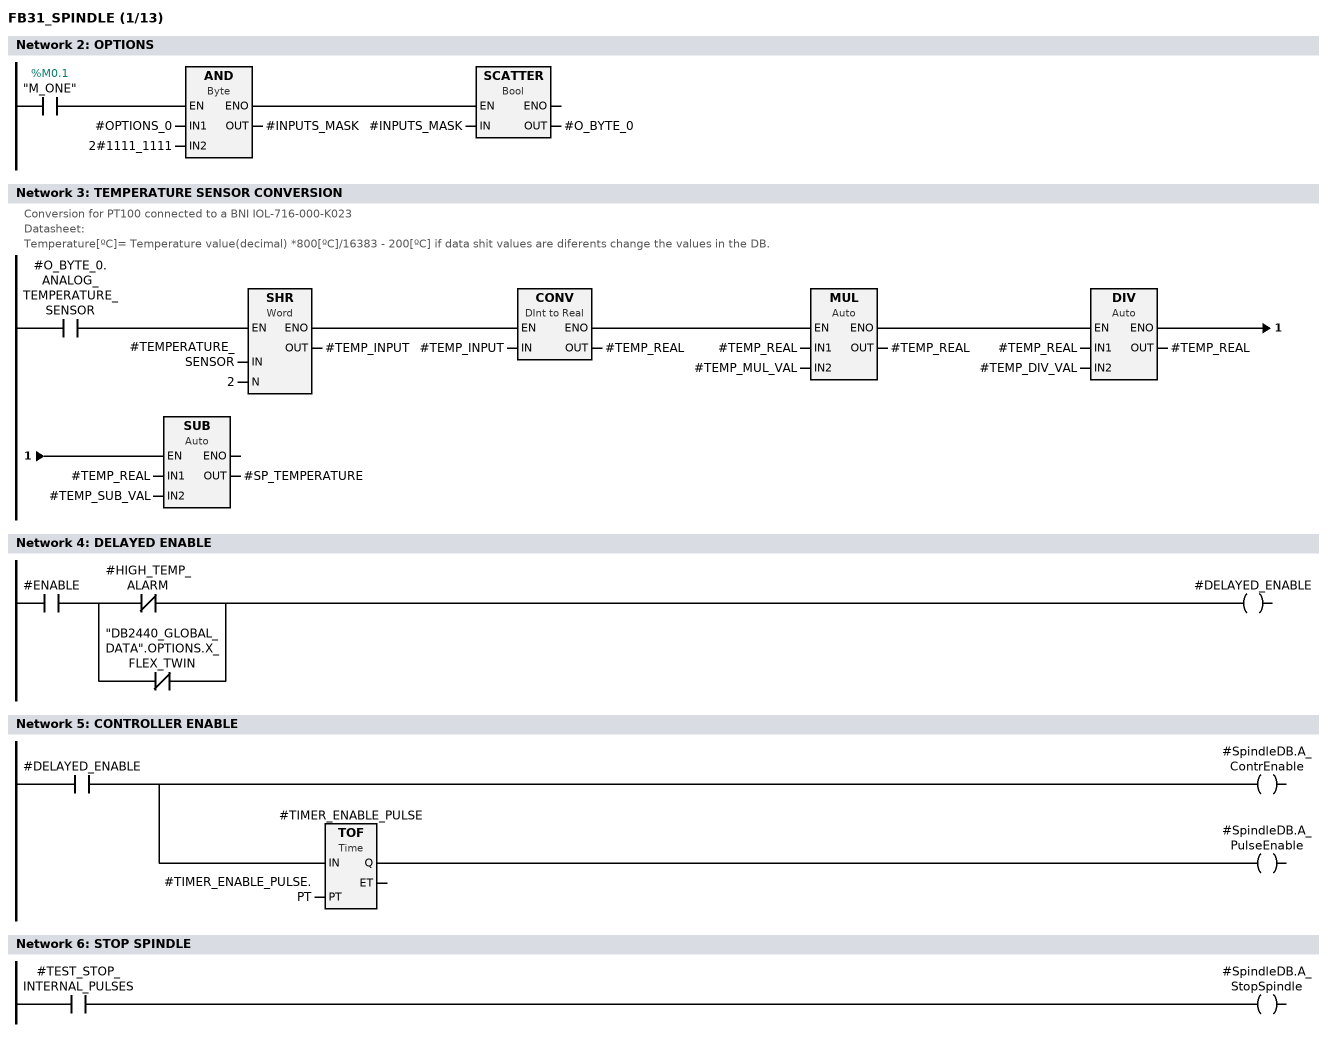
   RUNG wire#powerrail
      Contact( "M_ONE" )
      { S7_Templates := "SrcType := Byte"; S7_GenerateENO := "TRUE" } And(in1 := #OPTIONS_0, in2 := 2#1111_1111, out => #INPUTS_MASK)
      { S7_Templates := "[dest_type := Bool, src_type := Byte]" } SCATTER(IN := #INPUTS_MASK, OUT => #O_BYTE_0)
   END_RUNG
   // the same network as SCL:
   IF "M_ONE" THEN
       #INPUTS_MASK := #OPTIONS_0 AND 2#1111_1111;
       SCATTER(IN := #INPUTS_MASK, OUT => #O_BYTE_0);
   END_IF;
END_REGION

REGION Network 3: TEMPERATURE SENSOR CONVERSION
   // Conversion for PT100 connected to a BNI IOL-716-000-K023
   // 
   // Datasheet:
   // 
   //  Temperature[ºC]= Temperature value(decimal) *800[ºC]/16383 - 200[ºC] if data shit values are diferents change the values in the DB.
   RUNG wire#powerrail
      Contact( #O_BYTE_0.ANALOG_TEMPERATURE_SENSOR )
      { S7_Templates := "SrcType := Word" } Shr(in := #TEMPERATURE_SENSOR, n := 2, out => #TEMP_INPUT)
      { S7_Templates := "[SrcType := DInt, DestType := Real]" } Convert(in := #TEMP_INPUT, out => #TEMP_REAL)
      Mul(in1 := #TEMP_REAL, in2 := #TEMP_MUL_VAL, out => #TEMP_REAL)
      Div(in1 := #TEMP_REAL, in2 := #TEMP_DIV_VAL, out => #TEMP_REAL)
      Sub(in1 := #TEMP_REAL, in2 := #TEMP_SUB_VAL, out => #SP_TEMPERATURE)
   END_RUNG
   // the same network as SCL:
   IF #O_BYTE_0.ANALOG_TEMPERATURE_SENSOR THEN
       #TEMP_INPUT := SHR(IN := #TEMPERATURE_SENSOR, N := 2);
       #TEMP_REAL := DINT_TO_REAL(#TEMP_INPUT);
       #TEMP_REAL := #TEMP_REAL * #TEMP_MUL_VAL;
       #TEMP_REAL := #TEMP_REAL / #TEMP_DIV_VAL;
       #SP_TEMPERATURE := #TEMP_REAL - #TEMP_SUB_VAL;
   END_IF;
END_REGION

REGION Network 4: DELAYED ENABLE
   RUNG wire#powerrail
      Contact( #ENABLE )
      wire#w1
      I_Contact( #HIGH_TEMP_ALARM )
      wire#w2
      Coil( #DELAYED_ENABLE )
   END_RUNG
   RUNG wire#w1
      I_Contact( "DB2440_GLOBAL_DATA".OPTIONS.X_FLEX_TWIN )
   END_RUNG wire#w2
   // the same network as SCL:
   #DELAYED_ENABLE := #ENABLE AND (NOT #HIGH_TEMP_ALARM OR NOT "DB2440_GLOBAL_DATA".OPTIONS.X_FLEX_TWIN);
END_REGION

REGION Network 5: CONTROLLER ENABLE
   RUNG wire#powerrail
      Contact( #DELAYED_ENABLE )
      wire#w1
      Coil( #SpindleDB.A_ContrEnable )
   END_RUNG
   RUNG wire#w1
      { S7_Templates := "time_type := Time" } #TIMER_ENABLE_PULSE.TOF(pt := #TIMER_ENABLE_PULSE.PT, et =>)
      Coil( #SpindleDB.A_PulseEnable )
   END_RUNG
   // the same network as SCL:
   #SpindleDB.A_ContrEnable := #DELAYED_ENABLE;
   #TIMER_ENABLE_PULSE(IN := #DELAYED_ENABLE, PT := #TIMER_ENABLE_PULSE.PT);   // TOF
   #SpindleDB.A_PulseEnable := #TIMER_ENABLE_PULSE.Q;
END_REGION

REGION Network 6: STOP SPINDLE
   RUNG wire#powerrail
      Contact( #TEST_STOP_INTERNAL_PULSES )
      Coil( #SpindleDB.A_StopSpindle )
   END_RUNG
   // the same network as SCL:
   #SpindleDB.A_StopSpindle := #TEST_STOP_INTERNAL_PULSES;
END_REGION

REGION Network 7: DELETE DISTANCE TO GO / DELETE S VALUE
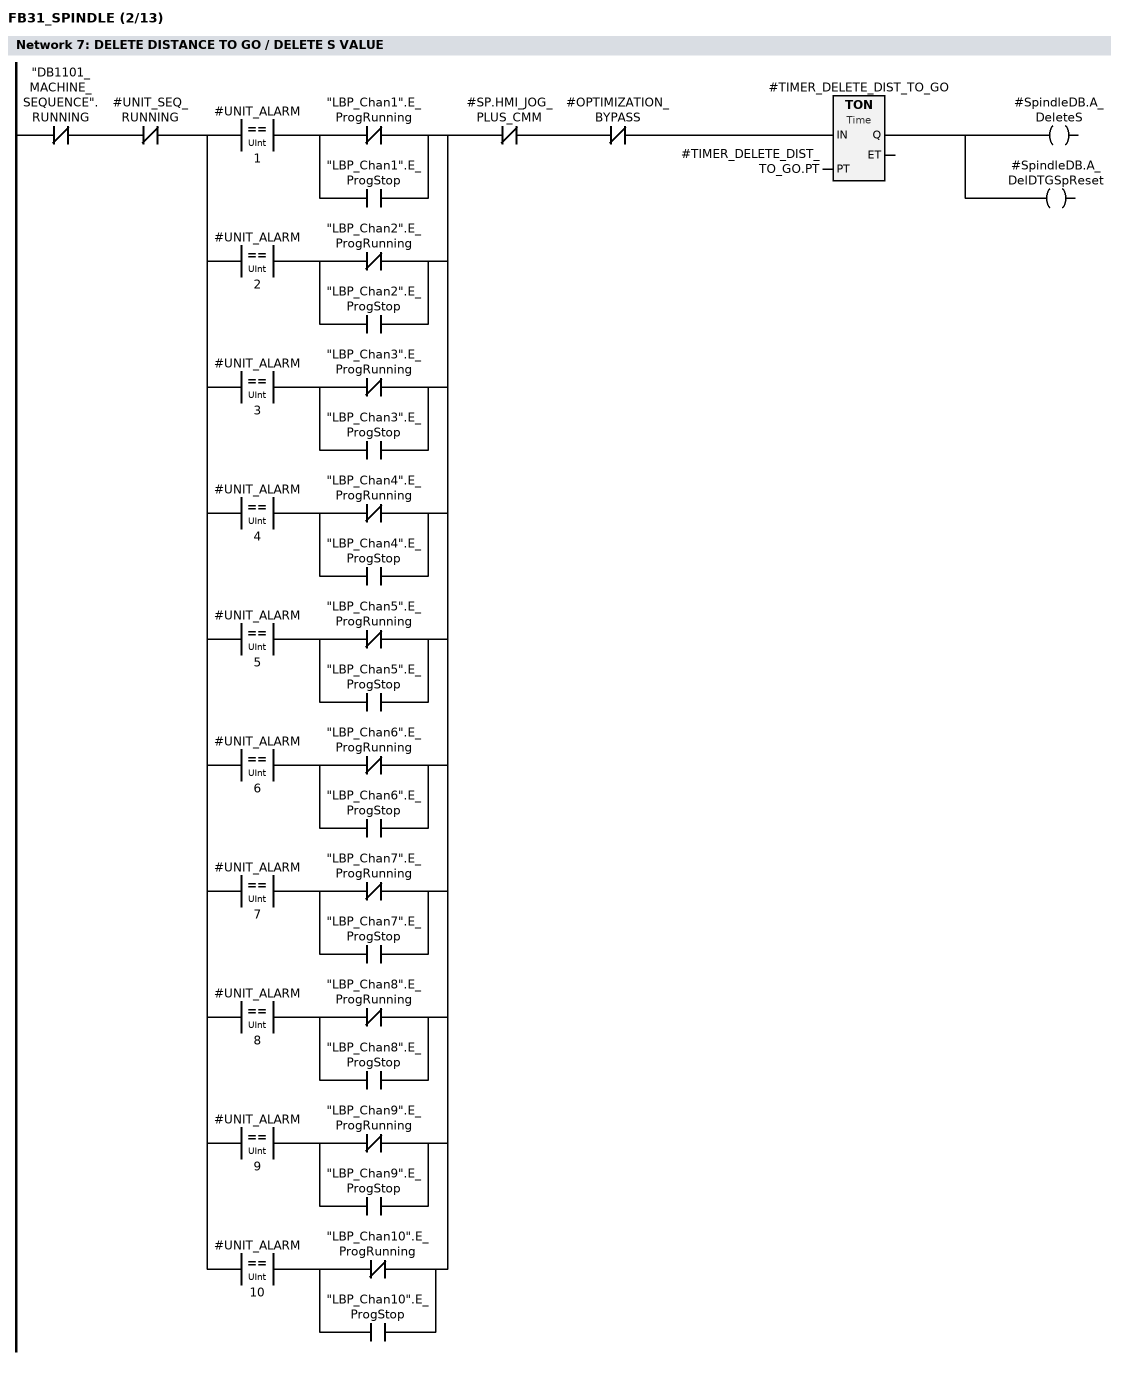
   RUNG wire#powerrail
      I_Contact( "DB1101_MACHINE_SEQUENCE".RUNNING )
      I_Contact( #UNIT_SEQ_RUNNING )
      wire#w1
      { S7_Templates := "SrcType := UInt" } EQ_Contact(in1 := #UNIT_ALARM, in2 := 1)
      wire#w2
      I_Contact( "LBP_Chan1".E_ProgRunning )
      wire#w3
      I_Contact( #SP.HMI_JOG_PLUS_CMM )
      I_Contact( #OPTIMIZATION_BYPASS )
      { S7_Templates := "time_type := Time" } #TIMER_DELETE_DIST_TO_GO.TON(pt := #TIMER_DELETE_DIST_TO_GO.PT, et =>)
      wire#w13
      Coil( #SpindleDB.A_DeleteS )
   END_RUNG
   RUNG wire#w2
      Contact( "LBP_Chan1".E_ProgStop )
   END_RUNG wire#w3
   RUNG wire#w1
      { S7_Templates := "SrcType := UInt" } EQ_Contact(in1 := #UNIT_ALARM, in2 := 2)
      wire#w4
      I_Contact( "LBP_Chan2".E_ProgRunning )
   END_RUNG wire#w3
   RUNG wire#w4
      Contact( "LBP_Chan2".E_ProgStop )
   END_RUNG wire#w3
   RUNG wire#w1
      { S7_Templates := "SrcType := UInt" } EQ_Contact(in1 := #UNIT_ALARM, in2 := 3)
      wire#w5
      I_Contact( "LBP_Chan3".E_ProgRunning )
   END_RUNG wire#w3
   RUNG wire#w5
      Contact( "LBP_Chan3".E_ProgStop )
   END_RUNG wire#w3
   RUNG wire#w1
      { S7_Templates := "SrcType := UInt" } EQ_Contact(in1 := #UNIT_ALARM, in2 := 4)
      wire#w6
      I_Contact( "LBP_Chan4".E_ProgRunning )
   END_RUNG wire#w3
   RUNG wire#w6
      Contact( "LBP_Chan4".E_ProgStop )
   END_RUNG wire#w3
   RUNG wire#w1
      { S7_Templates := "SrcType := UInt" } EQ_Contact(in1 := #UNIT_ALARM, in2 := 5)
      wire#w7
      I_Contact( "LBP_Chan5".E_ProgRunning )
   END_RUNG wire#w3
   RUNG wire#w7
      Contact( "LBP_Chan5".E_ProgStop )
   END_RUNG wire#w3
   RUNG wire#w1
      { S7_Templates := "SrcType := UInt" } EQ_Contact(in1 := #UNIT_ALARM, in2 := 6)
      wire#w8
      I_Contact( "LBP_Chan6".E_ProgRunning )
   END_RUNG wire#w3
   RUNG wire#w8
      Contact( "LBP_Chan6".E_ProgStop )
   END_RUNG wire#w3
   RUNG wire#w1
      { S7_Templates := "SrcType := UInt" } EQ_Contact(in1 := #UNIT_ALARM, in2 := 7)
      wire#w9
      I_Contact( "LBP_Chan7".E_ProgRunning )
   END_RUNG wire#w3
   RUNG wire#w9
      Contact( "LBP_Chan7".E_ProgStop )
   END_RUNG wire#w3
   RUNG wire#w1
      { S7_Templates := "SrcType := UInt" } EQ_Contact(in1 := #UNIT_ALARM, in2 := 8)
      wire#w10
      I_Contact( "LBP_Chan8".E_ProgRunning )
   END_RUNG wire#w3
   RUNG wire#w10
      Contact( "LBP_Chan8".E_ProgStop )
   END_RUNG wire#w3
   RUNG wire#w1
      { S7_Templates := "SrcType := UInt" } EQ_Contact(in1 := #UNIT_ALARM, in2 := 9)
      wire#w11
      I_Contact( "LBP_Chan9".E_ProgRunning )
   END_RUNG wire#w3
   RUNG wire#w11
      Contact( "LBP_Chan9".E_ProgStop )
   END_RUNG wire#w3
   RUNG wire#w1
      { S7_Templates := "SrcType := UInt" } EQ_Contact(in1 := #UNIT_ALARM, in2 := 10)
      wire#w12
      I_Contact( "LBP_Chan10".E_ProgRunning )
   END_RUNG wire#w3
   RUNG wire#w12
      Contact( "LBP_Chan10".E_ProgStop )
   END_RUNG wire#w3
   RUNG wire#w13
      Coil( #SpindleDB.A_DelDTGSpReset )
   END_RUNG
   // the same network as SCL:
   #TIMER_DELETE_DIST_TO_GO(IN := NOT "DB1101_MACHINE_SEQUENCE".RUNNING AND NOT #UNIT_SEQ_RUNNING AND (((#UNIT_ALARM = 1) AND (NOT "LBP_Chan1".E_ProgRunning OR "LBP_Chan1".E_ProgStop)) OR ((#UNIT_ALARM = 2) AND (NOT "LBP_Chan2".E_ProgRunning OR "LBP_Chan2".E_ProgStop)) OR ((#UNIT_ALARM = 3) AND (NOT "LBP_Chan3".E_ProgRunning OR "LBP_Chan3".E_ProgStop)) OR ((#UNIT_ALARM = 4) AND (NOT "LBP_Chan4".E_ProgRunning OR "LBP_Chan4".E_ProgStop)) OR ((#UNIT_ALARM = 5) AND (NOT "LBP_Chan5".E_ProgRunning OR "LBP_Chan5".E_ProgStop)) OR ((#UNIT_ALARM = 6) AND (NOT "LBP_Chan6".E_ProgRunning OR "LBP_Chan6".E_ProgStop)) OR ((#UNIT_ALARM = 7) AND (NOT "LBP_Chan7".E_ProgRunning OR "LBP_Chan7".E_ProgStop)) OR ((#UNIT_ALARM = 8) AND (NOT "LBP_Chan8".E_ProgRunning OR "LBP_Chan8".E_ProgStop)) OR ((#UNIT_ALARM = 9) AND (NOT "LBP_Chan9".E_ProgRunning OR "LBP_Chan9".E_ProgStop)) OR ((#UNIT_ALARM = 10) AND (NOT "LBP_Chan10".E_ProgRunning OR "LBP_Chan10".E_ProgStop))) AND NOT #SP.HMI_JOG_PLUS_CMM AND NOT #OPTIMIZATION_BYPASS,   // TON
                           PT := #TIMER_DELETE_DIST_TO_GO.PT);
   #SpindleDB.A_DeleteS := #TIMER_DELETE_DIST_TO_GO.Q;
   #SpindleDB.A_DelDTGSpReset := #TIMER_DELETE_DIST_TO_GO.Q;
END_REGION

REGION Network 8: POSITION MEASURING SYTEM
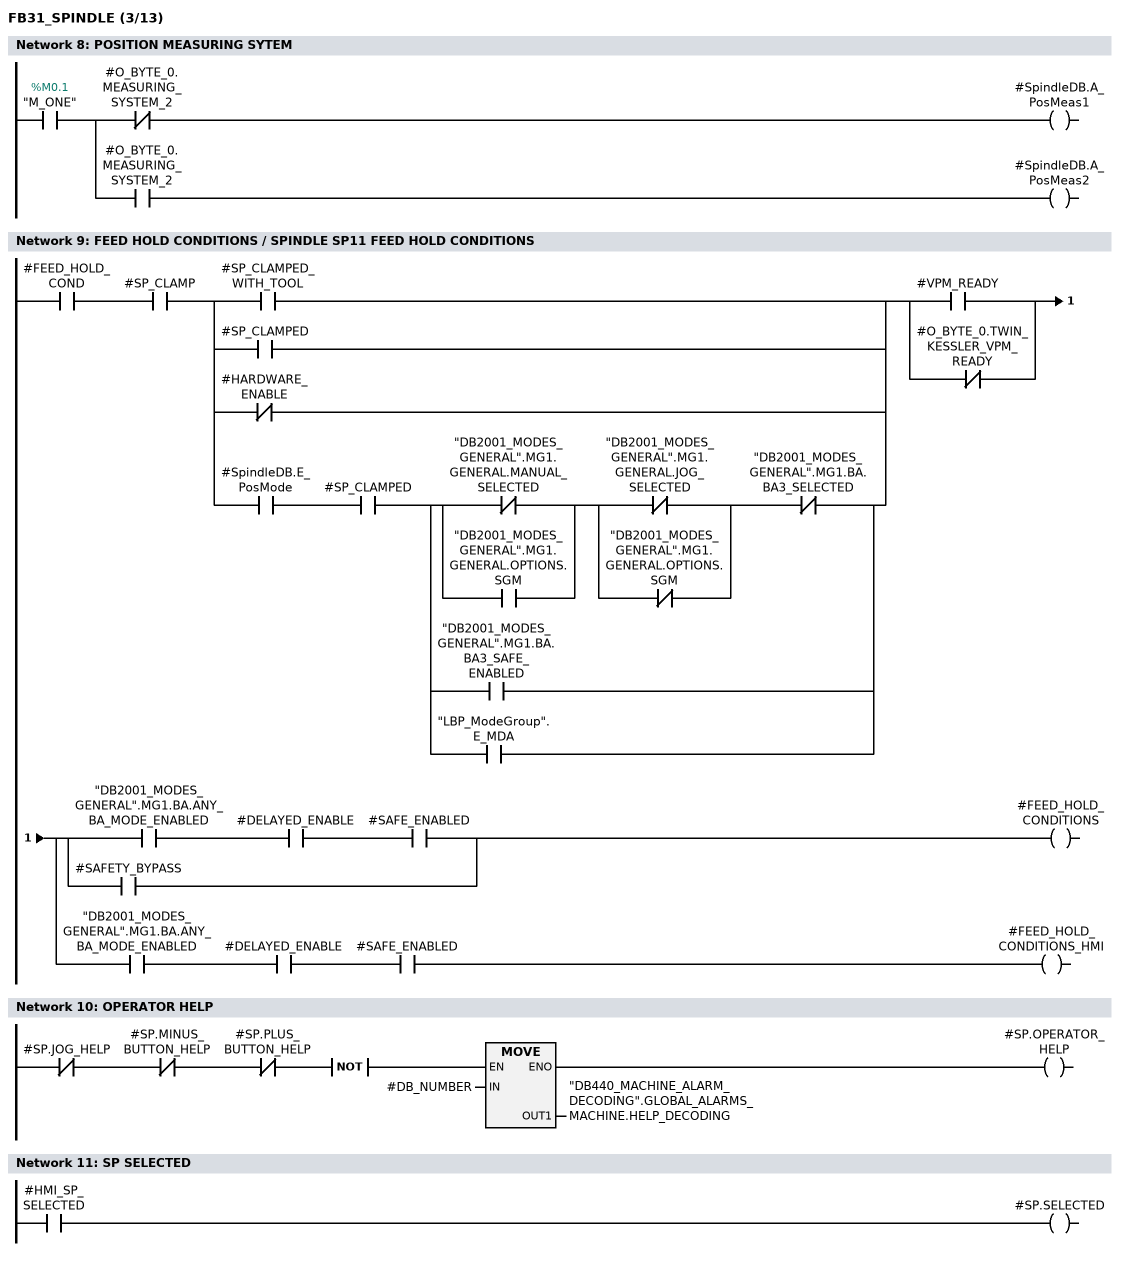
   RUNG wire#powerrail
      Contact( "M_ONE" )
      wire#w1
      I_Contact( #O_BYTE_0.MEASURING_SYSTEM_2 )
      Coil( #SpindleDB.A_PosMeas1 )
   END_RUNG
   RUNG wire#w1
      Contact( #O_BYTE_0.MEASURING_SYSTEM_2 )
      Coil( #SpindleDB.A_PosMeas2 )
   END_RUNG
   // the same network as SCL:
   #SpindleDB.A_PosMeas1 := "M_ONE" AND NOT #O_BYTE_0.MEASURING_SYSTEM_2;
   #SpindleDB.A_PosMeas2 := "M_ONE" AND #O_BYTE_0.MEASURING_SYSTEM_2;
END_REGION

REGION Network 9: FEED HOLD CONDITIONS / SPINDLE SP11 FEED HOLD CONDITIONS
   RUNG wire#powerrail
      Contact( #FEED_HOLD_COND )
      Contact( #SP_CLAMP )
      wire#w1
      Contact( #SP_CLAMPED_WITH_TOOL )
      wire#w2
      Contact( #VPM_READY )
      wire#w6
      Contact( "DB2001_MODES_GENERAL".MG1.BA.ANY_BA_MODE_ENABLED )
      Contact( #DELAYED_ENABLE )
      Contact( #SAFE_ENABLED )
      wire#w7
      Coil( #FEED_HOLD_CONDITIONS )
   END_RUNG
   RUNG wire#w1
      Contact( #SP_CLAMPED )
   END_RUNG wire#w2
   RUNG wire#w1
      I_Contact( #HARDWARE_ENABLE )
   END_RUNG wire#w2
   RUNG wire#w1
      Contact( #SpindleDB.E_PosMode )
      Contact( #SP_CLAMPED )
      wire#w3
      I_Contact( "DB2001_MODES_GENERAL".MG1.GENERAL.MANUAL_SELECTED )
      wire#w4
      I_Contact( "DB2001_MODES_GENERAL".MG1.GENERAL.JOG_SELECTED )
      wire#w5
      I_Contact( "DB2001_MODES_GENERAL".MG1.BA.BA3_SELECTED )
   END_RUNG wire#w2
   RUNG wire#w3
      Contact( "DB2001_MODES_GENERAL".MG1.GENERAL.OPTIONS.SGM )
   END_RUNG wire#w4
   RUNG wire#w4
      I_Contact( "DB2001_MODES_GENERAL".MG1.GENERAL.OPTIONS.SGM )
   END_RUNG wire#w5
   RUNG wire#w3
      Contact( "DB2001_MODES_GENERAL".MG1.BA.BA3_SAFE_ENABLED )
   END_RUNG wire#w2
   RUNG wire#w3
      Contact( "LBP_ModeGroup".E_MDA )
   END_RUNG wire#w2
   RUNG wire#w2
      I_Contact( #O_BYTE_0.TWIN_KESSLER_VPM_READY )
   END_RUNG wire#w6
   RUNG wire#w6
      Contact( #SAFETY_BYPASS )
   END_RUNG wire#w7
   RUNG wire#w6
      Contact( "DB2001_MODES_GENERAL".MG1.BA.ANY_BA_MODE_ENABLED )
      Contact( #DELAYED_ENABLE )
      Contact( #SAFE_ENABLED )
      Coil( #FEED_HOLD_CONDITIONS_HMI )
   END_RUNG
   // the same network as SCL:
   #_w1 := #FEED_HOLD_COND AND #SP_CLAMP AND (#SP_CLAMPED_WITH_TOOL OR #SP_CLAMPED OR NOT #HARDWARE_ENABLE OR (#SpindleDB.E_PosMode AND #SP_CLAMPED AND (((NOT "DB2001_MODES_GENERAL".MG1.GENERAL.MANUAL_SELECTED OR "DB2001_MODES_GENERAL".MG1.GENERAL.OPTIONS.SGM) AND (NOT "DB2001_MODES_GENERAL".MG1.GENERAL.JOG_SELECTED OR NOT "DB2001_MODES_GENERAL".MG1.GENERAL.OPTIONS.SGM) AND NOT "DB2001_MODES_GENERAL".MG1.BA.BA3_SELECTED) OR "DB2001_MODES_GENERAL".MG1.BA.BA3_SAFE_ENABLED OR "LBP_ModeGroup".E_MDA))) AND (#VPM_READY OR NOT #O_BYTE_0.TWIN_KESSLER_VPM_READY);
   #FEED_HOLD_CONDITIONS := #_w1 AND (("DB2001_MODES_GENERAL".MG1.BA.ANY_BA_MODE_ENABLED AND #DELAYED_ENABLE AND #SAFE_ENABLED) OR #SAFETY_BYPASS);
   #FEED_HOLD_CONDITIONS_HMI := #_w1 AND "DB2001_MODES_GENERAL".MG1.BA.ANY_BA_MODE_ENABLED AND #DELAYED_ENABLE AND #SAFE_ENABLED;
END_REGION

REGION Network 10: OPERATOR HELP
   RUNG wire#powerrail
      I_Contact( #SP.JOG_HELP )
      I_Contact( #SP.MINUS_BUTTON_HELP )
      I_Contact( #SP.PLUS_BUTTON_HELP )
      Not()
      { S7_GenerateENO := "TRUE" } Move(in := #DB_NUMBER, out1 => "DB440_MACHINE_ALARM_DECODING".GLOBAL_ALARMS_MACHINE.HELP_DECODING)
      Coil( #SP.OPERATOR_HELP )
   END_RUNG
   // the same network as SCL:
   // ENO of a box is taken as its EN; it also drops when the box reports an error
   #_w1 := NOT (NOT #SP.JOG_HELP AND NOT #SP.MINUS_BUTTON_HELP AND NOT #SP.PLUS_BUTTON_HELP);
   IF #_w1 THEN "DB440_MACHINE_ALARM_DECODING".GLOBAL_ALARMS_MACHINE.HELP_DECODING := #DB_NUMBER; END_IF;
   #SP.OPERATOR_HELP := #_w1;
END_REGION

REGION Network 11: SP SELECTED
   RUNG wire#powerrail
      Contact( #HMI_SP_SELECTED )
      Coil( #SP.SELECTED )
   END_RUNG
   // the same network as SCL:
   #SP.SELECTED := #HMI_SP_SELECTED;
END_REGION

REGION Network 12: SP DESELECTED
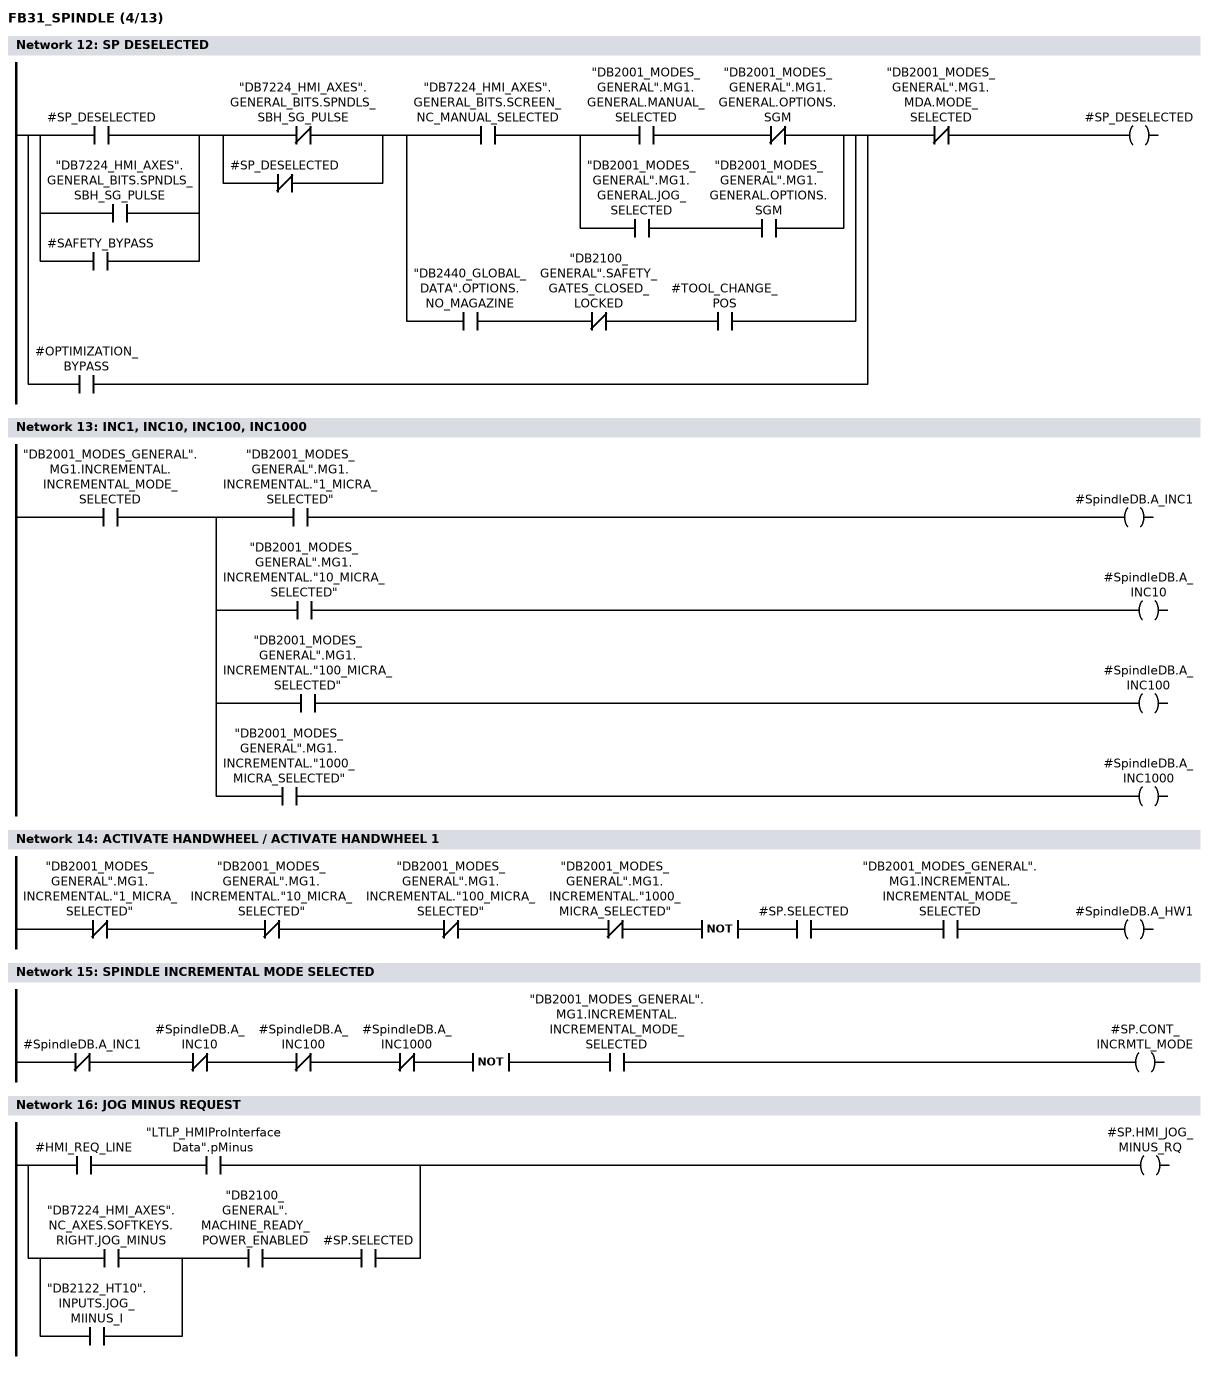
   RUNG wire#powerrail
      Contact( #SP_DESELECTED )
      wire#w1
      I_Contact( "DB7224_HMI_AXES".GENERAL_BITS.SPNDLS_SBH_SG_PULSE )
      wire#w2
      Contact( "DB7224_HMI_AXES".GENERAL_BITS.SCREEN_NC_MANUAL_SELECTED )
      wire#w3
      Contact( "DB2001_MODES_GENERAL".MG1.GENERAL.MANUAL_SELECTED )
      I_Contact( "DB2001_MODES_GENERAL".MG1.GENERAL.OPTIONS.SGM )
      wire#w4
      I_Contact( "DB2001_MODES_GENERAL".MG1.MDA.MODE_SELECTED )
      Coil( #SP_DESELECTED )
   END_RUNG
   RUNG wire#powerrail
      Contact( "DB7224_HMI_AXES".GENERAL_BITS.SPNDLS_SBH_SG_PULSE )
   END_RUNG wire#w1
   RUNG wire#powerrail
      Contact( #SAFETY_BYPASS )
   END_RUNG wire#w1
   RUNG wire#w1
      I_Contact( #SP_DESELECTED )
   END_RUNG wire#w2
   RUNG wire#w3
      Contact( "DB2001_MODES_GENERAL".MG1.GENERAL.JOG_SELECTED )
      Contact( "DB2001_MODES_GENERAL".MG1.GENERAL.OPTIONS.SGM )
   END_RUNG wire#w4
   RUNG wire#w2
      Contact( "DB2440_GLOBAL_DATA".OPTIONS.NO_MAGAZINE )
      I_Contact( "DB2100_GENERAL".SAFETY_GATES_CLOSED_LOCKED )
      Contact( #TOOL_CHANGE_POS )
   END_RUNG wire#w4
   RUNG wire#powerrail
      Contact( #OPTIMIZATION_BYPASS )
   END_RUNG wire#w4
   // the same network as SCL:
   #SP_DESELECTED := (((#SP_DESELECTED OR "DB7224_HMI_AXES".GENERAL_BITS.SPNDLS_SBH_SG_PULSE OR #SAFETY_BYPASS) AND (NOT "DB7224_HMI_AXES".GENERAL_BITS.SPNDLS_SBH_SG_PULSE OR NOT #SP_DESELECTED) AND (("DB7224_HMI_AXES".GENERAL_BITS.SCREEN_NC_MANUAL_SELECTED AND (("DB2001_MODES_GENERAL".MG1.GENERAL.MANUAL_SELECTED AND NOT "DB2001_MODES_GENERAL".MG1.GENERAL.OPTIONS.SGM) OR ("DB2001_MODES_GENERAL".MG1.GENERAL.JOG_SELECTED AND "DB2001_MODES_GENERAL".MG1.GENERAL.OPTIONS.SGM))) OR ("DB2440_GLOBAL_DATA".OPTIONS.NO_MAGAZINE AND NOT "DB2100_GENERAL".SAFETY_GATES_CLOSED_LOCKED AND #TOOL_CHANGE_POS))) OR #OPTIMIZATION_BYPASS) AND NOT "DB2001_MODES_GENERAL".MG1.MDA.MODE_SELECTED;
END_REGION

REGION Network 13: INC1, INC10, INC100, INC1000
   RUNG wire#powerrail
      Contact( "DB2001_MODES_GENERAL".MG1.INCREMENTAL.INCREMENTAL_MODE_SELECTED )
      wire#w1
      Contact( "DB2001_MODES_GENERAL".MG1.INCREMENTAL."1_MICRA_SELECTED" )
      Coil( #SpindleDB.A_INC1 )
   END_RUNG
   RUNG wire#w1
      Contact( "DB2001_MODES_GENERAL".MG1.INCREMENTAL."10_MICRA_SELECTED" )
      Coil( #SpindleDB.A_INC10 )
   END_RUNG
   RUNG wire#w1
      Contact( "DB2001_MODES_GENERAL".MG1.INCREMENTAL."100_MICRA_SELECTED" )
      Coil( #SpindleDB.A_INC100 )
   END_RUNG
   RUNG wire#w1
      Contact( "DB2001_MODES_GENERAL".MG1.INCREMENTAL."1000_MICRA_SELECTED" )
      Coil( #SpindleDB.A_INC1000 )
   END_RUNG
   // the same network as SCL:
   #SpindleDB.A_INC1 := "DB2001_MODES_GENERAL".MG1.INCREMENTAL.INCREMENTAL_MODE_SELECTED AND "DB2001_MODES_GENERAL".MG1.INCREMENTAL."1_MICRA_SELECTED";
   #SpindleDB.A_INC10 := "DB2001_MODES_GENERAL".MG1.INCREMENTAL.INCREMENTAL_MODE_SELECTED AND "DB2001_MODES_GENERAL".MG1.INCREMENTAL."10_MICRA_SELECTED";
   #SpindleDB.A_INC100 := "DB2001_MODES_GENERAL".MG1.INCREMENTAL.INCREMENTAL_MODE_SELECTED AND "DB2001_MODES_GENERAL".MG1.INCREMENTAL."100_MICRA_SELECTED";
   #SpindleDB.A_INC1000 := "DB2001_MODES_GENERAL".MG1.INCREMENTAL.INCREMENTAL_MODE_SELECTED AND "DB2001_MODES_GENERAL".MG1.INCREMENTAL."1000_MICRA_SELECTED";
END_REGION

